END_VAR
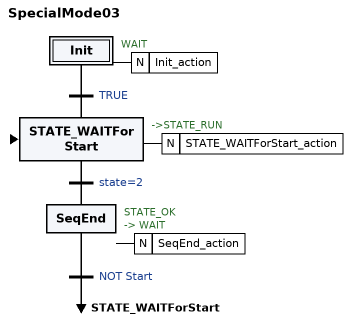
[picture p0: SpecialMode03 (SFC)]
INITIAL_STEP Init: (* WAIT *)
	Init_action(N);
END_STEP
TRANSITION FROM Init TO STATE_WAITForStart := TRUE;
END_TRANSITION
STEP STATE_WAITForStart: (* ->STATE_RUN *)
	STATE_WAITForStart_action(N);
END_STEP
TRANSITION FROM STATE_WAITForStart TO SeqEnd := state=2;
END_TRANSITION
STEP SeqEnd: (* STATE_OK / -> WAIT *)
	SeqEnd_action(N);
END_STEP
TRANSITION FROM SeqEnd TO STATE_WAITForStart := NOT Start;
END_TRANSITION

ACTION Init_action:
Start:=FALSE;
State:=STATE_WAIT;
END_ACTION

ACTION STATE_WAITForStart_action:
IF Start=TRUE
THEN
	State:=STATE_RUN;
	Result:=RESULT_NON;
	SFCTimeStart:=TIME();
(*ELSE*)
END_IF
END_ACTION

ACTION SeqEnd_action:
IF 	State=STATE_RUN THEN
	SFCTime:=TIME_TO_DINT(TIME()-SFCTimeStart);
	State:=STATE_OK;
END_IF

IF 	NOT Start THEN
	State:=STATE_WAIT;
END_IF
END_ACTION
END_PROGRAM

(* POU Stations/ST_00/ST00_SFCs/CheckSFCInInit, ST *)
PROGRAM CheckSFCInInit

VAR_OUTPUT

  AllSeqInInit	:	BOOL;

END_VAR
 AllSeqInInit:=
	ST03_Main.State=STATE_WAIT AND
	ST02_Main.State=STATE_WAIT AND
	(ST08_Process.State=STATE_WAIT OR ST08_Process.State=STATE_OK ) AND
	ST08_Palletizing.State=STATE_WAIT AND
	ST08_Depalletizing.State=STATE_WAIT
;
END_PROGRAM

(* POU Stations/ST_03_Ruestsaetze/ST_03_SFCs/ST03_Main, SFC *)
PROGRAM ST03_Main

VAR_OUTPUT
	SFCCurrentPOU			: STRING:='ST03_Main';
	SFCCurrentStep			: STRING:='';
	FB_CurrentStepHistorie	: FB_CurrentStepHistorie;
	SFCTime					: DINT;
	State   				: StateObject	:= STATE_WAIT;

	Nest10Locked			: BOOL;
	Nest10Done				: BOOL;
	IstPosHelp				: LREAL;
END_VAR
VAR_INPUT
	RunEmpty				: BOOL;
	TestPartsRemove			: BOOL;
	Result 					: DINT;
END_VAR
VAR
	MsgOK					: BOOL;
	MsgCancel				: BOOL;
	SFCRun					: BOOL;
	SFCTimeStart			: TIME;
	Delay					: TON;
	Error					: ErrorStruct;
	(* Userdefinded area *)
	AnzahlTeile   			: DINT;
	PutIdx					: DINT;
	Nest_Empty      		: BOOL;
	kein_Teil_NOK			: BOOL;
	CTR						: DINT;
	CTR2					: DINT;
	Result_help				: DINT;
END_VAR
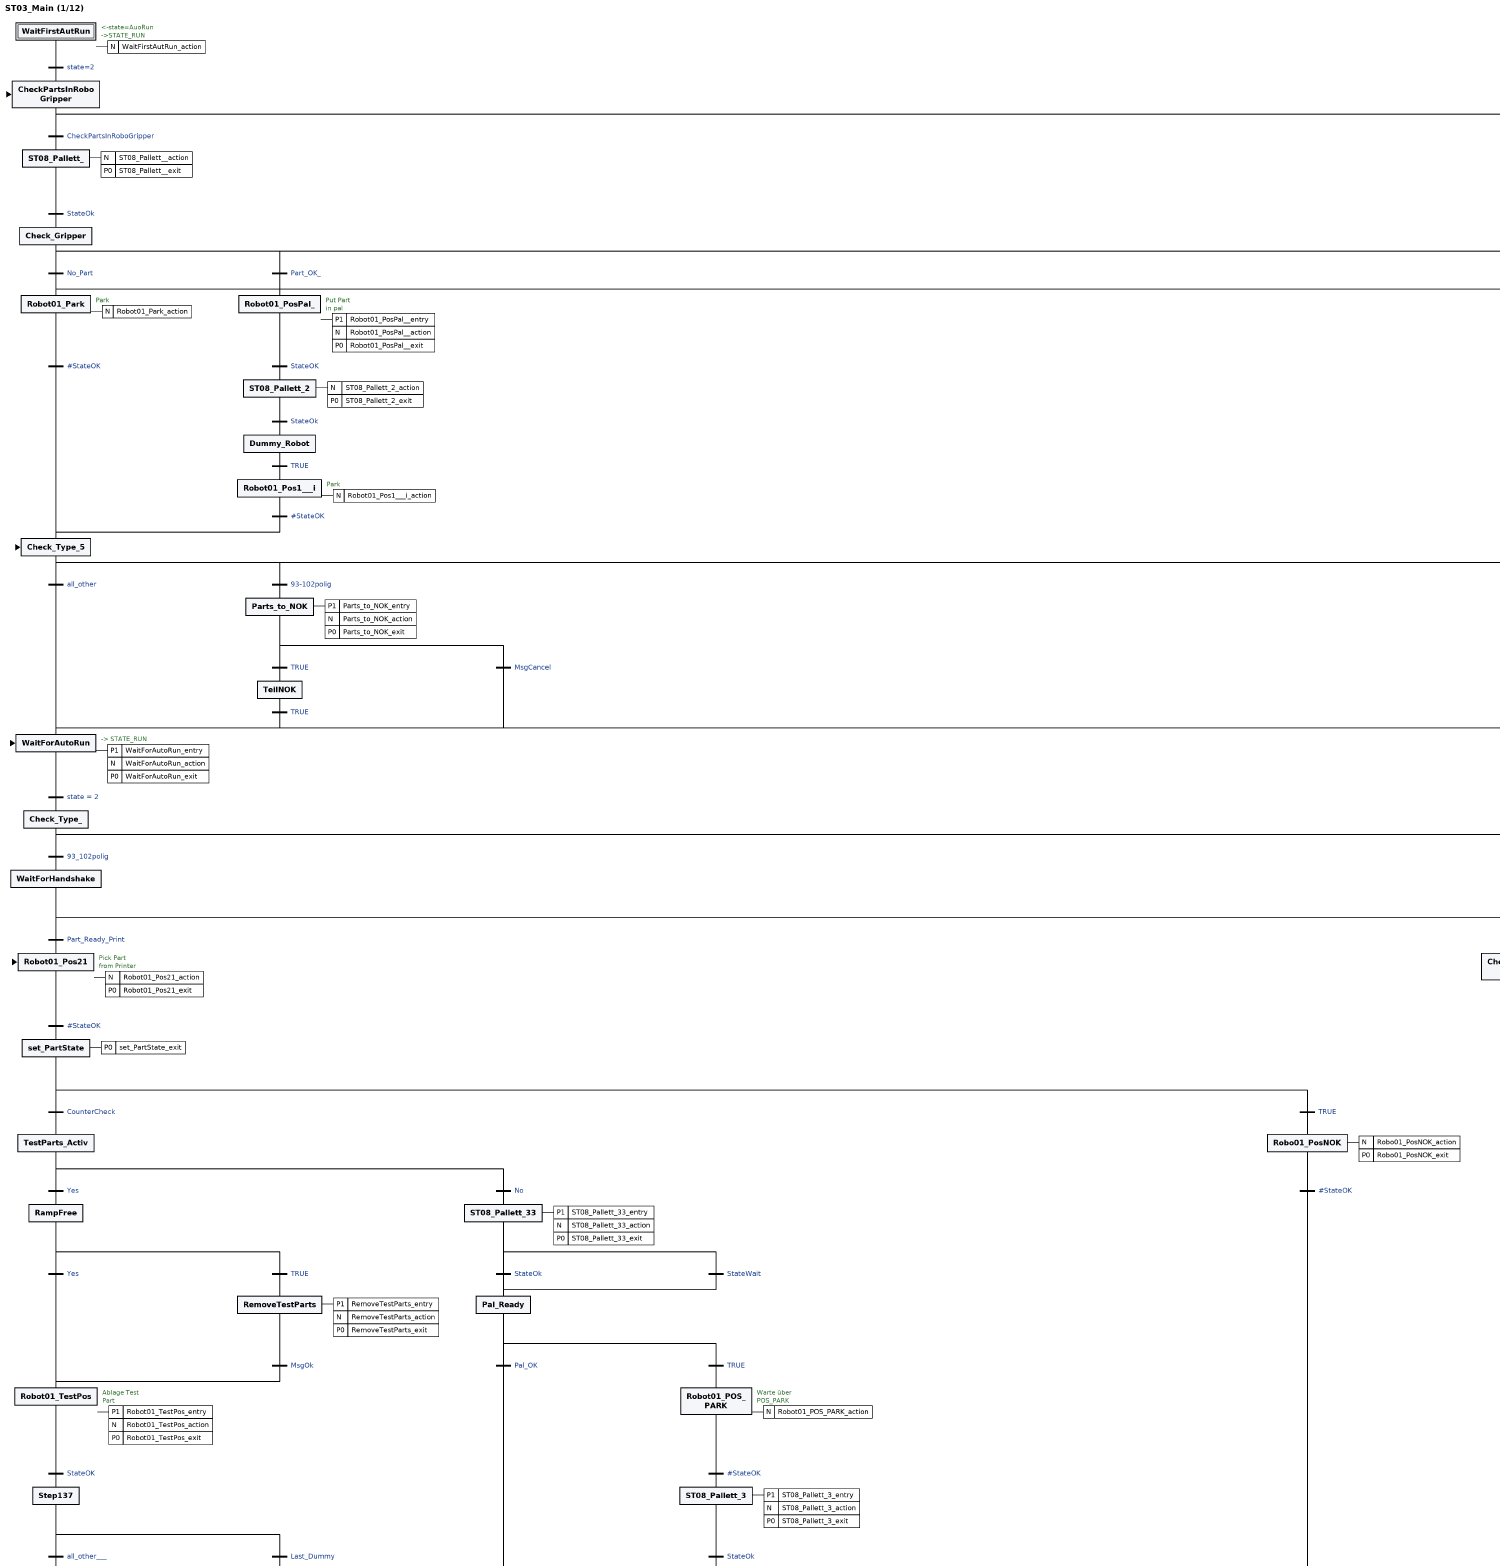
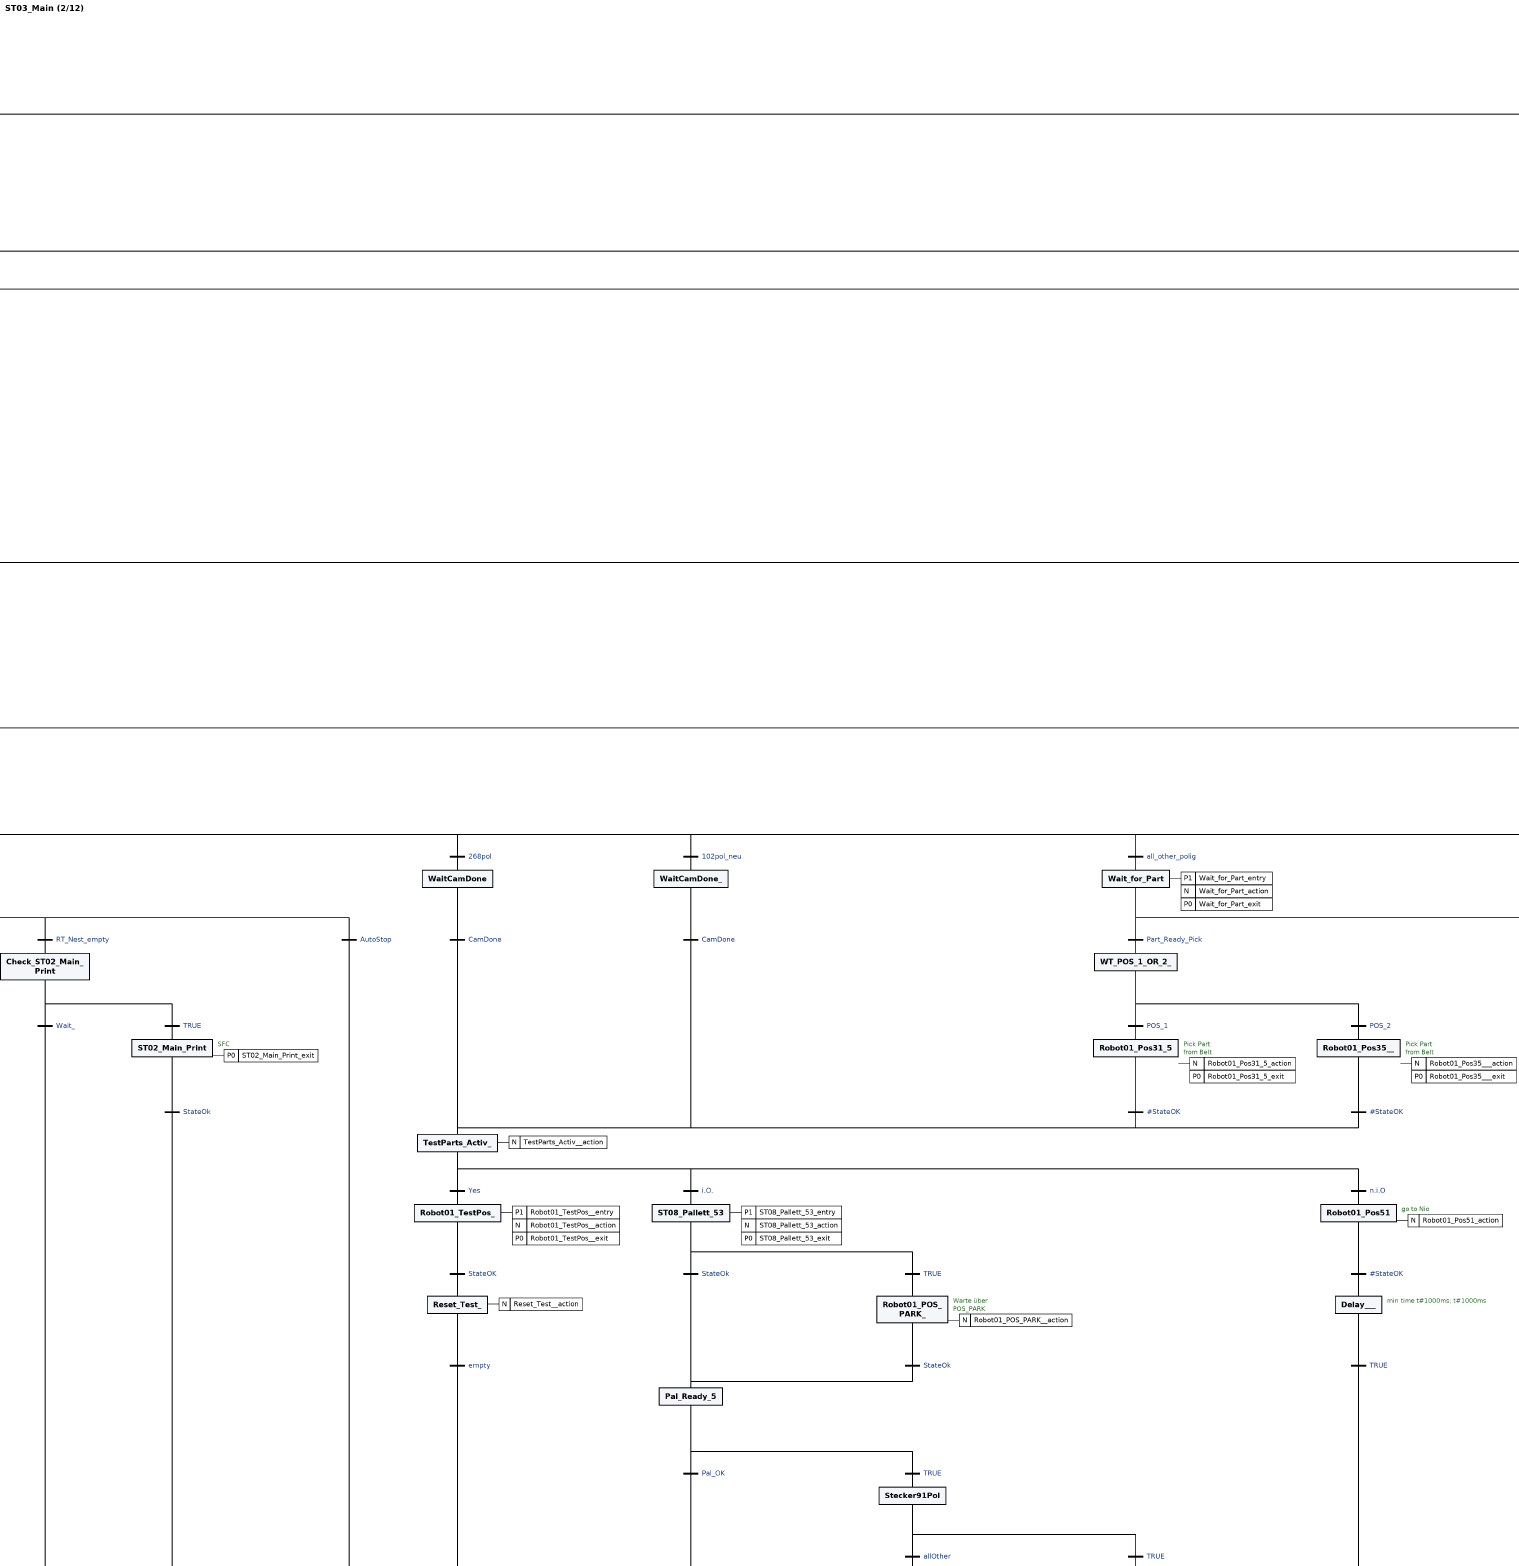
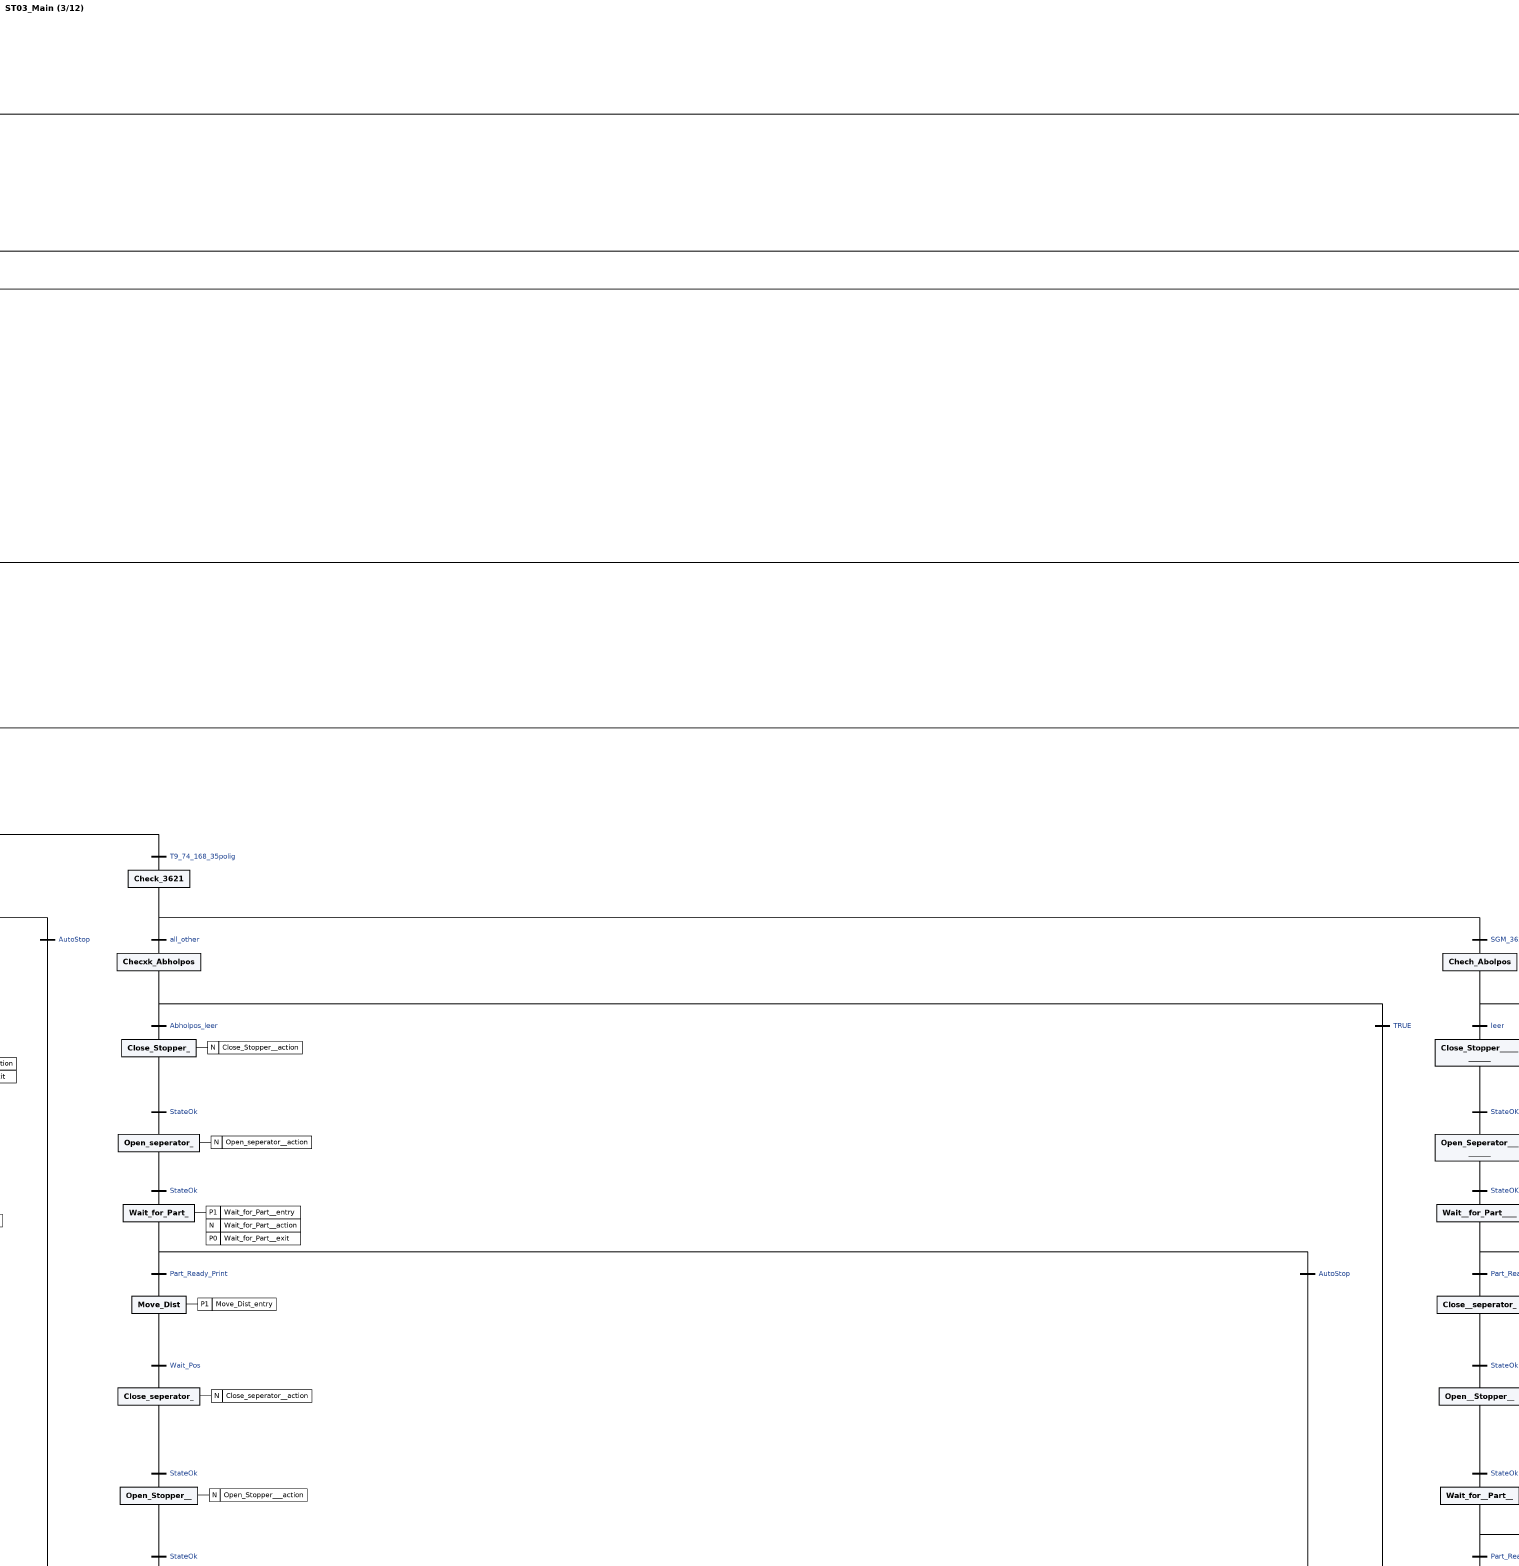
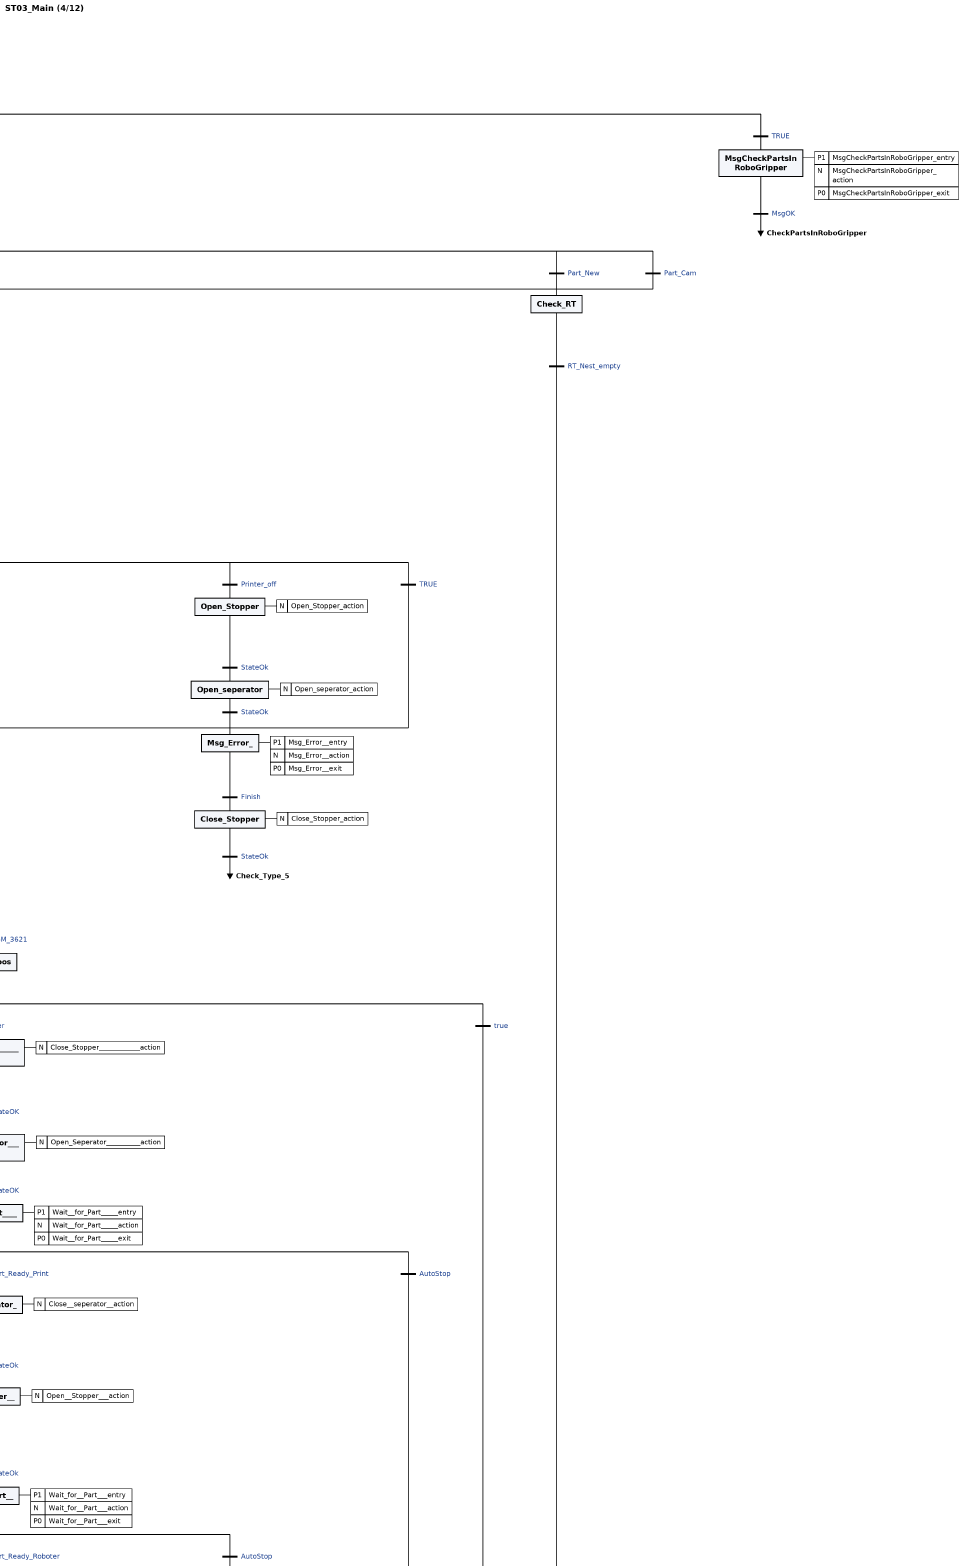
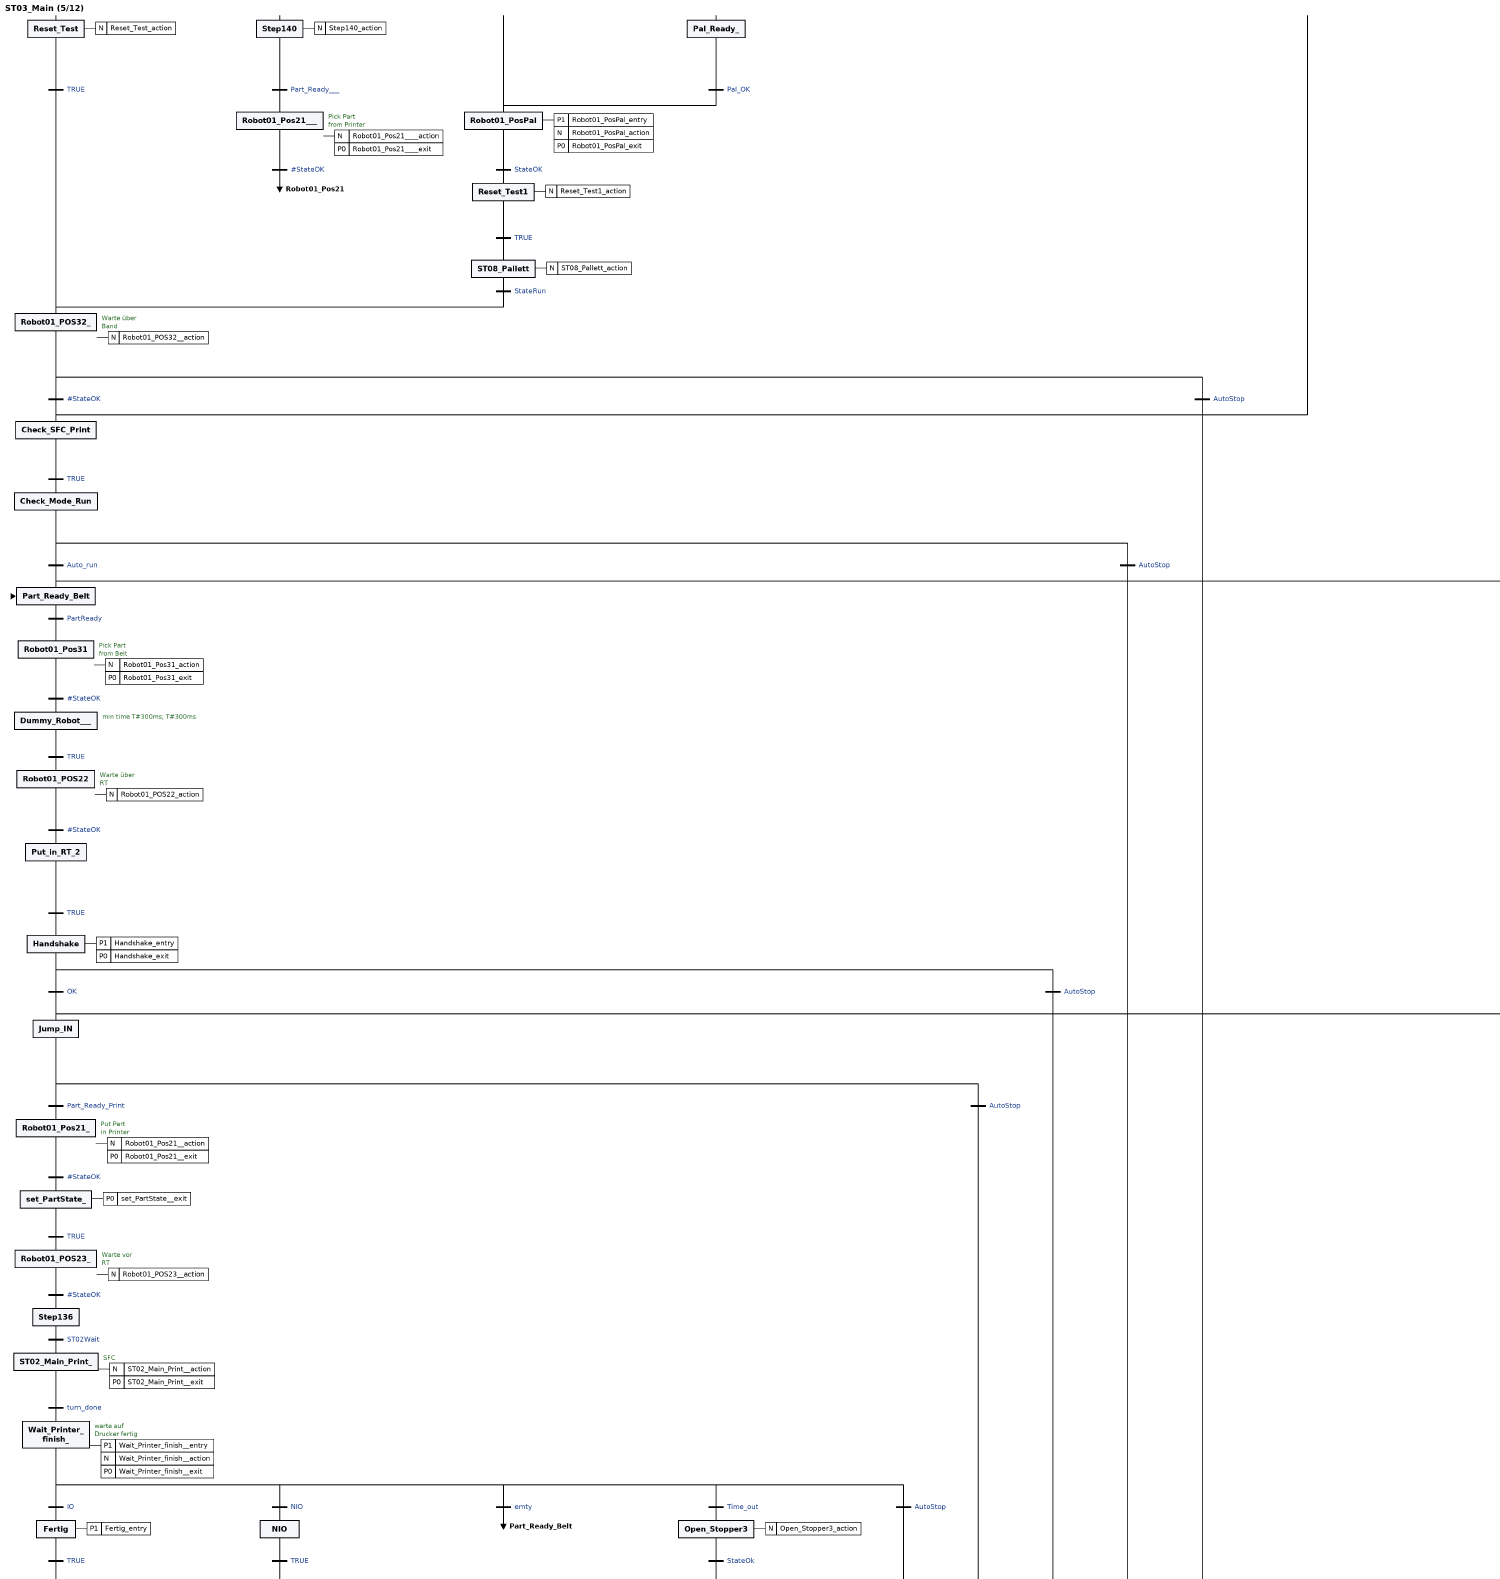
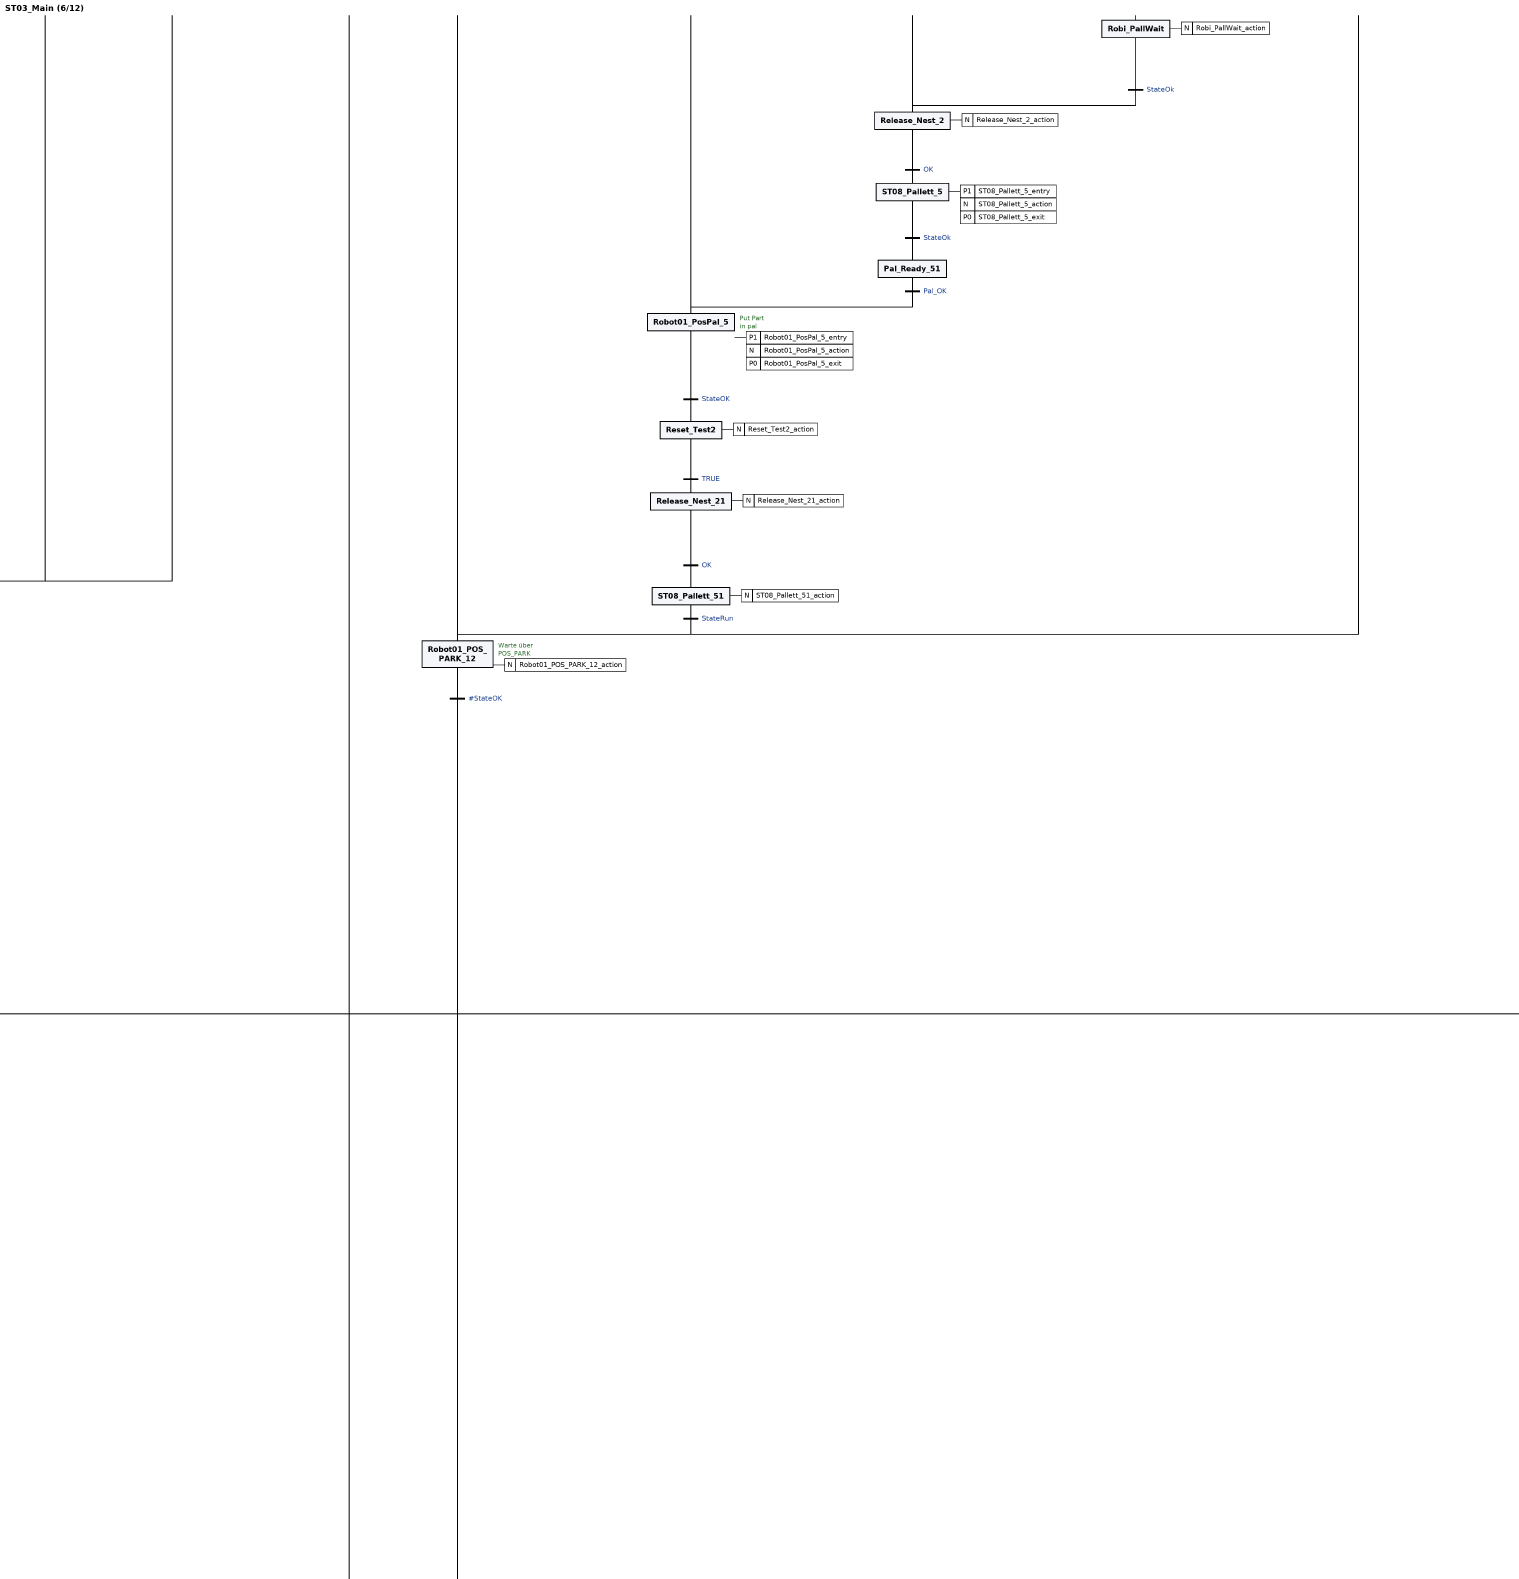
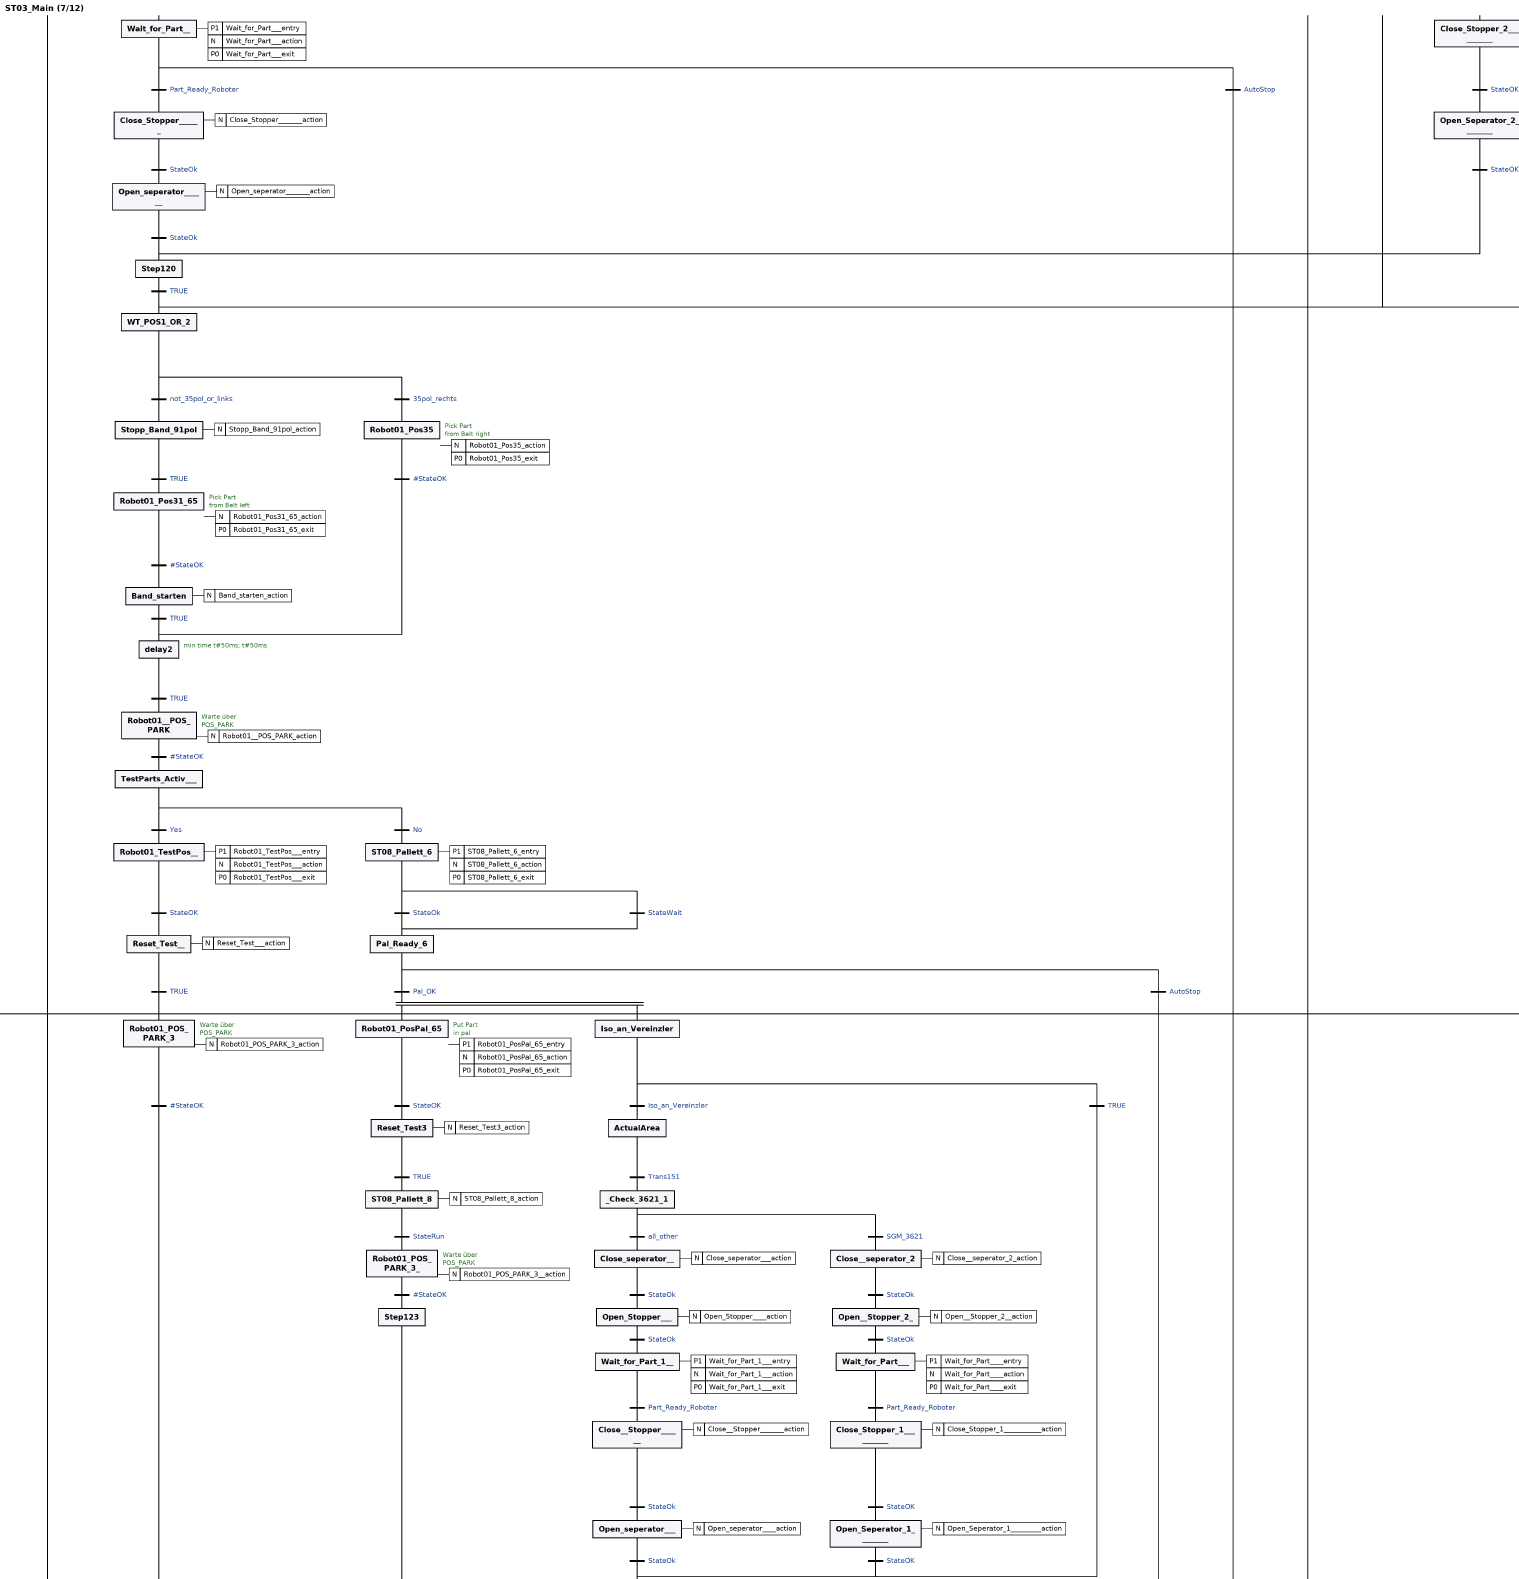
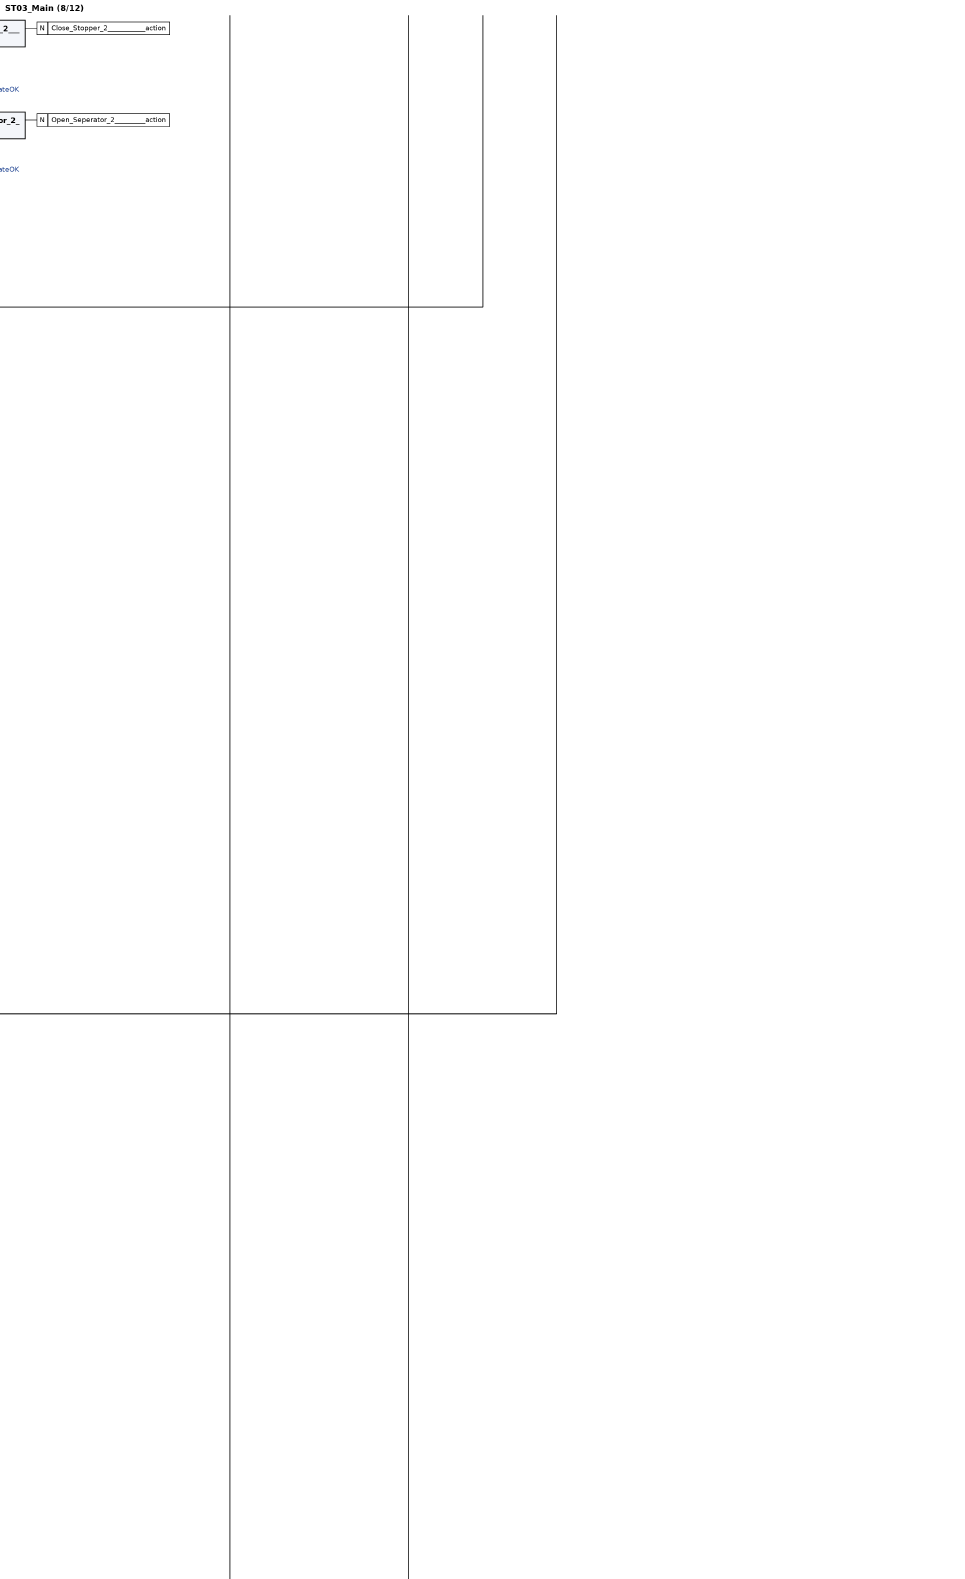
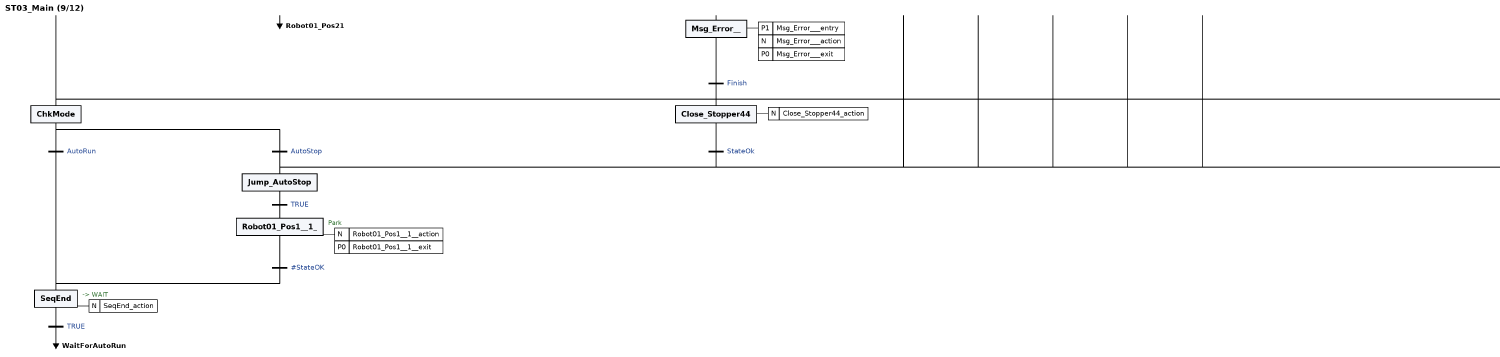
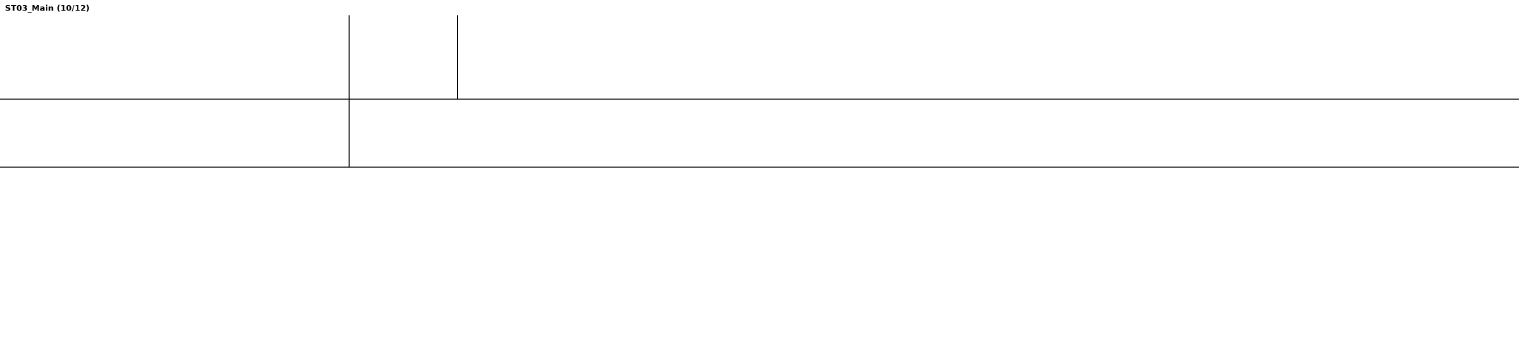
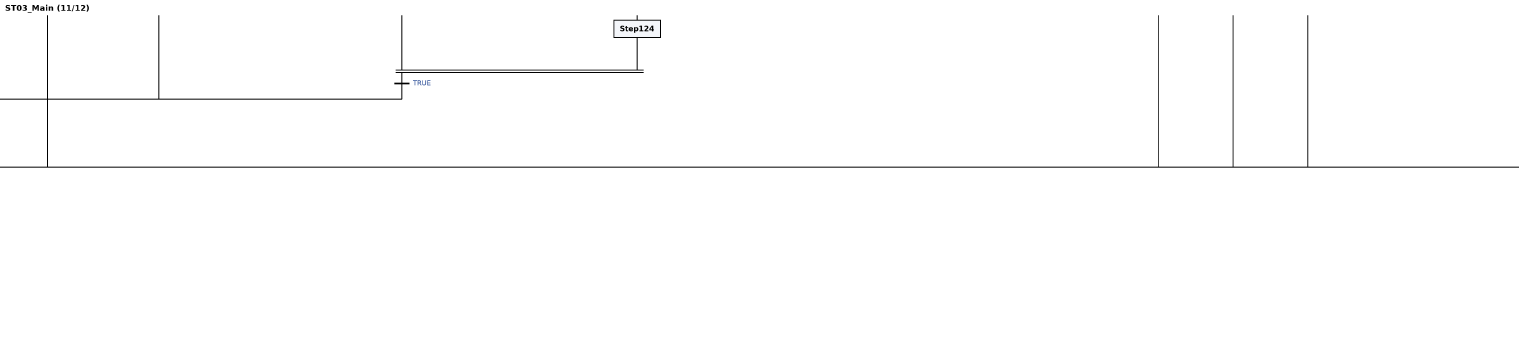
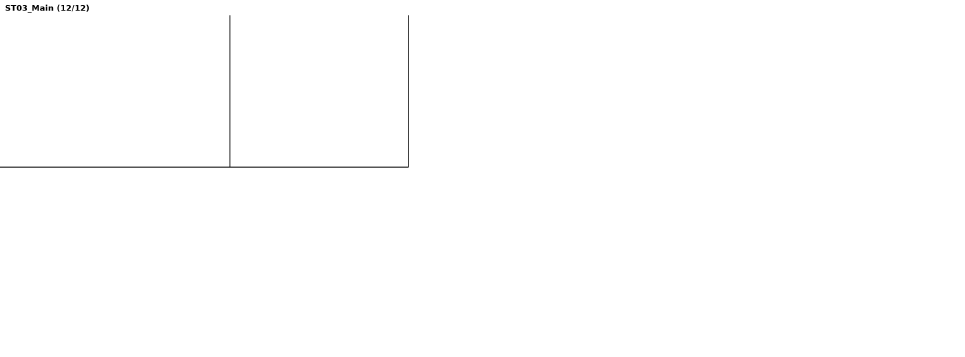
INITIAL_STEP WaitFirstAutRun: (* <-state=AuoRun / ->STATE_RUN *)
	WaitFirstAutRun_action(N);
END_STEP
TRANSITION FROM WaitFirstAutRun TO CheckPartsInRoboGripper := state=2;
END_TRANSITION
STEP CheckPartsInRoboGripper:
END_STEP
TRANSITION FROM CheckPartsInRoboGripper TO ST08_Pallett_ := CheckPartsInRoboGripper;
END_TRANSITION
TRANSITION FROM CheckPartsInRoboGripper TO MsgCheckPartsInRoboGripper := TRUE;
END_TRANSITION
STEP MsgCheckPartsInRoboGripper:
	MsgCheckPartsInRoboGripper_entry(P1);
	MsgCheckPartsInRoboGripper_action(N);
	MsgCheckPartsInRoboGripper_exit(P0);
END_STEP
TRANSITION FROM MsgCheckPartsInRoboGripper TO CheckPartsInRoboGripper := MsgOK;
END_TRANSITION
STEP ST08_Pallett_:
	ST08_Pallett__action(N);
	ST08_Pallett__exit(P0);
END_STEP
TRANSITION FROM ST08_Pallett_ TO Check_Gripper := StateOk;
END_TRANSITION
STEP Check_Gripper:
END_STEP
TRANSITION FROM Check_Gripper TO Robot01_Park := No_Part;
END_TRANSITION
TRANSITION FROM Check_Gripper TO Robot01_PosPal_ := Part_OK_;
END_TRANSITION
TRANSITION FROM Check_Gripper TO Check_RT := Part_New;
END_TRANSITION
TRANSITION FROM Check_Gripper TO Robot01_Park := Part_Cam;
END_TRANSITION
STEP Robot01_PosPal_: (* Put Part / in pal *)
	Robot01_PosPal__entry(P1);
	Robot01_PosPal__action(N);
	Robot01_PosPal__exit(P0);
END_STEP
TRANSITION FROM Robot01_PosPal_ TO ST08_Pallett_2 := StateOK;
END_TRANSITION
STEP ST08_Pallett_2:
	ST08_Pallett_2_action(N);
	ST08_Pallett_2_exit(P0);
END_STEP
TRANSITION FROM ST08_Pallett_2 TO Dummy_Robot := StateOk;
END_TRANSITION
STEP Dummy_Robot:
END_STEP
TRANSITION FROM Dummy_Robot TO Robot01_Pos1___i := TRUE;
END_TRANSITION
STEP Robot01_Pos1___i: (* Park *)
	Robot01_Pos1___i_action(N);
END_STEP
TRANSITION FROM Robot01_Pos1___i TO Check_Type_5 := #StateOK;
END_TRANSITION
STEP Check_RT:
END_STEP
TRANSITION FROM Check_RT TO Jump_IN := RT_Nest_empty;
END_TRANSITION
STEP Robot01_Park: (* Park *)
	Robot01_Park_action(N);
END_STEP
TRANSITION FROM Robot01_Park TO Check_Type_5 := #StateOK;
END_TRANSITION
STEP Check_Type_5:
END_STEP
TRANSITION FROM Check_Type_5 TO WaitForAutoRun := all_other;
END_TRANSITION
TRANSITION FROM Check_Type_5 TO Parts_to_NOK := 93-102polig;
END_TRANSITION
TRANSITION FROM Check_Type_5 TO Open_Stopper := Printer_off;
END_TRANSITION
TRANSITION FROM Check_Type_5 TO WaitForAutoRun := TRUE;
END_TRANSITION
STEP Parts_to_NOK:
	Parts_to_NOK_entry(P1);
	Parts_to_NOK_action(N);
	Parts_to_NOK_exit(P0);
END_STEP
TRANSITION FROM Parts_to_NOK TO TeilNOK := TRUE;
END_TRANSITION
TRANSITION FROM Parts_to_NOK TO WaitForAutoRun := MsgCancel;
END_TRANSITION
STEP TeilNOK:
END_STEP
TRANSITION FROM TeilNOK TO WaitForAutoRun := TRUE;
END_TRANSITION
STEP Open_Stopper:
	Open_Stopper_action(N);
END_STEP
TRANSITION FROM Open_Stopper TO Open_seperator := StateOk;
END_TRANSITION
STEP Open_seperator:
	Open_seperator_action(N);
END_STEP
TRANSITION FROM Open_seperator TO Msg_Error_ := StateOk;
END_TRANSITION
STEP Msg_Error_:
	Msg_Error__entry(P1);
	Msg_Error__action(N);
	Msg_Error__exit(P0);
END_STEP
TRANSITION FROM Msg_Error_ TO Close_Stopper := Finish;
END_TRANSITION
STEP Close_Stopper:
	Close_Stopper_action(N);
END_STEP
TRANSITION FROM Close_Stopper TO Check_Type_5 := StateOk;
END_TRANSITION
STEP WaitForAutoRun: (* -> STATE_RUN *)
	WaitForAutoRun_entry(P1);
	WaitForAutoRun_action(N);
	WaitForAutoRun_exit(P0);
END_STEP
TRANSITION FROM WaitForAutoRun TO Check_Type_ := state = 2;
END_TRANSITION
STEP Check_Type_:
END_STEP
TRANSITION FROM Check_Type_ TO WaitForHandshake := 93_102polig;
END_TRANSITION
TRANSITION FROM Check_Type_ TO WaitCamDone := 268pol;
END_TRANSITION
TRANSITION FROM Check_Type_ TO WaitCamDone_ := 102pol_neu;
END_TRANSITION
TRANSITION FROM Check_Type_ TO Wait_for_Part := all_other_polig;
END_TRANSITION
TRANSITION FROM Check_Type_ TO Check_3621 := T9_74_168_35polig;
END_TRANSITION
STEP WaitCamDone:
END_STEP
TRANSITION FROM WaitCamDone TO TestParts_Activ_ := CamDone;
END_TRANSITION
STEP WaitCamDone_:
END_STEP
TRANSITION FROM WaitCamDone_ TO TestParts_Activ_ := CamDone;
END_TRANSITION
STEP Wait_for_Part: (*  *)
	Wait_for_Part_entry(P1);
	Wait_for_Part_action(N);
	Wait_for_Part_exit(P0);
END_STEP
TRANSITION FROM Wait_for_Part TO WT_POS_1_OR_2_ := Part_Ready_Pick;
END_TRANSITION
TRANSITION FROM Wait_for_Part TO Jump_AutoStop := AutoStop;
END_TRANSITION
STEP WT_POS_1_OR_2_:
END_STEP
TRANSITION FROM WT_POS_1_OR_2_ TO Robot01_Pos31_5 := POS_1;
END_TRANSITION
TRANSITION FROM WT_POS_1_OR_2_ TO Robot01_Pos35__ := POS_2;
END_TRANSITION
STEP Robot01_Pos35__: (* Pick Part / from Belt *)
	Robot01_Pos35___action(N);
	Robot01_Pos35___exit(P0);
END_STEP
TRANSITION FROM Robot01_Pos35__ TO TestParts_Activ_ := #StateOK;
END_TRANSITION
STEP Robot01_Pos31_5: (* Pick Part / from Belt *)
	Robot01_Pos31_5_action(N);
	Robot01_Pos31_5_exit(P0);
END_STEP
TRANSITION FROM Robot01_Pos31_5 TO TestParts_Activ_ := #StateOK;
END_TRANSITION
STEP TestParts_Activ_:
	TestParts_Activ__action(N);
END_STEP
TRANSITION FROM TestParts_Activ_ TO Robot01_TestPos_ := Yes;
END_TRANSITION
TRANSITION FROM TestParts_Activ_ TO ST08_Pallett_53 := i.O.;
END_TRANSITION
TRANSITION FROM TestParts_Activ_ TO Robot01_Pos51 := n.i.O;
END_TRANSITION
STEP ST08_Pallett_53:
	ST08_Pallett_53_entry(P1);
	ST08_Pallett_53_action(N);
	ST08_Pallett_53_exit(P0);
END_STEP
TRANSITION FROM ST08_Pallett_53 TO Pal_Ready_5 := StateOk;
END_TRANSITION
TRANSITION FROM ST08_Pallett_53 TO Robot01_POS_PARK_ := TRUE;
END_TRANSITION
STEP Robot01_POS_PARK_: (* Warte über / POS_PARK *)
	Robot01_POS_PARK__action(N);
END_STEP
TRANSITION FROM Robot01_POS_PARK_ TO Pal_Ready_5 := StateOk;
END_TRANSITION
STEP Pal_Ready_5:
END_STEP
TRANSITION FROM Pal_Ready_5 TO Robot01_PosPal_5 := Pal_OK;
END_TRANSITION
TRANSITION FROM Pal_Ready_5 TO Stecker91Pol := TRUE;
END_TRANSITION
STEP Stecker91Pol:
END_STEP
TRANSITION FROM Stecker91Pol TO Release_Nest_2 := allOther;
END_TRANSITION
TRANSITION FROM Stecker91Pol TO Robi_PallWait := TRUE;
END_TRANSITION
STEP Robi_PallWait:
	Robi_PallWait_action(N);
END_STEP
TRANSITION FROM Robi_PallWait TO Release_Nest_2 := StateOk;
END_TRANSITION
STEP Release_Nest_2:
	Release_Nest_2_action(N);
END_STEP
TRANSITION FROM Release_Nest_2 TO ST08_Pallett_5 := OK;
END_TRANSITION
STEP ST08_Pallett_5:
	ST08_Pallett_5_entry(P1);
	ST08_Pallett_5_action(N);
	ST08_Pallett_5_exit(P0);
END_STEP
TRANSITION FROM ST08_Pallett_5 TO Pal_Ready_51 := StateOk;
END_TRANSITION
STEP Pal_Ready_51:
END_STEP
TRANSITION FROM Pal_Ready_51 TO Robot01_PosPal_5 := Pal_OK;
END_TRANSITION
STEP Robot01_PosPal_5: (* Put Part / in pal *)
	Robot01_PosPal_5_entry(P1);
	Robot01_PosPal_5_action(N);
	Robot01_PosPal_5_exit(P0);
END_STEP
TRANSITION FROM Robot01_PosPal_5 TO Reset_Test2 := StateOK;
END_TRANSITION
STEP Reset_Test2:
	Reset_Test2_action(N);
END_STEP
TRANSITION FROM Reset_Test2 TO Release_Nest_21 := TRUE;
END_TRANSITION
STEP Release_Nest_21:
	Release_Nest_21_action(N);
END_STEP
TRANSITION FROM Release_Nest_21 TO ST08_Pallett_51 := OK;
END_TRANSITION
STEP ST08_Pallett_51:
	ST08_Pallett_51_action(N);
END_STEP
TRANSITION FROM ST08_Pallett_51 TO Robot01_POS_PARK_12 := StateRun;
END_TRANSITION
STEP Robot01_Pos51: (* go to Nio *)
	Robot01_Pos51_action(N);
END_STEP
TRANSITION FROM Robot01_Pos51 TO Delay___ := #StateOK;
END_TRANSITION
STEP Delay___: (* min time t#1000ms; t#1000ms *)
END_STEP
TRANSITION FROM Delay___ TO Robot01_POS_PARK_12 := TRUE;
END_TRANSITION
STEP Robot01_TestPos_:
	Robot01_TestPos__entry(P1);
	Robot01_TestPos__action(N);
	Robot01_TestPos__exit(P0);
END_STEP
TRANSITION FROM Robot01_TestPos_ TO Reset_Test_ := StateOK;
END_TRANSITION
STEP Reset_Test_:
	Reset_Test__action(N);
END_STEP
TRANSITION FROM Reset_Test_ TO Robot01_POS_PARK_12 := empty;
END_TRANSITION
STEP Robot01_POS_PARK_12: (* Warte über / POS_PARK *)
	Robot01_POS_PARK_12_action(N);
END_STEP
TRANSITION FROM Robot01_POS_PARK_12 TO ChkMode := #StateOK;
END_TRANSITION
STEP Check_3621:
END_STEP
TRANSITION FROM Check_3621 TO Checxk_Abholpos := all_other;
END_TRANSITION
TRANSITION FROM Check_3621 TO Chech_Abolpos := SGM_3621;
END_TRANSITION
STEP Chech_Abolpos:
END_STEP
TRANSITION FROM Chech_Abolpos TO Close_Stopper___________ := leer;
END_TRANSITION
TRANSITION FROM Chech_Abolpos TO WT_POS1_OR_2 := true;
END_TRANSITION
STEP Close_Stopper___________:
	Close_Stopper____________action(N);
END_STEP
TRANSITION FROM Close_Stopper___________ TO Open_Seperator_________ := StateOK;
END_TRANSITION
STEP Open_Seperator_________:
	Open_Seperator__________action(N);
END_STEP
TRANSITION FROM Open_Seperator_________ TO Wait__for_Part____ := StateOK;
END_TRANSITION
STEP Wait__for_Part____: (*  *)
	Wait__for_Part_____entry(P1);
	Wait__for_Part_____action(N);
	Wait__for_Part_____exit(P0);
END_STEP
TRANSITION FROM Wait__for_Part____ TO Close__seperator_ := Part_Ready_Print;
END_TRANSITION
TRANSITION FROM Wait__for_Part____ TO Jump_AutoStop := AutoStop;
END_TRANSITION
STEP Close__seperator_:
	Close__seperator__action(N);
END_STEP
TRANSITION FROM Close__seperator_ TO Open__Stopper__ := StateOk;
END_TRANSITION
STEP Open__Stopper__:
	Open__Stopper___action(N);
END_STEP
TRANSITION FROM Open__Stopper__ TO Wait_for__Part__ := StateOk;
END_TRANSITION
STEP Wait_for__Part__:
	Wait_for__Part___entry(P1);
	Wait_for__Part___action(N);
	Wait_for__Part___exit(P0);
END_STEP
TRANSITION FROM Wait_for__Part__ TO Close_Stopper_2__________ := Part_Ready_Roboter;
END_TRANSITION
TRANSITION FROM Wait_for__Part__ TO Jump_AutoStop := AutoStop;
END_TRANSITION
STEP Close_Stopper_2__________:
	Close_Stopper_2___________action(N);
END_STEP
TRANSITION FROM Close_Stopper_2__________ TO Open_Seperator_2________ := StateOK;
END_TRANSITION
STEP Open_Seperator_2________:
	Open_Seperator_2_________action(N);
END_STEP
TRANSITION FROM Open_Seperator_2________ TO Step120 := StateOK;
END_TRANSITION
STEP Checxk_Abholpos:
END_STEP
TRANSITION FROM Checxk_Abholpos TO Close_Stopper_ := Abholpos_leer;
END_TRANSITION
TRANSITION FROM Checxk_Abholpos TO WT_POS1_OR_2 := TRUE;
END_TRANSITION
STEP Close_Stopper_:
	Close_Stopper__action(N);
END_STEP
TRANSITION FROM Close_Stopper_ TO Open_seperator_ := StateOk;
END_TRANSITION
STEP Open_seperator_:
	Open_seperator__action(N);
END_STEP
TRANSITION FROM Open_seperator_ TO Wait_for_Part_ := StateOk;
END_TRANSITION
STEP Wait_for_Part_: (*  *)
	Wait_for_Part__entry(P1);
	Wait_for_Part__action(N);
	Wait_for_Part__exit(P0);
END_STEP
TRANSITION FROM Wait_for_Part_ TO Move_Dist := Part_Ready_Print;
END_TRANSITION
TRANSITION FROM Wait_for_Part_ TO Jump_AutoStop := AutoStop;
END_TRANSITION
STEP Move_Dist:
	Move_Dist_entry(P1);
END_STEP
TRANSITION FROM Move_Dist TO Close_seperator_ := Wait_Pos;
END_TRANSITION
STEP Close_seperator_:
	Close_seperator__action(N);
END_STEP
TRANSITION FROM Close_seperator_ TO Open_Stopper__ := StateOk;
END_TRANSITION
STEP Open_Stopper__:
	Open_Stopper___action(N);
END_STEP
TRANSITION FROM Open_Stopper__ TO Wait_for_Part__ := StateOk;
END_TRANSITION
STEP Wait_for_Part__:
	Wait_for_Part___entry(P1);
	Wait_for_Part___action(N);
	Wait_for_Part___exit(P0);
END_STEP
TRANSITION FROM Wait_for_Part__ TO Close_Stopper______ := Part_Ready_Roboter;
END_TRANSITION
TRANSITION FROM Wait_for_Part__ TO Jump_AutoStop := AutoStop;
END_TRANSITION
STEP Close_Stopper______:
	Close_Stopper_______action(N);
END_STEP
TRANSITION FROM Close_Stopper______ TO Open_seperator______ := StateOk;
END_TRANSITION
STEP Open_seperator______:
	Open_seperator_______action(N);
END_STEP
TRANSITION FROM Open_seperator______ TO Step120 := StateOk;
END_TRANSITION
STEP Step120:
END_STEP
TRANSITION FROM Step120 TO WT_POS1_OR_2 := TRUE;
END_TRANSITION
STEP WT_POS1_OR_2:
END_STEP
TRANSITION FROM WT_POS1_OR_2 TO Stopp_Band_91pol := not_35pol_or_links;
END_TRANSITION
TRANSITION FROM WT_POS1_OR_2 TO Robot01_Pos35 := 35pol_rechts;
END_TRANSITION
STEP Robot01_Pos35: (* Pick Part / from Belt right *)
	Robot01_Pos35_action(N);
	Robot01_Pos35_exit(P0);
END_STEP
TRANSITION FROM Robot01_Pos35 TO delay2 := #StateOK;
END_TRANSITION
STEP Stopp_Band_91pol:
	Stopp_Band_91pol_action(N);
END_STEP
TRANSITION FROM Stopp_Band_91pol TO Robot01_Pos31_65 := TRUE;
END_TRANSITION
STEP Robot01_Pos31_65: (* Pick Part / from Belt left *)
	Robot01_Pos31_65_action(N);
	Robot01_Pos31_65_exit(P0);
END_STEP
TRANSITION FROM Robot01_Pos31_65 TO Band_starten := #StateOK;
END_TRANSITION
STEP Band_starten:
	Band_starten_action(N);
END_STEP
TRANSITION FROM Band_starten TO delay2 := TRUE;
END_TRANSITION
STEP delay2: (* min time t#50ms; t#50ms *)
END_STEP
TRANSITION FROM delay2 TO Robot01__POS_PARK := TRUE;
END_TRANSITION
STEP Robot01__POS_PARK: (* Warte über / POS_PARK *)
	Robot01__POS_PARK_action(N);
END_STEP
TRANSITION FROM Robot01__POS_PARK TO TestParts_Activ___ := #StateOK;
END_TRANSITION
STEP TestParts_Activ___:
END_STEP
TRANSITION FROM TestParts_Activ___ TO Robot01_TestPos__ := Yes;
END_TRANSITION
TRANSITION FROM TestParts_Activ___ TO ST08_Pallett_6 := No;
END_TRANSITION
STEP ST08_Pallett_6:
	ST08_Pallett_6_entry(P1);
	ST08_Pallett_6_action(N);
	ST08_Pallett_6_exit(P0);
END_STEP
TRANSITION FROM ST08_Pallett_6 TO Pal_Ready_6 := StateOk;
END_TRANSITION
TRANSITION FROM ST08_Pallett_6 TO Pal_Ready_6 := StateWait;
END_TRANSITION
STEP Pal_Ready_6:
END_STEP
TRANSITION FROM Pal_Ready_6 TO (Robot01_PosPal_65, Iso_an_Vereinzler) := Pal_OK;
END_TRANSITION
TRANSITION FROM Pal_Ready_6 TO Jump_AutoStop := AutoStop;
END_TRANSITION
STEP Robot01_PosPal_65: (* Put Part / in pal *)
	Robot01_PosPal_65_entry(P1);
	Robot01_PosPal_65_action(N);
	Robot01_PosPal_65_exit(P0);
END_STEP
TRANSITION FROM Robot01_PosPal_65 TO Reset_Test3 := StateOK;
END_TRANSITION
STEP Reset_Test3:
	Reset_Test3_action(N);
END_STEP
TRANSITION FROM Reset_Test3 TO ST08_Pallett_8 := TRUE;
END_TRANSITION
STEP ST08_Pallett_8:
	ST08_Pallett_8_action(N);
END_STEP
TRANSITION FROM ST08_Pallett_8 TO Robot01_POS_PARK_3_ := StateRun;
END_TRANSITION
STEP Robot01_POS_PARK_3_: (* Warte über / POS_PARK *)
	Robot01_POS_PARK_3__action(N);
END_STEP
TRANSITION FROM Robot01_POS_PARK_3_ TO Step123 := #StateOK;
END_TRANSITION
STEP Step123:
END_STEP
STEP Iso_an_Vereinzler:
END_STEP
TRANSITION FROM Iso_an_Vereinzler TO ActualArea := Iso_an_Vereinzler;
END_TRANSITION
TRANSITION FROM Iso_an_Vereinzler TO Step124 := TRUE;
END_TRANSITION
STEP ActualArea:
END_STEP
TRANSITION FROM ActualArea TO _Check_3621_1 := Trans151;
END_TRANSITION
STEP _Check_3621_1:
END_STEP
TRANSITION FROM _Check_3621_1 TO Close_seperator__ := all_other;
END_TRANSITION
TRANSITION FROM _Check_3621_1 TO Close__seperator_2 := SGM_3621;
END_TRANSITION
STEP Close__seperator_2:
	Close__seperator_2_action(N);
END_STEP
TRANSITION FROM Close__seperator_2 TO Open__Stopper_2_ := StateOk;
END_TRANSITION
STEP Open__Stopper_2_:
	Open__Stopper_2__action(N);
END_STEP
TRANSITION FROM Open__Stopper_2_ TO Wait_for_Part___ := StateOk;
END_TRANSITION
STEP Wait_for_Part___:
	Wait_for_Part____entry(P1);
	Wait_for_Part____action(N);
	Wait_for_Part____exit(P0);
END_STEP
TRANSITION FROM Wait_for_Part___ TO Close_Stopper_1__________ := Part_Ready_Roboter;
END_TRANSITION
STEP Close_Stopper_1__________:
	Close_Stopper_1___________action(N);
END_STEP
TRANSITION FROM Close_Stopper_1__________ TO Open_Seperator_1________ := StateOK;
END_TRANSITION
STEP Open_Seperator_1________:
	Open_Seperator_1_________action(N);
END_STEP
TRANSITION FROM Open_Seperator_1________ TO Step124 := StateOK;
END_TRANSITION
STEP Close_seperator__:
	Close_seperator___action(N);
END_STEP
TRANSITION FROM Close_seperator__ TO Open_Stopper___ := StateOk;
END_TRANSITION
STEP Open_Stopper___:
	Open_Stopper____action(N);
END_STEP
TRANSITION FROM Open_Stopper___ TO Wait_for_Part_1__ := StateOk;
END_TRANSITION
STEP Wait_for_Part_1__:
	Wait_for_Part_1___entry(P1);
	Wait_for_Part_1___action(N);
	Wait_for_Part_1___exit(P0);
END_STEP
TRANSITION FROM Wait_for_Part_1__ TO Close__Stopper______ := Part_Ready_Roboter;
END_TRANSITION
STEP Close__Stopper______:
	Close__Stopper_______action(N);
END_STEP
TRANSITION FROM Close__Stopper______ TO Open_seperator___ := StateOk;
END_TRANSITION
STEP Open_seperator___:
	Open_seperator____action(N);
END_STEP
TRANSITION FROM Open_seperator___ TO Step124 := StateOk;
END_TRANSITION
STEP Step124:
END_STEP
TRANSITION FROM (Step123, Step124) TO ChkMode := TRUE;
END_TRANSITION
STEP Robot01_TestPos__:
	Robot01_TestPos___entry(P1);
	Robot01_TestPos___action(N);
	Robot01_TestPos___exit(P0);
END_STEP
TRANSITION FROM Robot01_TestPos__ TO Reset_Test__ := StateOK;
END_TRANSITION
STEP Reset_Test__:
	Reset_Test___action(N);
END_STEP
TRANSITION FROM Reset_Test__ TO Robot01_POS_PARK_3 := TRUE;
END_TRANSITION
STEP Robot01_POS_PARK_3: (* Warte über / POS_PARK *)
	Robot01_POS_PARK_3_action(N);
END_STEP
TRANSITION FROM Robot01_POS_PARK_3 TO ChkMode := #StateOK;
END_TRANSITION
STEP WaitForHandshake: (*  *)
END_STEP
TRANSITION FROM WaitForHandshake TO Robot01_Pos21 := Part_Ready_Print;
END_TRANSITION
TRANSITION FROM WaitForHandshake TO Check_ST02_Main_Print := RT_Nest_empty;
END_TRANSITION
TRANSITION FROM WaitForHandshake TO Jump_AutoStop := AutoStop;
END_TRANSITION
STEP Check_ST02_Main_Print:
END_STEP
TRANSITION FROM Check_ST02_Main_Print TO Part_Ready_Belt := Wait_;
END_TRANSITION
TRANSITION FROM Check_ST02_Main_Print TO ST02_Main_Print := TRUE;
END_TRANSITION
STEP ST02_Main_Print: (* SFC *)
	ST02_Main_Print_exit(P0);
END_STEP
TRANSITION FROM ST02_Main_Print TO Part_Ready_Belt := StateOk;
END_TRANSITION
STEP Robot01_Pos21: (* Pick Part / from Printer *)
	Robot01_Pos21_action(N);
	Robot01_Pos21_exit(P0);
END_STEP
TRANSITION FROM Robot01_Pos21 TO set_PartState := #StateOK;
END_TRANSITION
STEP set_PartState:
	set_PartState_exit(P0);
END_STEP
TRANSITION FROM set_PartState TO TestParts_Activ := CounterCheck;
END_TRANSITION
TRANSITION FROM set_PartState TO Robo01_PosNOK := TRUE;
END_TRANSITION
STEP Robo01_PosNOK:
	Robo01_PosNOK_action(N);
	Robo01_PosNOK_exit(P0);
END_STEP
TRANSITION FROM Robo01_PosNOK TO Check_SFC_Print := #StateOK;
END_TRANSITION
STEP TestParts_Activ:
END_STEP
TRANSITION FROM TestParts_Activ TO RampFree := Yes;
END_TRANSITION
TRANSITION FROM TestParts_Activ TO ST08_Pallett_33 := No;
END_TRANSITION
STEP ST08_Pallett_33:
	ST08_Pallett_33_entry(P1);
	ST08_Pallett_33_action(N);
	ST08_Pallett_33_exit(P0);
END_STEP
TRANSITION FROM ST08_Pallett_33 TO Pal_Ready := StateOk;
END_TRANSITION
TRANSITION FROM ST08_Pallett_33 TO Pal_Ready := StateWait;
END_TRANSITION
STEP Pal_Ready:
END_STEP
TRANSITION FROM Pal_Ready TO Robot01_PosPal := Pal_OK;
END_TRANSITION
TRANSITION FROM Pal_Ready TO Robot01_POS_PARK := TRUE;
END_TRANSITION
STEP Robot01_POS_PARK: (* Warte über / POS_PARK *)
	Robot01_POS_PARK_action(N);
END_STEP
TRANSITION FROM Robot01_POS_PARK TO ST08_Pallett_3 := #StateOK;
END_TRANSITION
STEP ST08_Pallett_3:
	ST08_Pallett_3_entry(P1);
	ST08_Pallett_3_action(N);
	ST08_Pallett_3_exit(P0);
END_STEP
TRANSITION FROM ST08_Pallett_3 TO Pal_Ready_ := StateOk;
END_TRANSITION
STEP Pal_Ready_:
END_STEP
TRANSITION FROM Pal_Ready_ TO Robot01_PosPal := Pal_OK;
END_TRANSITION
STEP Robot01_PosPal:
	Robot01_PosPal_entry(P1);
	Robot01_PosPal_action(N);
	Robot01_PosPal_exit(P0);
END_STEP
TRANSITION FROM Robot01_PosPal TO Reset_Test1 := StateOK;
END_TRANSITION
STEP Reset_Test1:
	Reset_Test1_action(N);
END_STEP
TRANSITION FROM Reset_Test1 TO ST08_Pallett := TRUE;
END_TRANSITION
STEP ST08_Pallett:
	ST08_Pallett_action(N);
END_STEP
TRANSITION FROM ST08_Pallett TO Robot01_POS32_ := StateRun;
END_TRANSITION
STEP RampFree:
END_STEP
TRANSITION FROM RampFree TO Robot01_TestPos := Yes;
END_TRANSITION
TRANSITION FROM RampFree TO RemoveTestParts := TRUE;
END_TRANSITION
STEP RemoveTestParts:
	RemoveTestParts_entry(P1);
	RemoveTestParts_action(N);
	RemoveTestParts_exit(P0);
END_STEP
TRANSITION FROM RemoveTestParts TO Robot01_TestPos := MsgOk;
END_TRANSITION
STEP Robot01_TestPos: (* Ablage Test / Part *)
	Robot01_TestPos_entry(P1);
	Robot01_TestPos_action(N);
	Robot01_TestPos_exit(P0);
END_STEP
TRANSITION FROM Robot01_TestPos TO Step137 := StateOK;
END_TRANSITION
STEP Step137:
END_STEP
TRANSITION FROM Step137 TO Reset_Test := all_other___;
END_TRANSITION
TRANSITION FROM Step137 TO Step140 := Last_Dummy;
END_TRANSITION
STEP Step140:
	Step140_action(N);
END_STEP
TRANSITION FROM Step140 TO Robot01_Pos21___ := Part_Ready___;
END_TRANSITION
STEP Robot01_Pos21___: (* Pick Part / from Printer *)
	Robot01_Pos21____action(N);
	Robot01_Pos21____exit(P0);
END_STEP
TRANSITION FROM Robot01_Pos21___ TO Robot01_Pos21 := #StateOK;
END_TRANSITION
STEP Reset_Test:
	Reset_Test_action(N);
END_STEP
TRANSITION FROM Reset_Test TO Robot01_POS32_ := TRUE;
END_TRANSITION
STEP Robot01_POS32_: (* Warte über / Band *)
	Robot01_POS32__action(N);
END_STEP
TRANSITION FROM Robot01_POS32_ TO Check_SFC_Print := #StateOK;
END_TRANSITION
TRANSITION FROM Robot01_POS32_ TO Jump_AutoStop := AutoStop;
END_TRANSITION
STEP Check_SFC_Print:
END_STEP
TRANSITION FROM Check_SFC_Print TO Check_Mode_Run := TRUE;
END_TRANSITION
STEP Check_Mode_Run:
END_STEP
TRANSITION FROM Check_Mode_Run TO Part_Ready_Belt := Auto_run;
END_TRANSITION
TRANSITION FROM Check_Mode_Run TO Jump_AutoStop := AutoStop;
END_TRANSITION
STEP Part_Ready_Belt:
END_STEP
TRANSITION FROM Part_Ready_Belt TO Robot01_Pos31 := PartReady;
END_TRANSITION
STEP Robot01_Pos31: (* Pick Part / from Belt *)
	Robot01_Pos31_action(N);
	Robot01_Pos31_exit(P0);
END_STEP
TRANSITION FROM Robot01_Pos31 TO Dummy_Robot___ := #StateOK;
END_TRANSITION
STEP Dummy_Robot___: (* min time T#300ms; T#300ms *)
END_STEP
TRANSITION FROM Dummy_Robot___ TO Robot01_POS22 := TRUE;
END_TRANSITION
STEP Robot01_POS22: (* Warte über / RT *)
	Robot01_POS22_action(N);
END_STEP
TRANSITION FROM Robot01_POS22 TO Put_in_RT_2 := #StateOK;
END_TRANSITION
STEP Put_in_RT_2:
END_STEP
TRANSITION FROM Put_in_RT_2 TO Handshake := TRUE;
END_TRANSITION
STEP Handshake:
	Handshake_entry(P1);
	Handshake_exit(P0);
END_STEP
TRANSITION FROM Handshake TO Jump_IN := OK;
END_TRANSITION
TRANSITION FROM Handshake TO Jump_AutoStop := AutoStop;
END_TRANSITION
STEP Jump_IN:
END_STEP
TRANSITION FROM Jump_IN TO Robot01_Pos21_ := Part_Ready_Print;
END_TRANSITION
TRANSITION FROM Jump_IN TO Jump_AutoStop := AutoStop;
END_TRANSITION
STEP Robot01_Pos21_: (* Put Part / in Printer *)
	Robot01_Pos21__action(N);
	Robot01_Pos21__exit(P0);
END_STEP
TRANSITION FROM Robot01_Pos21_ TO set_PartState_ := #StateOK;
END_TRANSITION
STEP set_PartState_:
	set_PartState__exit(P0);
END_STEP
TRANSITION FROM set_PartState_ TO Robot01_POS23_ := TRUE;
END_TRANSITION
STEP Robot01_POS23_: (* Warte vor / RT *)
	Robot01_POS23__action(N);
END_STEP
TRANSITION FROM Robot01_POS23_ TO Step136 := #StateOK;
END_TRANSITION
STEP Step136:
END_STEP
TRANSITION FROM Step136 TO ST02_Main_Print_ := ST02Wait;
END_TRANSITION
STEP ST02_Main_Print_: (* SFC *)
	ST02_Main_Print__action(N);
	ST02_Main_Print__exit(P0);
END_STEP
TRANSITION FROM ST02_Main_Print_ TO Wait_Printer_finish_ := turn_done;
END_TRANSITION
STEP Wait_Printer_finish_: (* warte auf / Drucker fertig *)
	Wait_Printer_finish__entry(P1);
	Wait_Printer_finish__action(N);
	Wait_Printer_finish__exit(P0);
END_STEP
TRANSITION FROM Wait_Printer_finish_ TO Fertig := IO;
END_TRANSITION
TRANSITION FROM Wait_Printer_finish_ TO NIO := NIO;
END_TRANSITION
TRANSITION FROM Wait_Printer_finish_ TO Part_Ready_Belt := emty;
END_TRANSITION
TRANSITION FROM Wait_Printer_finish_ TO Open_Stopper3 := Time_out;
END_TRANSITION
TRANSITION FROM Wait_Printer_finish_ TO Jump_AutoStop := AutoStop;
END_TRANSITION
STEP NIO:
END_STEP
TRANSITION FROM NIO TO Robot01_Pos21 := TRUE;
END_TRANSITION
STEP Open_Stopper3:
	Open_Stopper3_action(N);
END_STEP
TRANSITION FROM Open_Stopper3 TO Msg_Error__ := StateOk;
END_TRANSITION
STEP Msg_Error__:
	Msg_Error___entry(P1);
	Msg_Error___action(N);
	Msg_Error___exit(P0);
END_STEP
TRANSITION FROM Msg_Error__ TO Close_Stopper44 := Finish;
END_TRANSITION
STEP Close_Stopper44:
	Close_Stopper44_action(N);
END_STEP
TRANSITION FROM Close_Stopper44 TO Jump_AutoStop := StateOk;
END_TRANSITION
STEP Fertig:
	Fertig_entry(P1);
END_STEP
TRANSITION FROM Fertig TO ChkMode := TRUE;
END_TRANSITION
STEP ChkMode:
END_STEP
TRANSITION FROM ChkMode TO SeqEnd := AutoRun;
END_TRANSITION
TRANSITION FROM ChkMode TO Jump_AutoStop := AutoStop;
END_TRANSITION
STEP Jump_AutoStop:
END_STEP
TRANSITION FROM Jump_AutoStop TO Robot01_Pos1__1_ := TRUE;
END_TRANSITION
STEP Robot01_Pos1__1_: (* Park *)
	Robot01_Pos1__1__action(N);
	Robot01_Pos1__1__exit(P0);
END_STEP
TRANSITION FROM Robot01_Pos1__1_ TO SeqEnd := #StateOK;
END_TRANSITION
STEP SeqEnd: (* -> WAIT *)
	SeqEnd_action(N);
END_STEP
TRANSITION FROM SeqEnd TO WaitForAutoRun := TRUE;
END_TRANSITION

ACTION WaitFirstAutRun_action:
IF 	ModeSelect.Mode=MODE_AUTO_RUN OR
	ModeSelect.Mode=MODE_STEP_RUN OR
	(SpecialMode06.State=State_Run AND
	(gTypeCode=312 OR			(*93pol*)
	gTypeCode=499)) 			(*102pol*)
THEN
	State:=STATE_RUN;
ELSE
	State:=STATE_WAIT;
	MsgOK:=FALSE;
	MsgCancel:=FALSE;
	SFCRun:=FALSE;
END_IF

Nest10Locked:=FALSE;
Nest10Done:=FALSE;
Side_1:=FALSE;
Side_2:=FALSE;
PutIdx:=0;
Nest_Empty:=FALSE;
ST03_Autostop.Start:=FALSE;
CTR:=0;
CTR2:=0;
END_ACTION

ACTION MsgCheckPartsInRoboGripper_entry:
MessageHandler.ClearMessageLines(sVisu:=Visu.Message);
MsgOk := FALSE;
END_ACTION

ACTION MsgCheckPartsInRoboGripper_action:
MessageHandler.Msg.ID:='PM121';
MessageHandler.Msg.Name:='Anzahl Teile im Greifer darf nicht 0 sein';
MessageHandler.Msg.Text:= 'Anzahl Teile im Greifer darf nicht 0 sein ';
MessageHandler.Msg.Color:=Color.red;
MessageHandler.Msg.Station:=1;

MessageHandler(
	Prio:=2, 								(*1=highest, .. , 4=lowest*)
	Btn1Addr:=ADR(MsgOk),		(*Address of Button1 , if Zero then Button is unvisible*)
	Btn2Addr:=0,						(*Address of Button2 , if Zero then Button is unvisible*)
	sVisu:=Visu.Message);
END_ACTION

ACTION MsgCheckPartsInRoboGripper_exit:
MsgOk := FALSE;
END_ACTION

ACTION ST08_Pallett__action:
IF 	ST08_Process.State=STATE_WAIT THEN
	ST08_Process.Start:=TRUE;
END_IF
END_ACTION

ACTION ST08_Pallett__exit:
ST08_Process.Start:=FALSE;
END_ACTION

ACTION Robot01_PosPal__entry:
IF 	PosIdx<TD.PartsInRoboGripper THEN
	PosIdx:=TD.PartsInRoboGripper;
END_IF
END_ACTION

ACTION Robot01_PosPal__action:
Robot01.PosNo:=POS_FEED_PAL_WAIT + (PosIdx/TD.PartsInRoboGripper);
Robot01.PosOffset:=gRobotOffset;
Robot01.Override:=MP.ST00.Override;
Robot01.SetToolOn:=TRUE;
Robot01.SetToolOff:=FALSE;
Robot01.ExecuteMove:=TRUE;
END_ACTION

ACTION Robot01_PosPal__exit:
gRob01GripState:=PART_NO;
PosIdx:=PosIdx+TD.PartsInRoboGripper;
gPartsInserted:=gPartsInserted+TD.PartsInRoboGripper;
gPartsTest:=gPartsTest+TD.PartsInRoboGripper;
END_ACTION

ACTION ST08_Pallett_2_action:
IF 	ST08_Process.State=STATE_WAIT THEN
	ST08_Process.Start:=TRUE;
END_IF
END_ACTION

ACTION ST08_Pallett_2_exit:
ST08_Process.Start:=FALSE;
END_ACTION

ACTION Robot01_Pos1___i_action:
Robot01.PosNo:=POS_PARK;
Robot01.PosOffset:=gRobotOffset;
Robot01.Override:=MP.ST00.Override;
(*Robot01.SetToolOn:=TRUE;
Robot01.SetToolOff:=FALSE;*)
Robot01.ExecuteMove:=TRUE;
END_ACTION

ACTION Robot01_Park_action:
Robot01.PosNo:=POS_PARK;
Robot01.PosOffset:=gRobotOffset;
Robot01.Override:=MP.ST00.Override;
Robot01.SetToolOn:=TRUE;
Robot01.SetToolOff:=FALSE;
Robot01.ExecuteMove:=TRUE;
END_ACTION

ACTION Parts_to_NOK_entry:
MessageHandler.ClearMessageLines(sVisu:=Visu.Message);
END_ACTION

ACTION Parts_to_NOK_action:
MessageHandler.Msg.ID:='PM114';
MessageHandler.Msg.Name:='Start Stecker 93polig';
MessageHandler.Msg.Text:='Solllen die ersten Teile auf NOK pos gelegt werden -> mit OK$R';
MessageHandler.Msg.Text:=CONCAT(MessageHandler.Msg.Text,'-> Abbrechen, sofort in Palettierer');
MessageHandler.Msg.Color:=Color.yellow;
MessageHandler.Msg.Station:=1;


MessageHandler(
	Prio:=2, 									(*1=highest, .. , 4=lowest*)
	Btn1Addr:=ADR(MsgOk),			(*Address of Button1 , if Zero then Button is unvisible*)
	Btn2Addr:=ADR(MsgCancel),	(*Address of Button2 , if Zero then Button is unvisible*)
	sVisu:=Visu.Message);


MessageHandler.MessageLine[1].Visible:=TRUE;
MessageHandler.MessageLine[1].Editable:=TRUE;
MessageHandler.MessageLine[1].Text:='Anzahl Teile auf NOK';
MessageHandler.MessageLine[1].MsgTypeEnum:=MsgDataTypeDint;
END_ACTION

ACTION Parts_to_NOK_exit:
MsgOk:=FALSE;
MsgCancel:=FALSE;
AnzahlTeile:=MessageHandler.MessageLine[1].MsgInt;

(*erstes Teil soll immer in nok Box*)
IF AnzahlTeile < 3 THEN
	AnzahlTeile := 3;
END_IF
END_ACTION

ACTION Open_Stopper_action:
ST00_74_Y2_4.MoveWork:=TRUE;
END_ACTION

ACTION Open_seperator_action:
ST00_74_Y2_5.MoveInit:=TRUE;
END_ACTION

ACTION Msg_Error__entry:
MessageHandler.ClearMessageLines(sVisu:=Visu.Message);
END_ACTION

ACTION Msg_Error__action:
MessageHandler.Msg.ID:='PM115';
MessageHandler.Msg.Name:='Drucker';
MessageHandler.Msg.Text:='Kein Betriebsbereit vom Drucker!Drucker Einschalten weiter mit OK ';
MessageHandler.Msg.Color:=Color.Red;
MessageHandler.Msg.Station:=1;


MessageHandler(
	Prio:=2, 									(*1=highest, .. , 4=lowest*)
	Btn1Addr:=ADR(MsgOk),			(*Address of Button1 , if Zero then Button is unvisible*)
	Btn2Addr:=0,	(*Address of Button2 , if Zero then Button is unvisible*)
	sVisu:=Visu.Message);
END_ACTION

ACTION Msg_Error__exit:
MessageHandler.ClearMessageLines(sVisu:=Visu.Message);
MsgOk:=FALSE;
END_ACTION

ACTION Close_Stopper_action:
ST00_74_Y2_4.MoveInit:=TRUE;
END_ACTION

ACTION WaitForAutoRun_entry:
ST03_Autostop.Start:=FALSE;
END_ACTION

ACTION WaitForAutoRun_action:
IF 	(ModeSelect.Mode=MODE_AUTO_RUN OR
	ModeSelect.Mode=MODE_STEP_RUN OR
	(SpecialMode06.State=State_Run AND
	(gTypeCode=312 OR			(*93pol*)
	gTypeCode=499) ) ) AND			(*102pol*)
	NOT gRunEmpty
THEN
	State:=STATE_RUN;
	SFCTimeStart:=TIME();
ELSE
	State:=STATE_WAIT;
	MsgOK:=FALSE;
	MsgCancel:=FALSE;
	SFCRun:=FALSE;
	ST08_Process.Start:=FALSE;
END_IF

IF 	CTR >= MP.ST03.NoOfTestParts THEN
	CTR:=0;
	gTakeTestParts:=FALSE;
	gTakeTestPartsAuto:=FALSE;
END_IF

IF 	CTR2 >= MP.ST02.NoOfDummys THEN
	CTR2:=0;
	MP.ST02.DummyPruefung_93pol := FALSE;
END_IF
END_ACTION

ACTION WaitForAutoRun_exit:
ST03_Autostop.Start:=TRUE;
END_ACTION

ACTION Wait_for_Part_entry:
ProcessMessage01:='';
Delay.IN:=FALSE;
Delay();
END_ACTION

ACTION Wait_for_Part_action:
ProcessMessage01:='1IM10';(*warte auf Teil in Abholpositon*)
Delay(IN:=ST03_Init_AbholPos.RoboPos31 OR ST03_Init_AbholPos.RoboPos35);
Delay.PT:=T#50ms;
END_ACTION

ACTION Wait_for_Part_exit:
ProcessMessage01:='';
END_ACTION

ACTION Robot01_Pos35___action:
Robot01.PosNo:=POS_WT_POS2;
Robot01.PosOffset:=gRobotOffset;
Robot01.Override:=MP.ST00.Override;
Robot01.SetToolOn:=FALSE;
Robot01.SetToolOff:=TRUE;
Robot01.ExecuteMove:=TRUE;
END_ACTION

ACTION Robot01_Pos35___exit:
IF	Result = RESULT_OK THEN
	gRob01GripState:=PART_OK;
ELSE
	gRob01GripState:=PART_NOK;
END_IF
Result:= RESULT_NON;
END_ACTION

ACTION Robot01_Pos31_5_action:
Robot01.PosNo:=POS_WT_POS1;
Robot01.PosOffset:=gRobotOffset;
Robot01.Override:=MP.ST00.Override;
Robot01.SetToolOn:=FALSE;
Robot01.SetToolOff:=TRUE;
Robot01.ExecuteMove:=TRUE;
END_ACTION

ACTION Robot01_Pos31_5_exit:
IF	Result = RESULT_OK THEN
	gRob01GripState:=PART_OK;
ELSE
	gRob01GripState:=PART_NOK;
END_IF
Result:= RESULT_NON;
END_ACTION

ACTION TestParts_Activ__action:
ST03_51_M1.MotorOn:=TRUE;
END_ACTION

ACTION ST08_Pallett_53_entry:
ProcessMessage01:='';
END_ACTION

ACTION ST08_Pallett_53_action:
ProcessMessage01:='1IM7';(*warte Pallette*)
END_ACTION

ACTION ST08_Pallett_53_exit:
ST08_Process.Start:=FALSE;
ProcessMessage01:='';
END_ACTION

ACTION Robot01_POS_PARK__action:
Robot01.PosNo:=POS_PARK;
Robot01.PosOffset:=gRobotOffset;
Robot01.Override:=MP.ST00.Override;
Robot01.SetToolOn:=FALSE;
Robot01.SetToolOff:=TRUE;
Robot01.ExecuteMove:=TRUE;
END_ACTION

ACTION Robi_PallWait_action:
Robot01.PosNo:=POS_FEED_PAL_WAIT;
	Robot01.PosOffset:=gRobotOffset;
	Robot01.Override:=MP.ST00.Override;
	Robot01.SetToolOn:=FALSE;
	Robot01.SetToolOff:=TRUE;
	Robot01.ExecuteMove:=TRUE;
END_ACTION

ACTION Release_Nest_2_action:
ST00_71_K2.SetSignalHigh:=TRUE; (* Schnittstelle Bedrucken Tinte Abholposition frei *)
END_ACTION

ACTION ST08_Pallett_5_entry:
ProcessMessage01:='';
END_ACTION

ACTION ST08_Pallett_5_action:
ProcessMessage01:='1IM7';(*warte Pallette*)
END_ACTION

ACTION ST08_Pallett_5_exit:
ST08_Process.Start:=FALSE;
ProcessMessage01:='';
END_ACTION

ACTION Robot01_PosPal_5_entry:
IF 	PosIdx<TD.PartsInRoboGripper THEN
	PosIdx:=TD.PartsInRoboGripper;
END_IF

(*für das ausschleusen der Testteile mit einem Blister*)
IF	(gTakeTestParts OR gTakeTestPartsAuto) AND
	PosIdx <= MP.ST03.NoOfTestParts THEN
	CTR:=PosIdx;
END_IF
END_ACTION

ACTION Robot01_PosPal_5_action:
Robot01.PosNo:=POS_FEED_PAL_WAIT + (PosIdx/TD.PartsInRoboGripper);
Robot01.PosOffset:=gRobotOffset;
Robot01.Override:=MP.ST00.Override;
Robot01.SetToolOn:=TRUE;
Robot01.SetToolOff:=FALSE;
Robot01.ExecuteMove:=TRUE;
END_ACTION

ACTION Robot01_PosPal_5_exit:
gRob01GripState:=PART_NO;
PosIdx:=PosIdx+ TD.PartsInRoboGripper;
gPartsInserted:=gPartsInserted+ TD.PartsInRoboGripper;
gPartsTest:=gPartsTest+ TD.PartsInRoboGripper;
END_ACTION

ACTION Reset_Test2_action:
(*für das ausschleusen der Testteile mit einem Blister*)
IF	(gTakeTestParts OR gTakeTestPartsAuto) AND
	CTR>= MP.ST03.NoOfTestParts THEN
	ST08_Palletizing.TestpartMoveOut:=TRUE;
	CTR:=0;
	gTakeTestParts:=FALSE;
	gTakeTestPartsAuto:=FALSE;
	TestPartsRemove := TRUE;
END_IF
END_ACTION

ACTION Release_Nest_21_action:
ST00_71_K2.SetSignalHigh:=TRUE; (* Schnittstelle Bedrucken Tinte Abholposition frei *)
END_ACTION

ACTION ST08_Pallett_51_action:
IF ST08_Process.State=STATE_WAIT THEN
	ST08_Process.Start:=TRUE;
END_IF
END_ACTION

ACTION Robot01_Pos51_action:
Robot01.PosNo:=POS_NOK;
Robot01.PosOffset:=gRobotOffset;
Robot01.Override:=MP.ST00.Override;
Robot01.SetToolOn:=TRUE;
Robot01.SetToolOff:=FALSE;
Robot01.ExecuteMove:=TRUE;
END_ACTION

ACTION Robot01_TestPos__entry:
CTR:=CTR+1;
END_ACTION

ACTION Robot01_TestPos__action:
Robot01.PosNo:=POS_TEST_PARTS ;
Robot01.PosOffset:=gRobotOffset;
Robot01.Override:=MP.ST00.Override;
Robot01.SetToolOn:=TRUE;
Robot01.SetToolOff:=FALSE;
Robot01.ExecuteMove:=TRUE;
END_ACTION

ACTION Robot01_TestPos__exit:
gRob01GripState:=PART_NO;
END_ACTION

ACTION Reset_Test__action:
IF CTR>=MP.ST03.NoOfTestParts THEN
	CTR:=0;
	gTakeTestParts:=FALSE;
	gTakeTestPartsAuto:=FALSE;
	TestPartsRemove:=TRUE;
END_IF
END_ACTION

ACTION Robot01_POS_PARK_12_action:
Robot01.PosNo:=POS_PARK;
Robot01.PosOffset:=gRobotOffset;
Robot01.Override:=MP.ST00.Override;
Robot01.SetToolOn:=FALSE;
Robot01.SetToolOff:=FALSE;
Robot01.ExecuteMove:=TRUE;
END_ACTION

ACTION Close_Stopper____________action:
ST03_422_Y64_6.MoveInit:=TRUE;
END_ACTION

ACTION Open_Seperator__________action:
ST03_422_Y64_5.MoveInit:=TRUE;	(* Förderband  Stopper Vereinzler AST/GST *)
END_ACTION

ACTION Wait__for_Part_____entry:
ProcessMessage01:='';
Delay.IN:=FALSE;
Delay();
END_ACTION

ACTION Wait__for_Part_____action:
ProcessMessage01:='1IM6';(*warte auf Teil in Vereinzelung*)
Delay.IN:= ST03_421_B63_7.BitInToCheck; 			 (* Schnittstelle Iso auf Übergabeposition *)
Delay.PT:=T#500ms;
Delay();
END_ACTION

ACTION Wait__for_Part_____exit:
ProcessMessage01:='';
END_ACTION

ACTION Close__seperator__action:
ST03_422_Y64_5.MoveWork:=TRUE;
END_ACTION

ACTION Open__Stopper___action:
ST03_422_Y64_6.MoveWork:=TRUE;
END_ACTION

ACTION Wait_for__Part___entry:
ProcessMessage01:='';
Delay.IN:=FALSE;
Delay();
END_ACTION

ACTION Wait_for__Part___action:
ProcessMessage01:='1IM10';(*warte auf Teil in Abholpositon*)
Delay.IN:=ST03_422_B64_4.BitInToCheck; 		 (* Teil auf Abholposition Roboter *)
Delay.PT:=T#500ms;
Delay();
END_ACTION

ACTION Wait_for__Part___exit:
ProcessMessage01:='';
END_ACTION

ACTION Close_Stopper_2___________action:
ST03_422_Y64_6.MoveInit:=TRUE;
END_ACTION

ACTION Open_Seperator_2_________action:
ST03_422_Y64_5.MoveInit:=TRUE;	(* Förderband  Stopper Vereinzler AST/GST *)
END_ACTION

ACTION Close_Stopper__action:
ST08_412_Y55_2.MoveWork:=TRUE;
END_ACTION

ACTION Open_seperator__action:
ST08_412_Y55_0.MoveInit:=TRUE;
END_ACTION

ACTION Wait_for_Part__entry:
ProcessMessage01:='';
Delay.IN:=FALSE;
Delay();
END_ACTION

ACTION Wait_for_Part__action:
ProcessMessage01:='1IM6';(*warte auf Teil in Vereinzelung*)
Delay.IN:=ST08_412_B58_7.BitInToCheck; 		 (* Schnittstelle Iso auf Übergabeposition *)
Delay.PT:=T#50ms;
Delay();
END_ACTION

ACTION Wait_for_Part__exit:
ProcessMessage01:='';
END_ACTION

ACTION Move_Dist_entry:
IstPosHelp:=ST03_51_M1.sPos.ist;
END_ACTION

ACTION Close_seperator__action:
ST08_412_Y55_0.MoveWork:=TRUE;
END_ACTION

ACTION Open_Stopper___action:
ST08_412_Y55_2.MoveInit:=TRUE;
END_ACTION

ACTION Wait_for_Part___entry:
ProcessMessage01:='';
Delay.IN:=FALSE;
Delay();
END_ACTION

ACTION Wait_for_Part___action:
ProcessMessage01:='1IM10';(*warte auf Teil in Abholpositon*)
Delay.IN:=ST08_412_B59_0.BitInToCheck; 		 (* Teil auf Abholposition Roboter *)
Delay.PT:=T#500ms;
Delay();
END_ACTION

ACTION Wait_for_Part___exit:
ProcessMessage01:='';
END_ACTION

ACTION Close_Stopper_______action:
ST08_412_Y55_2.MoveWork:=TRUE;
END_ACTION

ACTION Open_seperator_______action:
ST08_412_Y55_0.MoveInit:=TRUE;
END_ACTION

ACTION Robot01_Pos35_action:
Robot01.PosNo:=POS_WT_POS2;
Robot01.PosOffset:=gRobotOffset;
Robot01.Override:=MP.ST00.Override;
Robot01.SetToolOn:=FALSE;
Robot01.SetToolOff:=TRUE;
Robot01.ExecuteMove:=TRUE;
END_ACTION

ACTION Robot01_Pos35_exit:
gRob01GripState:=PART_OK;
END_ACTION

ACTION Stopp_Band_91pol_action:
(* Bei 91 poligen Stecker das Band anhalten*)

IF 	gTypeCode=379 THEN
	ST03_51_M1.MotorOn:=FALSE;
	ST03_51_M1.MotorOff :=TRUE;
END_IF
END_ACTION

ACTION Robot01_Pos31_65_action:
Robot01.PosNo:=POS_WT_POS1;
Robot01.PosOffset:=gRobotOffset;
Robot01.Override:=MP.ST00.Override;
Robot01.SetToolOn:=FALSE;
Robot01.SetToolOff:=TRUE;
Robot01.ExecuteMove:=TRUE;
END_ACTION

ACTION Robot01_Pos31_65_exit:
gRob01GripState:=PART_OK;
END_ACTION

ACTION Band_starten_action:
(* Band wieder starten*)

IF 	gTypeCode=379 THEN
	ST03_51_M1.MotorOn:=TRUE;
	ST03_51_M1.MotorOff :=FALSE;
END_IF
END_ACTION

ACTION Robot01__POS_PARK_action:
Robot01.PosNo:=POS_PARK;
Robot01.PosOffset:=gRobotOffset;
Robot01.Override:=MP.ST00.Override;
Robot01.SetToolOn:=FALSE;
Robot01.SetToolOff:=FALSE;
Robot01.ExecuteMove:=TRUE;
END_ACTION

ACTION ST08_Pallett_6_entry:
ProcessMessage01:='';
END_ACTION

ACTION ST08_Pallett_6_action:
ProcessMessage01:='1IM7';(*warte Pallette*)
END_ACTION

ACTION ST08_Pallett_6_exit:
ST08_Process.Start:=FALSE;
ProcessMessage01:='';
END_ACTION

ACTION Robot01_PosPal_65_entry:
IF 	PosIdx<TD.PartsInRoboGripper THEN
	PosIdx:=TD.PartsInRoboGripper;
END_IF

(*für das ausschleusen der Testteile mit einem Blister*)
IF	(gTakeTestParts OR gTakeTestPartsAuto) AND
	PosIdx <= MP.ST03.NoOfTestParts THEN
	CTR:=PosIdx;
END_IF
END_ACTION

ACTION Robot01_PosPal_65_action:
Robot01.PosNo:=POS_FEED_PAL_WAIT + PosIdx;
Robot01.PosOffset:=gRobotOffset;
Robot01.Override:=MP.ST00.Override;
Robot01.SetToolOn:=TRUE;
Robot01.SetToolOff:=FALSE;
Robot01.ExecuteMove:=TRUE;
END_ACTION

ACTION Robot01_PosPal_65_exit:
gRob01GripState:=PART_NO;
PosIdx:=PosIdx+TD.PartsInRoboGripper;
gPartsInserted:=gPartsInserted+TD.PartsInRoboGripper;
gPartsTest:=gPartsTest+ TD.PartsInRoboGripper;
END_ACTION

ACTION Reset_Test3_action:
(*für das ausschleusen der Testteile mit einem Blister*)
IF	(gTakeTestParts OR gTakeTestPartsAuto) AND
	CTR>= MP.ST03.NoOfTestParts THEN
	ST08_Palletizing.TestpartMoveOut:=TRUE;
	CTR:=0;
	gTakeTestParts:=FALSE;
	gTakeTestPartsAuto:=FALSE;
	TestPartsRemove := TRUE;
END_IF
END_ACTION

ACTION ST08_Pallett_8_action:
IF 	ST08_Process.State=STATE_WAIT THEN
	ST08_Process.Start:=TRUE;
END_IF
END_ACTION

ACTION Robot01_POS_PARK_3__action:
Robot01.PosNo:=POS_PARK;
Robot01.PosOffset:=gRobotOffset;
Robot01.Override:=MP.ST00.Override;
Robot01.SetToolOn:=FALSE;
Robot01.SetToolOff:=FALSE;
Robot01.ExecuteMove:=TRUE;
END_ACTION

ACTION Close__seperator_2_action:
ST03_422_Y64_5.MoveWork:=TRUE;
END_ACTION

ACTION Open__Stopper_2__action:
ST03_422_Y64_6.MoveWork:=TRUE;
END_ACTION

ACTION Wait_for_Part____entry:
ProcessMessage01:='';
Delay.IN:=FALSE;
Delay();
END_ACTION

ACTION Wait_for_Part____action:
ProcessMessage01:='1IM10';(*warte auf Teil in Abholpositon*)
Delay.IN:=ST03_422_B64_4.BitInToCheck; 		 (* Teil auf Abholposition Roboter *)
Delay.PT:=T#500ms;
Delay();
END_ACTION

ACTION Wait_for_Part____exit:
ProcessMessage01:='';
END_ACTION

ACTION Close_Stopper_1___________action:
ST03_422_Y64_6.MoveInit:=TRUE;
END_ACTION

ACTION Open_Seperator_1_________action:
ST03_422_Y64_5.MoveInit:=TRUE;	(* Förderband  Stopper Vereinzler AST/GST *)
END_ACTION

ACTION Close_seperator___action:
ST08_412_Y55_0.MoveWork:=TRUE;
END_ACTION

ACTION Open_Stopper____action:
ST08_412_Y55_2.MoveInit:=TRUE;
END_ACTION

ACTION Wait_for_Part_1___entry:
ProcessMessage01:='';
Delay.IN:=FALSE;
Delay();
END_ACTION

ACTION Wait_for_Part_1___action:
ProcessMessage01:='1IM10';(*warte auf Teil in Abholpositon*)
Delay.IN:=ST08_412_B59_0.BitInToCheck; 		 (* Teil auf Abholposition Roboter *)
Delay.PT:=T#500ms;
Delay();
END_ACTION

ACTION Wait_for_Part_1___exit:
ProcessMessage01:='';
END_ACTION

ACTION Close__Stopper_______action:
ST08_412_Y55_2.MoveWork:=TRUE;
END_ACTION

ACTION Open_seperator____action:
ST08_412_Y55_0.MoveInit:=TRUE;
END_ACTION

ACTION Robot01_TestPos___entry:
CTR:=CTR+1;
END_ACTION

ACTION Robot01_TestPos___action:
Robot01.PosNo:=POS_TEST_PARTS ;
Robot01.PosOffset:=gRobotOffset;
Robot01.Override:=MP.ST00.Override;
Robot01.SetToolOn:=TRUE;
Robot01.SetToolOff:=FALSE;
Robot01.ExecuteMove:=TRUE;
END_ACTION

ACTION Robot01_TestPos___exit:
gRob01GripState:=PART_NO;
END_ACTION

ACTION Reset_Test___action:
IF CTR>=MP.ST03.NoOfTestParts
THEN
	CTR:=0;
	gTakeTestParts:=FALSE;
	gTakeTestPartsAuto:=FALSE;
END_IF
END_ACTION

ACTION Robot01_POS_PARK_3_action:
Robot01.PosNo:=POS_PARK;
Robot01.PosOffset:=gRobotOffset;
Robot01.Override:=MP.ST00.Override;
Robot01.SetToolOn:=FALSE;
Robot01.SetToolOff:=FALSE;
Robot01.ExecuteMove:=TRUE;
END_ACTION

ACTION ST02_Main_Print_exit:
ST02_Main.Start:=FALSE;
SFCRun:=FALSE;
END_ACTION

ACTION Robot01_Pos21_action:
Robot01.PosNo:=POS_RT;
Robot01.PosOffset:=gRobotOffset;
Robot01.Override:=MP.ST00.Override;
Robot01.SetToolOn:=FALSE;
Robot01.SetToolOff:=TRUE;
Robot01.ExecuteMove:=TRUE;
END_ACTION

ACTION Robot01_Pos21_exit:
IF	MP.ST02.TableData[1].ProcessData.	Result =11 THEN
	gRob01GripState:= PART_OK;
ELSE
	gRob01GripState:=PART_NOK;
END_IF
END_ACTION

ACTION set_PartState_exit:
Result_help:=MP.ST02.TableData[1].ProcessData.Result;
MP.ST02.TableData[1].ProcessData.Part:= FALSE; 		 (* Schnittstelle Tampondrucker Nest 1 leer *)
MP.ST02.TableData[1].ProcessData.Result:=0;	(*   0 = Teil noch nicht bearbeitet *)
											(*   1 =  Oberseite OK*)
											(*  11 = Oberseite und Unterseite OK*)
											(*  99 = Teil ist NOK	*)
END_ACTION

ACTION Robo01_PosNOK_action:
Robot01.PosNo:=POS_NOK;
Robot01.PosOffset:=gRobotOffset;
Robot01.Override:=MP.ST00.Override;
Robot01.SetToolOn:=TRUE;
Robot01.SetToolOff:=FALSE;
Robot01.ExecuteMove:=TRUE;
END_ACTION

ACTION Robo01_PosNOK_exit:
gRob01GripState:=PART_NO;
IF	Result_help =11 THEN
	PutIdx:=PutIdx+1;
	i32_first_parts :=i32_first_parts+1;
END_IF
END_ACTION

ACTION ST08_Pallett_33_entry:
ProcessMessage01:='';
END_ACTION

ACTION ST08_Pallett_33_action:
ProcessMessage01:='1IM7';(*warte Pallette*)
END_ACTION

ACTION ST08_Pallett_33_exit:
ST08_Process.Start:=FALSE;
ProcessMessage01:='';
END_ACTION

ACTION Robot01_POS_PARK_action:
Robot01.PosNo:=POS_PARK;
Robot01.PosOffset:=gRobotOffset;
Robot01.Override:=MP.ST00.Override;
Robot01.SetToolOn:=FALSE;
Robot01.SetToolOff:=FALSE;
Robot01.ExecuteMove:=TRUE;
END_ACTION

ACTION ST08_Pallett_3_entry:
ProcessMessage01:='';
END_ACTION

ACTION ST08_Pallett_3_action:
ProcessMessage01:='1IM7';(*warte Pallette*)
END_ACTION

ACTION ST08_Pallett_3_exit:
ST08_Process.Start:=FALSE;
ProcessMessage01:='';
END_ACTION

ACTION Robot01_PosPal_entry:
IF 	PosIdx<TD.PartsInRoboGripper THEN
	PosIdx:=TD.PartsInRoboGripper;
END_IF

(*für das ausschleusen der Testteile mit einem Blister*)
IF	(gTakeTestParts OR gTakeTestPartsAuto) AND
	PosIdx <= MP.ST03.NoOfTestParts THEN
	CTR:=PosIdx;
END_IF
END_ACTION

ACTION Robot01_PosPal_action:
Robot01.PosNo:=POS_FEED_PAL_WAIT + (PosIdx/TD.PartsInRoboGripper);
Robot01.PosOffset:=gRobotOffset;
Robot01.Override:=MP.ST00.Override;
Robot01.SetToolOn:=TRUE;
Robot01.SetToolOff:=FALSE;
Robot01.ExecuteMove:=TRUE;
END_ACTION

ACTION Robot01_PosPal_exit:
gRob01GripState:=PART_NO;
PosIdx:=PosIdx+TD.PartsInRoboGripper;
gPartsInserted:=gPartsInserted+TD.PartsInRoboGripper;
gPartsTest:=gPartsTest+TD.PartsInRoboGripper;
END_ACTION

ACTION Reset_Test1_action:
(*für das ausschleusen der Testteile mit einem Blister*)
IF	(gTakeTestParts OR gTakeTestPartsAuto) AND
	CTR>= MP.ST03.NoOfTestParts THEN
	ST08_Palletizing.TestpartMoveOut:=TRUE;
	CTR:=0;
	gTakeTestParts:=FALSE;
	gTakeTestPartsAuto:=FALSE;
	TestPartsRemove := TRUE;
END_IF
END_ACTION

ACTION ST08_Pallett_action:
IF 	ST08_Process.State=STATE_WAIT THEN
	ST08_Process.Start:=TRUE;
END_IF
END_ACTION

ACTION RemoveTestParts_entry:
MessageHandler.ClearMessageLines(sVisu:=Visu.Message);
END_ACTION

ACTION RemoveTestParts_action:
IF  ST03_8_75_B13_5.SignalIn THEN		(*voll/belegt keine Prüfmittel mehr  *)
	MessageHandler.Msg.ID:='PM116';
ELSIF ST03_8_75_B13_6.SignalIn THEN	(* belegt mit 6 Prüfmittel  *)
	MessageHandler.Msg.ID:='PM117';
END_IF

MessageHandler.Msg.Name:='Prüfteile entnehmen';
MessageHandler.Msg.Text:='Kontrolle ob die Rutsche leer ist.';
MessageHandler.Msg.Color:=Color.red;
MessageHandler.Msg.Station:=1;


MessageHandler(
	Prio:=2, 							(*1=highest, .. , 4=lowest*)
	Btn1Addr:=ADR(MsgOk),			(*Address of Button1 , if Zero then Button is unvisible*)
	Btn2Addr:=0,						(*Address of Button2 , if Zero then Button is unvisible*)
	sVisu:=Visu.Message);
END_ACTION

ACTION RemoveTestParts_exit:
MsgOk:=FALSE;
MsgCancel:=FALSE;
END_ACTION

ACTION Robot01_TestPos_entry:
CTR:=CTR+1;
CTR2:=CTR2+1;
END_ACTION

ACTION Robot01_TestPos_action:
Robot01.PosNo:=POS_TEST_PARTS;
Robot01.PosOffset:=gRobotOffset;
Robot01.Override:=MP.ST00.Override;
Robot01.SetToolOn:=TRUE;
Robot01.SetToolOff:=FALSE;
Robot01.ExecuteMove:=TRUE;
END_ACTION

ACTION Robot01_TestPos_exit:
gRob01GripState:=PART_NO;
i32_first_parts :=i32_first_parts+1;
END_ACTION

ACTION Step140_action:
IF ST02_Main.State=STATE_WAIT THEN
	ST02_Main.Start:=TRUE;
END_IF
END_ACTION

ACTION Robot01_Pos21____action:
Robot01.PosNo:=POS_RT;
Robot01.PosOffset:=gRobotOffset;
Robot01.Override:=MP.ST00.Override;
Robot01.SetToolOn:=FALSE;
Robot01.SetToolOff:=TRUE;
Robot01.ExecuteMove:=TRUE;
END_ACTION

ACTION Robot01_Pos21____exit:
IF	MP.ST02.TableData[1].ProcessData.	Result =11 THEN
	gRob01GripState:= PART_OK;
ELSE
	gRob01GripState:=PART_NOK;
END_IF
END_ACTION

ACTION Reset_Test_action:
IF NOT MP.ST02.DummyPruefung_93pol AND
 CTR=MP.ST03.NoOfTestParts
THEN
	CTR:=0;
	gTakeTestParts:=FALSE;
	gTakeTestPartsAuto:=FALSE;
	TestPartsRemove:=TRUE;
ELSIF
	 CTR2 = MP.ST02.NoOfDummys THEN
	CTR2:=0;
	MP.ST02.DummyPruefung_93pol:= FALSE;
END_IF
END_ACTION

ACTION Robot01_POS32__action:
Robot01.PosNo:=POS_WT_POS1_WAIT;
Robot01.PosOffset:=gRobotOffset;
Robot01.Override:=MP.ST00.Override;
Robot01.SetToolOn:=FALSE;
Robot01.SetToolOff:=FALSE;
Robot01.ExecuteMove:=TRUE;
END_ACTION

ACTION Robot01_Pos31_action:
Robot01.PosNo:=POS_WT_POS1;
Robot01.PosOffset:=gRobotOffset;
Robot01.Override:=MP.ST00.Override;
Robot01.SetToolOn:=FALSE;
Robot01.SetToolOff:=TRUE;
Robot01.ExecuteMove:=TRUE;
END_ACTION

ACTION Robot01_Pos31_exit:
gRob01GripState:=PART_NEW;
END_ACTION

ACTION Robot01_POS22_action:
Robot01.PosNo:=POS_RT_WAIT;
Robot01.PosOffset:=gRobotOffset;
Robot01.Override:=MP.ST00.Override;
Robot01.SetToolOn:=FALSE;
Robot01.SetToolOff:=FALSE;
Robot01.ExecuteMove:=TRUE;
END_ACTION

ACTION Handshake_entry:
Nest_Empty:=TRUE;
END_ACTION

ACTION Handshake_exit:
Nest_Empty:=FALSE;
END_ACTION

ACTION Robot01_Pos21__action:
Robot01.PosNo:=POS_RT;
Robot01.PosOffset:=gRobotOffset;
Robot01.Override:=MP.ST00.Override;
Robot01.SetToolOn:=TRUE;
Robot01.SetToolOff:=FALSE;
Robot01.ExecuteMove:=TRUE;
END_ACTION

ACTION Robot01_Pos21__exit:
gRob01GripState:=PART_NO;
gRTState[1]:=PART_NEW;
END_ACTION

ACTION set_PartState__exit:
MP.ST02.TableData[1].ProcessData.Part:= TRUE; 		 (* Schnittstelle Tampondrucker Nest 1 leer *)
MP.ST02.TableData[1].ProcessData.Result:=0;	(*   0 = Teil noch nicht bearbeitet *)
											(*   1 =  Oberseite OK*)
											(*  11 = Oberseite und Unterseite OK*)
											(*  99 = Teil ist NOK	*)
END_ACTION

ACTION Robot01_POS23__action:
Robot01.PosNo:=23;
Robot01.PosOffset:=gRobotOffset;
Robot01.Override:=MP.ST00.Override;
Robot01.SetToolOn:=FALSE;
Robot01.SetToolOff:=FALSE;
Robot01.ExecuteMove:=TRUE;
END_ACTION

ACTION ST02_Main_Print__action:
IF 	ST02_Main.State=STATE_WAIT THEN
	ST02_Main.Start:=TRUE;
END_IF
END_ACTION

ACTION ST02_Main_Print__exit:
ST02_Main.Start:=FALSE;
END_ACTION

ACTION Wait_Printer_finish__entry:
ProcessMessage01:='';
Delay.IN:=FALSE;
Delay();
END_ACTION

ACTION Wait_Printer_finish__action:
ProcessMessage01:='1IM23';(*warte auf Druck fertig*)
Delay.IN:=TRUE;

IF MP.ST00.Override >0 AND gTipImp THEN
	DElay.PT:=t#4000s / MP.ST00.Override;
ELSE
	DElay.PT:=t#1h;
END_IF

Delay();
END_ACTION

ACTION Wait_Printer_finish__exit:
ProcessMessage01:='';
END_ACTION

ACTION Open_Stopper3_action:
ST00_74_Y2_4.MoveWork:=TRUE;
END_ACTION

ACTION Msg_Error___entry:
MessageHandler.ClearMessageLines(sVisu:=Visu.Message);
END_ACTION

ACTION Msg_Error___action:
MessageHandler.Msg.ID:='PM115';
MessageHandler.Msg.Name:='Drucker';
MessageHandler.Msg.Text:='Kein Betriebsbereit vom Drucker ';
MessageHandler.Msg.Color:=Color.Red;
MessageHandler.Msg.Station:=1;


MessageHandler(
	Prio:=2, 									(*1=highest, .. , 4=lowest*)
	Btn1Addr:=ADR(MsgOk),			(*Address of Button1 , if Zero then Button is unvisible*)
	Btn2Addr:=0,	(*Address of Button2 , if Zero then Button is unvisible*)
	sVisu:=Visu.Message);
END_ACTION

ACTION Msg_Error___exit:
MessageHandler.ClearMessageLines(sVisu:=Visu.Message);
MsgOk:=FALSE;
END_ACTION

ACTION Close_Stopper44_action:
ST00_74_Y2_4.MoveInit:=TRUE;
END_ACTION

ACTION Fertig_entry:
gRTState[1]:=gRTState[2];
gRTState[2]:=PART_OK;
END_ACTION

ACTION Robot01_Pos1__1__action:
Robot01.PosNo:=POS_PARK;
Robot01.PosOffset:=gRobotOffset;
Robot01.Override:=MP.ST00.Override;
(*Robot01.SetToolOn:=TRUE;
Robot01.SetToolOff:=FALSE;*)
Robot01.ExecuteMove:=TRUE;
END_ACTION

ACTION Robot01_Pos1__1__exit:
ST08_Process.Start:=FALSE;
END_ACTION

ACTION SeqEnd_action:
SFCTime:=TIME_TO_DINT(TIME()-SFCTimeStart);
State:=STATE_WAIT;
END_ACTION

TRANSITION CheckPartsInRoboGripper:
TD.PartsInRoboGripper > 0 (*Diffision durch 0 verhindern*)
END_TRANSITION

TRANSITION StateOk:
ST08_Process.State=STATE_OK
END_TRANSITION

TRANSITION No_Part:
gRob01GripState=PART_NO
END_TRANSITION

TRANSITION Part_OK_:
gRob01GripState = PART_OK AND
((NOT MP.ST08.TrayAushebenMotor AND ST08_406_B54_4.ValveSensor) OR	(* Ausheber Trays Entnahmepos. Isok. STN8 AST *)
(MP.ST08.TrayAushebenMotor AND ABS(ST08_190_M1.sPos.ist - TD.PosTrayAusheben[2].Pos) < 0.5)) (*1=unten, 2=oben, *)
END_TRANSITION

TRANSITION StateOK:
Robot01.State=STATE_OK
END_TRANSITION

TRANSITION StateOk:
ST08_Process.State=STATE_OK
END_TRANSITION

TRANSITION #StateOK:
Robot01.State=STATE_OK

AND gTipImp
END_TRANSITION

TRANSITION Part_New:
gRob01GripState=PART_NEW AND
gTypeCode=312
END_TRANSITION

TRANSITION Part_Cam:
gRob01GripState=PART_CAM (*Teil im Greifer ohne Kameraprüfung*)
END_TRANSITION

TRANSITION RT_Nest_empty:
     (ST02_DT_65B11.BitInToCheck      (* Tampondrucker Nest 1 leer *)
 	 AND ST02_DT_62_B91.ValveSensor )	     (* Tampondrucker Nest 1 in Abholposition *)

OR
	   (ST02_DT_65B21.BitInToCheck  		 (* Tampondrucker Nest 2 leer *)
  AND ST02_DT_62_B81.ValveSensor )     (* Tampondrucker Nest 2 in Abholposition *)
END_TRANSITION

TRANSITION #StateOK:
Robot01.State=STATE_OK

AND gTipImp
END_TRANSITION

TRANSITION all_other:
(gTypeCode<>4991 AND	(*102 pol*)
 gTypeCode<>312) 		(*93 pol*)
END_TRANSITION

TRANSITION 93-102polig:
(gTypeCode=4991 OR 	(*102 pol*)
 gTypeCode=312) 	(*93 pol*)

AND
(ST02_DT_62_B81.ValveSensor OR	(* Tampondrucker Nest 1 in Abholposition *)
 ST02_DT_62_B91.ValveSensor )		(* Tampondrucker Nest 2 in Abholposition *)
END_TRANSITION

TRANSITION Printer_off:
NOT ST02_DT_62_B81.ValveSensor	 AND	     (* Tampondrucker Nest 1 in Abholposition *)
NOT ST02_DT_62_B91.ValveSensor 		     (* Tampondrucker Nest 2 in Abholposition *)
END_TRANSITION

TRANSITION StateOk:
ST00_74_Y2_4.State=STATE_OK
END_TRANSITION

TRANSITION StateOk:
ST00_74_Y2_5.State=STATE_OK
END_TRANSITION

TRANSITION Finish:
	ST00_72_X1_8.BitInToCheck (* Schnittstelle Tampondrucker Druck abgeschlossen *)
END_TRANSITION

TRANSITION StateOk:
ST00_74_Y2_4.State=STATE_OK
END_TRANSITION

TRANSITION 93_102polig:
(*mit Tampondrucker*)
gTypeCode=4991 OR 	(*102 pol*)
gTypeCode=312		(*93 pol*)
END_TRANSITION

TRANSITION 268pol:
gTypeCode=5841 (* AND 	(*268 pol*)
ST03_8_100_A1.Activated*)
END_TRANSITION

TRANSITION CamDone:
(gRob01GripState=PART_OK OR
gRob01GripState=PART_NOK) AND
ST03_268pol_Zufuehrung.State=STATE_WAIT
END_TRANSITION

TRANSITION 102pol_neu:
gTypeCode=4993 (*  AND 	(*102 pol neu*)
ST03_8_100_A1.Activated*)
END_TRANSITION

TRANSITION CamDone:
(gRob01GripState=PART_OK OR
gRob01GripState=PART_NOK) AND
ST03_102pol_neu_Zufuehrung.State=STATE_WAIT
END_TRANSITION

TRANSITION all_other_polig:
(*Tampondrucker*)
(gTypeCode<>4991 AND(*102 pol*)
gTypeCode<>312) AND	(*93 pol*)

(*alte Rüstsätze*)
gTypeCode<>360  AND	(*74pol*)
(*gTypeCode<>379  AND*)	(*91pol*)
gTypeCode<>4992 AND	(*35pol*)
gTypeCode<>489		(*168pol*)
END_TRANSITION

TRANSITION Part_Ready_Pick:
Delay.Q
END_TRANSITION

TRANSITION AutoStop:
		ModeSelect.Mode=MODE_AUTO_STOP
OR	ModeSelect.Mode=MODE_STEP_STOP
END_TRANSITION

TRANSITION POS_1:
ST03_Init_AbholPos.RoboPos31
END_TRANSITION

TRANSITION POS_2:
ST03_Init_AbholPos.RoboPos35
END_TRANSITION

TRANSITION #StateOK:
Robot01.State=STATE_OK

AND gTipImp
END_TRANSITION

TRANSITION #StateOK:
Robot01.State=STATE_OK

AND gTipImp
END_TRANSITION

TRANSITION Yes:
(
gTakeTestParts OR
gTakeTestPartsAuto)
AND
NOT TD.TestpartBilister AND
gRob01GripState = PART_OK AND
NOT ST03_8_75_B13_5.BitInToCheck
END_TRANSITION

TRANSITION i.O.:
gRob01GripState = PART_OK
END_TRANSITION

TRANSITION StateOk:
ST08_Process.State=STATE_OK
OR
gTypeCode=379
END_TRANSITION

TRANSITION StateOk:
Robot01.State=STATE_OK
END_TRANSITION

TRANSITION Pal_OK:
ST08_Process.Pal_Ready AND
NOT ST08_Palletizing.TestpartMoveOut AND
((NOT MP.ST08.TrayAushebenMotor AND ST08_406_B54_4.ValveSensor) OR	(* Ausheber Trays Entnahmepos. Isok. STN8 AST *)
(MP.ST08.TrayAushebenMotor AND ABS(ST08_190_M1.sPos.ist - TD.PosTrayAusheben[2].Pos) < 0.5)) (*1=unten, 2=oben, *)
END_TRANSITION

TRANSITION allOther:
gTypeCode<>379 AND	(*91 pol*)
gTypeCode<>4993		(*102pol neu*)
END_TRANSITION

TRANSITION StateOk:
Robot01.State=STATE_OK
END_TRANSITION

TRANSITION OK:
ST00_71_K2.State=State_OK
END_TRANSITION

TRANSITION StateOk:
ST08_Process.State=STATE_OK OR
ST08_Process.State=STATE_Wait
END_TRANSITION

TRANSITION Pal_OK:
ST08_Process.Pal_Ready AND
NOT ST08_Palletizing.TestpartMoveOut AND
((NOT MP.ST08.TrayAushebenMotor AND ST08_406_B54_4.ValveSensor) OR	(* Ausheber Trays Entnahmepos. Isok. STN8 AST *)
(MP.ST08.TrayAushebenMotor AND ABS(ST08_190_M1.sPos.ist - TD.PosTrayAusheben[2].Pos) < 0.5)) (*1=unten, 2=oben, *)
END_TRANSITION

TRANSITION StateOK:
Robot01.State=STATE_OK
END_TRANSITION

TRANSITION OK:
ST00_71_K2.State=State_OK
END_TRANSITION

TRANSITION StateRun:
ST08_Process.State=STATE_Run OR
gRunEmpty
END_TRANSITION

TRANSITION n.i.O:
gRob01GripState = PART_NOK
END_TRANSITION

TRANSITION #StateOK:
Robot01.State=STATE_OK

AND gTipImp
END_TRANSITION

TRANSITION StateOK:
Robot01.State=STATE_OK
END_TRANSITION

TRANSITION empty:
NOT ST03_8_75_B13_5.BitInToCheck
END_TRANSITION

TRANSITION #StateOK:
Robot01.State=STATE_OK

AND gTipImp
END_TRANSITION

TRANSITION T9_74_168_35polig:
(*alte Rüstsätze*)
gTypeCode=360 OR	(*74pol*)
(*gTypeCode=379 OR*)	(*91pol*)
gTypeCode=4992 OR	(*35pol*)
gTypeCode=489		(*168pol*)
END_TRANSITION

TRANSITION all_other:
NOT MP.ST03.SGM_3621
END_TRANSITION

TRANSITION SGM_3621:
MP.ST03.SGM_3621
END_TRANSITION

TRANSITION leer:
NOT ST03_422_B64_4.BitInToCheck 		 (* Teil auf Abholpos *)
END_TRANSITION

TRANSITION StateOK:
ST03_422_Y64_6.State=STATE_OK
END_TRANSITION

TRANSITION StateOK:
ST03_422_Y64_5.State=STATE_OK
END_TRANSITION

TRANSITION Part_Ready_Print:
Delay.Q
END_TRANSITION

TRANSITION AutoStop:
		ModeSelect.Mode=MODE_AUTO_STOP
OR	ModeSelect.Mode=MODE_STEP_STOP
END_TRANSITION

TRANSITION StateOk:
ST03_422_Y64_5.State=STATE_OK
END_TRANSITION

TRANSITION StateOk:
ST03_422_Y64_6.State=STATE_OK
END_TRANSITION

TRANSITION Part_Ready_Roboter:
Delay.Q
END_TRANSITION

TRANSITION AutoStop:
		ModeSelect.Mode=MODE_AUTO_STOP
OR	ModeSelect.Mode=MODE_STEP_STOP
END_TRANSITION

TRANSITION StateOK:
ST03_422_Y64_6.State=STATE_OK
END_TRANSITION

TRANSITION StateOK:
ST03_422_Y64_5.State=STATE_OK
END_TRANSITION

TRANSITION Abholpos_leer:
NOT ST08_412_B59_0.BitInToCheck 		 (* Teil auf Abholpos *)
END_TRANSITION

TRANSITION StateOk:
ST08_412_Y55_2.State=STATE_OK
END_TRANSITION

TRANSITION StateOk:
ST08_412_Y55_0.State=STATE_OK
END_TRANSITION

TRANSITION Part_Ready_Print:
Delay.Q
END_TRANSITION

TRANSITION AutoStop:
		ModeSelect.Mode=MODE_AUTO_STOP
OR	ModeSelect.Mode=MODE_STEP_STOP
END_TRANSITION

TRANSITION Wait_Pos:
(ST03_51_M1.sPos.ist >
IstPosHelp +TD.DistIso AND MP.ST03.BandMoveP)

OR
(ST03_51_M1.sPos.ist <
IstPosHelp + TD.DistIso AND NOT MP.ST03.BandMoveP)
END_TRANSITION

TRANSITION StateOk:
ST08_412_Y55_0.State=STATE_OK
END_TRANSITION

TRANSITION StateOk:
ST08_412_Y55_2.State=STATE_OK
END_TRANSITION

TRANSITION Part_Ready_Roboter:
Delay.Q
END_TRANSITION

TRANSITION AutoStop:
		ModeSelect.Mode=MODE_AUTO_STOP
OR	ModeSelect.Mode=MODE_STEP_STOP
END_TRANSITION

TRANSITION StateOk:
ST08_412_Y55_2.State=STATE_OK
END_TRANSITION

TRANSITION StateOk:
ST08_412_Y55_0.State=STATE_OK
END_TRANSITION

TRANSITION not_35pol_or_links:
ST03_Init_AbholPos.RoboPos31
END_TRANSITION

TRANSITION 35pol_rechts:
ST03_Init_AbholPos.RoboPos35
END_TRANSITION

TRANSITION #StateOK:
Robot01.State=STATE_OK

AND gTipImp
END_TRANSITION

TRANSITION #StateOK:
Robot01.State=STATE_OK

AND gTipImp
END_TRANSITION

TRANSITION #StateOK:
Robot01.State=STATE_OK

AND gTipImp
END_TRANSITION

TRANSITION Yes:
(gTakeTestParts OR
gTakeTestPartsAuto)
AND
NOT TD.TestpartBilister
AND
NOT ST03_8_75_B13_5.BitInToCheck
END_TRANSITION

TRANSITION No:
gRob01GripState = PART_OK
END_TRANSITION

TRANSITION StateOk:
ST08_Process.State=STATE_OK
END_TRANSITION

TRANSITION StateWait:
ST08_Process.State=STATE_Wait
END_TRANSITION

TRANSITION Pal_OK:
ST08_Process.Pal_Ready
END_TRANSITION

TRANSITION AutoStop:
		ModeSelect.Mode=MODE_AUTO_STOP
OR	ModeSelect.Mode=MODE_STEP_STOP
END_TRANSITION

TRANSITION StateOK:
Robot01.State=STATE_OK
END_TRANSITION

TRANSITION StateRun:
ST08_Process.State=STATE_Run
END_TRANSITION

TRANSITION #StateOK:
Robot01.State=STATE_OK

AND gTipImp
END_TRANSITION

TRANSITION Iso_an_Vereinzler:
ST08_412_B58_7.BitInToCheck 		 (* Schnittstelle Iso auf Übergabeposition *)
OR
 ST03_421_B63_7.BitInToCheck (* für SGM 3621 *)
END_TRANSITION

TRANSITION Trans151:
Robot01.ActualArea <> 4
END_TRANSITION

TRANSITION all_other:
NOT MP.ST03.SGM_3621
END_TRANSITION

TRANSITION SGM_3621:
MP.ST03.SGM_3621
END_TRANSITION

TRANSITION StateOk:
ST03_422_Y64_5.State=STATE_OK
END_TRANSITION

TRANSITION StateOk:
ST03_422_Y64_6.State=STATE_OK
END_TRANSITION

TRANSITION Part_Ready_Roboter:
Delay.Q
END_TRANSITION

TRANSITION StateOK:
ST03_422_Y64_6.State=STATE_OK
END_TRANSITION

TRANSITION StateOK:
ST03_422_Y64_5.State=STATE_OK
END_TRANSITION

TRANSITION StateOk:
ST08_412_Y55_0.State=STATE_OK
END_TRANSITION

TRANSITION StateOk:
ST08_412_Y55_2.State=STATE_OK
END_TRANSITION

TRANSITION Part_Ready_Roboter:
Delay.Q
END_TRANSITION

TRANSITION StateOk:
ST08_412_Y55_2.State=STATE_OK
END_TRANSITION

TRANSITION StateOk:
ST08_412_Y55_0.State=STATE_OK
END_TRANSITION

TRANSITION StateOK:
Robot01.State=STATE_OK
END_TRANSITION

TRANSITION #StateOK:
Robot01.State=STATE_OK

AND gTipImp
END_TRANSITION

TRANSITION Part_Ready_Print:
(NOT ST02_DT_65B11.BitInToCheck AND	(* Tampondrucker Nest 1 leer *)
ST02_DT_61_B51.ValveSensor AND			(* Schwenkarm 1 90 Grad*)
ST02_DT_62_B91.ValveSensor)				(* Tampondrucker Nest 1 in Abholposition 180°*)
OR
(NOT ST02_DT_65B21.BitInToCheck AND	(* Tampondrucker Nest 2 leer *)
ST02_DT_61_B21.ValveSensor AND			(* Schwenkarm 2 90 Grad*)
ST02_DT_62_B81.ValveSensor)			 	(* Tampondrucker Nest 2 in Abholposition 0° *)
END_TRANSITION

TRANSITION RT_Nest_empty:
(ST02_DT_65B11.BitInToCheck AND		(* Tampondrucker Nest 1 leer *)
 ST02_DT_62_B91.ValveSensor)		(* Tampondrucker Nest 1 in Abholposition 180°*)
OR
(ST02_DT_65B21.BitInToCheck AND		(* Tampondrucker Nest 2 leer *)
 ST02_DT_62_B81.ValveSensor ) 		(* Tampondrucker Nest 2 in Abholposition 0°*)
END_TRANSITION

TRANSITION Wait_:
ST02_Main.State=State_WAIT
END_TRANSITION

TRANSITION StateOk:
(*SFCRun AND*)
ST02_Main.State=State_WAIT
END_TRANSITION

TRANSITION AutoStop:
(ModeSelect.Mode=MODE_AUTO_STOP OR
ModeSelect.Mode=MODE_STEP_STOP) AND
ST02_Main.State = STATE_WAIT
END_TRANSITION

TRANSITION #StateOK:
Robot01.State=STATE_OK

AND gTipImp
END_TRANSITION

TRANSITION CounterCheck:
MP.ST02.DummyPruefung_93pol OR
 (gRob01GripState = PART_OK
AND
(PutIdx>=AnzahlTeile OR	(*93pol*)
kein_Teil_NOK))
END_TRANSITION

TRANSITION #StateOK:
Robot01.State = STATE_OK

AND gTipImp
END_TRANSITION

TRANSITION Yes:
(gTakeTestParts OR
gTakeTestPartsAuto OR
MP.ST02.DummyPruefung_93pol)
AND
NOT TD.TestpartBilister
END_TRANSITION

TRANSITION No:
NOT MP.ST02.DummyPruefung_93pol
OR
NOT ST03_8_75_B13_5.BitInToCheck
END_TRANSITION

TRANSITION StateOk:
ST08_Process.State=STATE_OK
END_TRANSITION

TRANSITION StateWait:
ST08_Process.State=STATE_Wait
END_TRANSITION

TRANSITION Pal_OK:
ST08_Process.Pal_Ready=TRUE
END_TRANSITION

TRANSITION #StateOK:
Robot01.State=STATE_OK

AND gTipImp
END_TRANSITION

TRANSITION StateOk:
ST08_Process.State=STATE_OK OR ST08_Process.State=STATE_Wait
END_TRANSITION

TRANSITION Pal_OK:
ST08_Process.Pal_Ready=TRUE
END_TRANSITION

TRANSITION StateOK:
Robot01.State=STATE_OK
END_TRANSITION

TRANSITION StateRun:
ST08_Process.State=STATE_Run
END_TRANSITION

TRANSITION Yes:
NOT ST03_8_75_B13_5.SignalIn AND	(*voll/belegt keine Prüfmittel mehr  *)
NOT ST03_8_75_B13_6.SignalIn AND	(* belegt mit 6 Prüfmittel  *)
NOT TestPartsRemove
END_TRANSITION

TRANSITION StateOK:
Robot01.State=STATE_OK
END_TRANSITION

TRANSITION all_other___:
(gTakeTestParts OR
(gTakeTestPartsAuto AND NOT MP.ST02.DummyPruefung_93pol )OR
(MP.ST02.DummyPruefung_93pol AND CTR2 <>5))
AND
NOT TD.TestpartBilister
END_TRANSITION

TRANSITION Last_Dummy:
MP.ST02.DummyPruefung_93pol AND
CTR2 = 5
END_TRANSITION

TRANSITION Part_Ready___:
(NOT ST02_DT_65B11.BitInToCheck AND	(* Tampondrucker Nest 1 leer *)
ST02_DT_61_B51.ValveSensor AND			(* Schwenkarm 1 90 Grad*)
ST02_DT_62_B91.ValveSensor)				(* Tampondrucker Nest 1 in Abholposition 180°*)
OR
(NOT ST02_DT_65B21.BitInToCheck AND	(* Tampondrucker Nest 2 leer *)
ST02_DT_61_B21.ValveSensor AND			(* Schwenkarm 2 90 Grad*)
ST02_DT_62_B81.ValveSensor)			 	(* Tampondrucker Nest 2 in Abholposition 0° *)
END_TRANSITION

TRANSITION #StateOK:
Robot01.State=STATE_OK

AND gTipImp
END_TRANSITION

TRANSITION #StateOK:
Robot01.State=STATE_OK
AND gTipImp
END_TRANSITION

TRANSITION AutoStop:
(ModeSelect.Mode=MODE_AUTO_STOP OR
ModeSelect.Mode=MODE_STEP_STOP) AND
ST02_Main.State = STATE_WAIT
END_TRANSITION

TRANSITION Auto_run:
ModeSelect.Mode<>MODE_AUTO_STOP AND
ModeSelect.Mode<>MODE_STEP_STOP
END_TRANSITION

TRANSITION AutoStop:
ModeSelect.Mode=MODE_AUTO_STOP OR
ModeSelect.Mode=MODE_STEP_STOP
END_TRANSITION

TRANSITION PartReady:
ST03_102pol_Zufuehrung.PartReady
END_TRANSITION

TRANSITION #StateOK:
Robot01.State=STATE_OK

AND gTipImp
END_TRANSITION

TRANSITION #StateOK:
Robot01.State=STATE_OK

AND gTipImp
END_TRANSITION

TRANSITION OK:
NOT ST03_102pol_Zufuehrung.PartReady
END_TRANSITION

TRANSITION AutoStop:
(ModeSelect.Mode=MODE_AUTO_STOP OR
ModeSelect.Mode=MODE_STEP_STOP) AND
ST02_Main.State = STATE_WAIT
END_TRANSITION

TRANSITION Part_Ready_Print:
  ( ST02_DT_65B11.BitInToCheck AND     (* Tampondrucker Nest 1 leer *)
ST02_DT_61_B51.ValveSensor AND		(* Schwenkarm 1 90 Grad*)
ST02_DT_62_B91.ValveSensor)  		(* Tampondrucker Nest 1 in Abholposition *)
OR
  ( ST02_DT_65B21.BitInToCheck AND  	(* Tampondrucker Nest 2 leer *)
ST02_DT_61_B21.ValveSensor AND		(* Schwenkarm 2 90 Grad*)
ST02_DT_62_B81.ValveSensor ) 		(* Tampondrucker Nest 2 in Abholposition *)
END_TRANSITION

TRANSITION AutoStop:
(ModeSelect.Mode=MODE_AUTO_STOP OR
ModeSelect.Mode=MODE_STEP_STOP) AND
ST02_Main.State = STATE_WAIT
END_TRANSITION

TRANSITION #StateOK:
Robot01.State=STATE_OK

AND gTipImp
END_TRANSITION

TRANSITION #StateOK:
Robot01.State=STATE_OK

AND gTipImp
END_TRANSITION

TRANSITION ST02Wait:
ST02_Main.State=STATE_WAIT
END_TRANSITION

TRANSITION turn_done:
ST02_Main.turn_done
END_TRANSITION

TRANSITION IO:
ST02_Main.turn_done
AND
MP.ST02.TableData[1].ProcessData.	Result =11
											(*   0 = Teil noch nicht bearbeitet *)
											(*   1 =  Oberseite OK*)
											(*  11 = Oberseite und Unterseite OK*)
											(*  99 = Teil ist NOK	*)
END_TRANSITION

TRANSITION NIO:
ST02_Main.turn_done
AND

MP.ST02.TableData[1].ProcessData.	Result <>11
AND

((ST02_DT_65B11.BitInToCheck=FALSE AND     (* Tampondrucker Nest 1 leer *)
ST02_DT_62_B91.ValveSensor)  		(* Tampondrucker Nest 1 in Abholposition *)(*180 Grad*)
OR
(ST02_DT_65B21.BitInToCheck=FALSE AND  	(* Tampondrucker Nest 2 leer *)
ST02_DT_62_B81.ValveSensor )) 		(* Tampondrucker Nest 2 in Abholposition *)(*0 Grad*)
END_TRANSITION

TRANSITION emty:
(ST02_DT_62_B91.ValveSensor AND	(* Tampondrucker Nest 1 in Abholposition *) (*180 Grad*)
 ST02_DT_65B11.BitInToCheck)     		(* Tampondrucker Nest 1 leer *)

OR
(ST02_DT_62_B81.ValveSensor AND 	(* Tampondrucker Nest 2 in Abholposition *)(*0 Grad*)
 ST02_DT_65B21.BitInToCheck) 		 (* Tampondrucker Nest 2 leer *)
END_TRANSITION

TRANSITION Time_out:
Delay.Q
END_TRANSITION

TRANSITION StateOk:
ST00_74_Y2_4.State=STATE_OK
END_TRANSITION

TRANSITION Finish:
 MsgOk
END_TRANSITION

TRANSITION StateOk:
ST00_74_Y2_4.State=STATE_OK
END_TRANSITION

TRANSITION AutoStop:
(ModeSelect.Mode=MODE_AUTO_STOP OR
ModeSelect.Mode=MODE_STEP_STOP) AND
ST02_Main.State = STATE_WAIT
END_TRANSITION

TRANSITION AutoRun:
ModeSelect.Mode=MODE_AUTO_RUN OR
ModeSelect.Mode=MODE_STEP_RUN
	OR (SpecialMode06.State=State_Run AND
		(gTypeCode=312 OR			(*93pol*)
		gTypeCode=499 OR				(*102pol*)
		gTypeCode=322))				(*160pol*)
END_TRANSITION

TRANSITION AutoStop:
(ModeSelect.Mode=MODE_AUTO_STOP OR
ModeSelect.Mode=MODE_STEP_STOP) AND
ST02_Main.State = STATE_WAIT
END_TRANSITION

TRANSITION #StateOK:
    Robot01.State=STATE_OK
AND gTipImp
END_TRANSITION
END_PROGRAM

(* POU zLibrary/ept/Funktionen/FB_CurrentStepHistorie, ST *)
FUNCTION_BLOCK FB_CurrentStepHistorie
VAR_INPUT
	st_CurrentStep	:STRING(20);
END_VAR

VAR
	arr_last_step_history 		:ARRAY[0..maxNumberOfPuffer] OF STRING;
	fb_Time					:TON;
	st_Time					:STRING;
	st_CurrentStepCopy		:STRING;
END_VAR
VAR_TEMP
	i					:INT;
END_VAR
VAR CONSTANT
	maxNumberOfPuffer			: INT:=30;
END_VAR
(*======================================================
   PRG: ST_CurrentStepHistorie
 ------------------------------------------------------
   Auth: 		Werner Friedl    						 
   Date: 		1.6.2015    						     
   Rev.: 		1.0	
   Desc:		Ablauf wird in einer Historie aufgezeichnet
   Historie:   1.0

	Beispiel eines Aufrufs:
	ST02_Nest05.FB_CurrentStepHistorie(st_CurrentStep:=ST02_Nest05.SFCCurrentStep);
 ========================================================*)

fb_Time();

IF st_CurrentStep<>st_CurrentStepCopy THEN
	fb_Time(IN:=FALSE);
	FOR i:=maxNumberOfPuffer TO 1  BY -1 DO
			arr_last_step_history[i] :=arr_last_step_history[i-1];
	END_FOR
	st_CurrentStepCopy:=st_CurrentStep;
	fb_Time(IN:=TRUE,PT:=t#100m);
END_IF
st_Time:=TIME_TO_STRING(fb_Time.ET);
st_Time:=DELETE(st_Time,2,1);
st_Time:=CONCAT(st_Time,': ');
arr_last_step_history[0]:=CONCAT(st_Time,st_CurrentStep);
END_FUNCTION_BLOCK

(* POU Stations/ST_00/ST00_SFCs/_SpecialModeSFCs/SpecialMode06, SFC *)
PROGRAM SpecialMode06 (*Used for: Dummytestprogramm*)
(* Date: 06.03.2019    Author: Rid Tobias   *)

VAR_OUTPUT
	SFCCurrentPOU		: STRING:='SpecialMode06';
	SFCCurrentStep		: STRING:='';
	SFCTime			: DINT;
 	State   				: DINT;
  	Result  				: DINT;
END_VAR
VAR_INPUT
	Start					: BOOL;

END_VAR
VAR

	MsgOK				: BOOL;
	MsgCancel			: BOOL;
	SFCRun				: BOOL;
	SFCTimeStart		: TIME;
  	LoopCounter   		: DINT;	(* aktuelle Dummynummer *)
	Delay				: TON;
	(*PartOk				: BOOL;	(* Ergebnisvariable für aktuelles *)*)
  	Dummy_ResOK		: BOOL;	(* Ergebnisvariable für den kompletten Dummytest *)
 	i           				: DINT;
  	NokMsgString		: STRING(255);
	startBand			:BOOL;
	NokMsgString1		 : STRING;

	StartErlaubt93pol			:BOOL;
	(* Userdefinded area *)

END_VAR
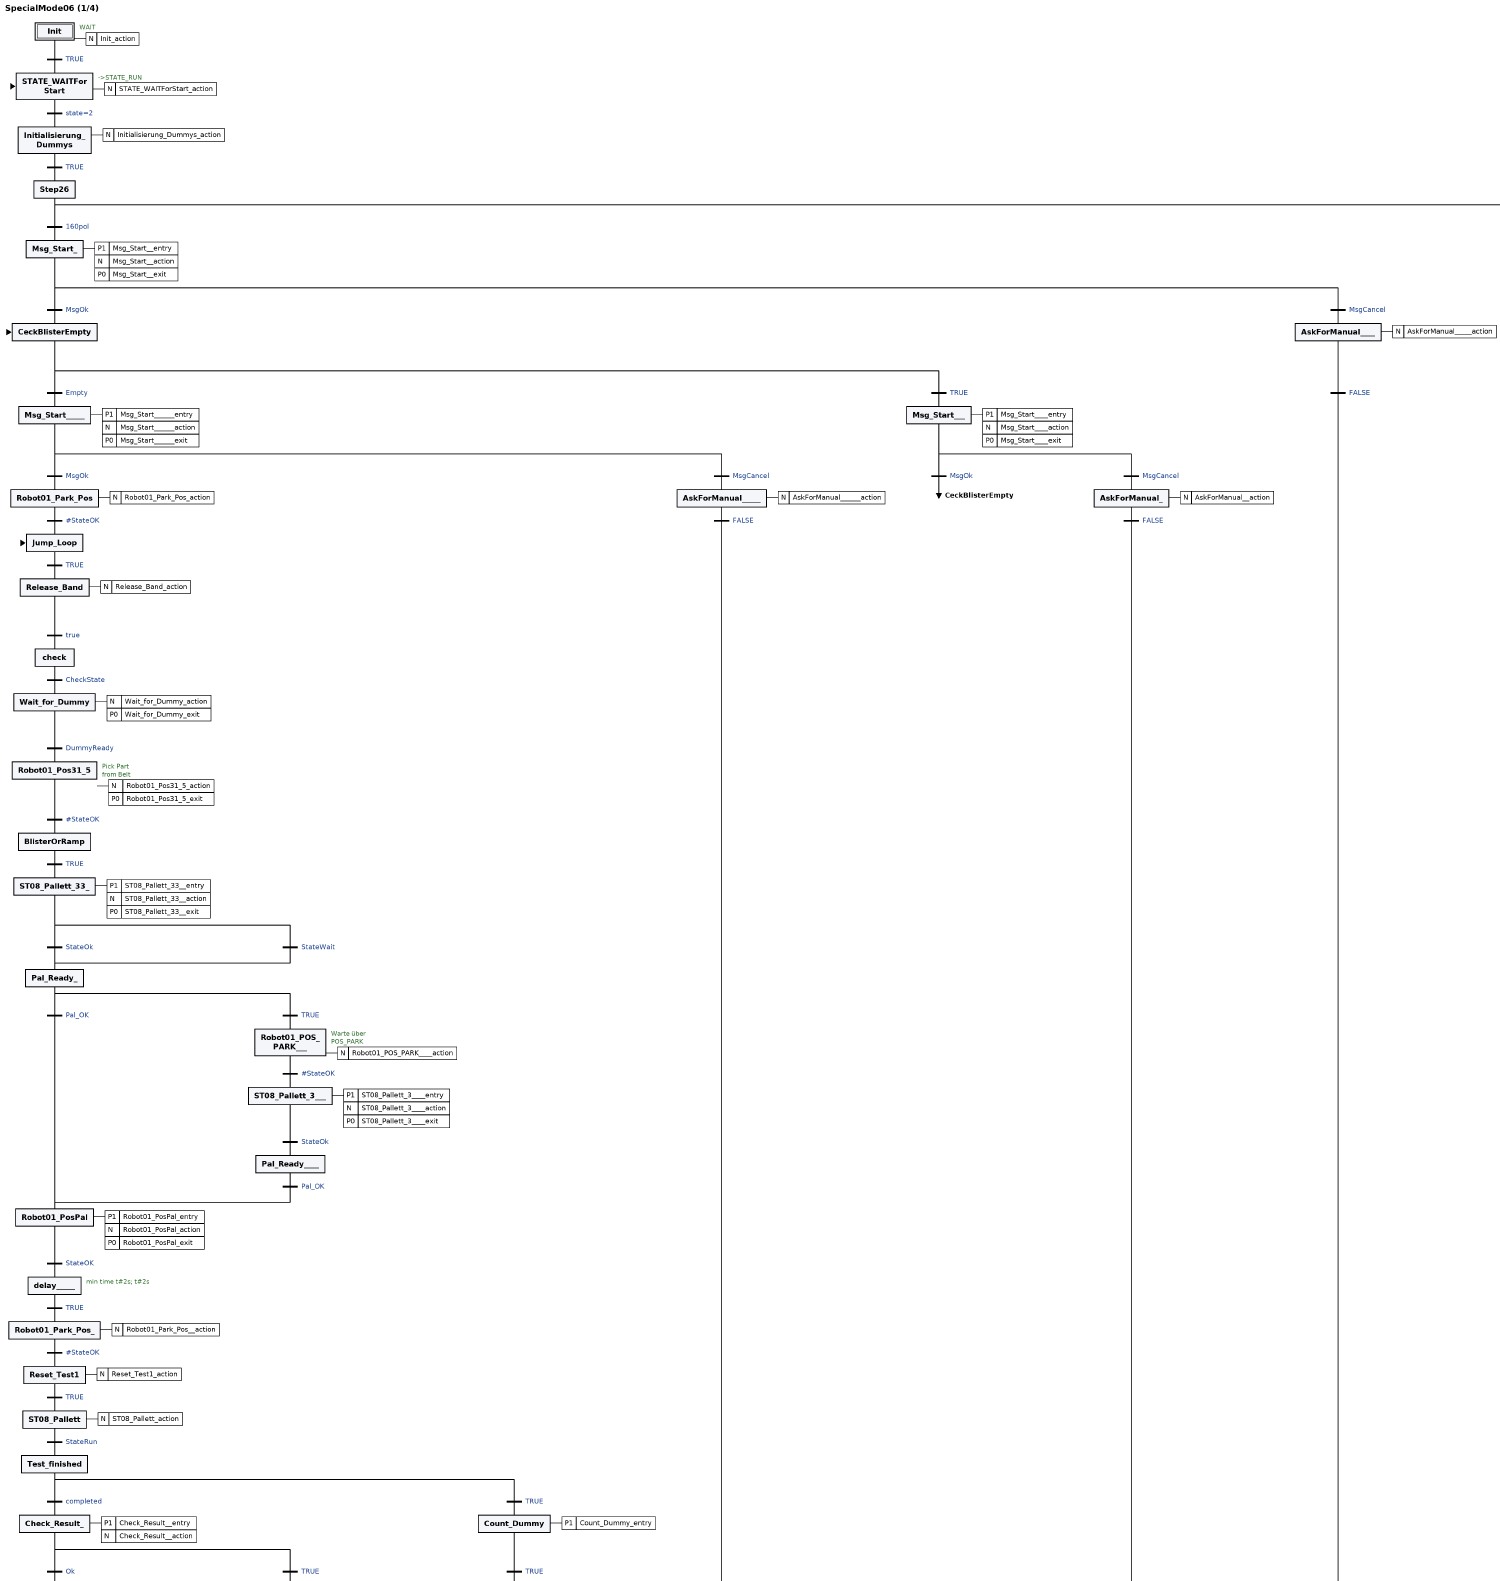
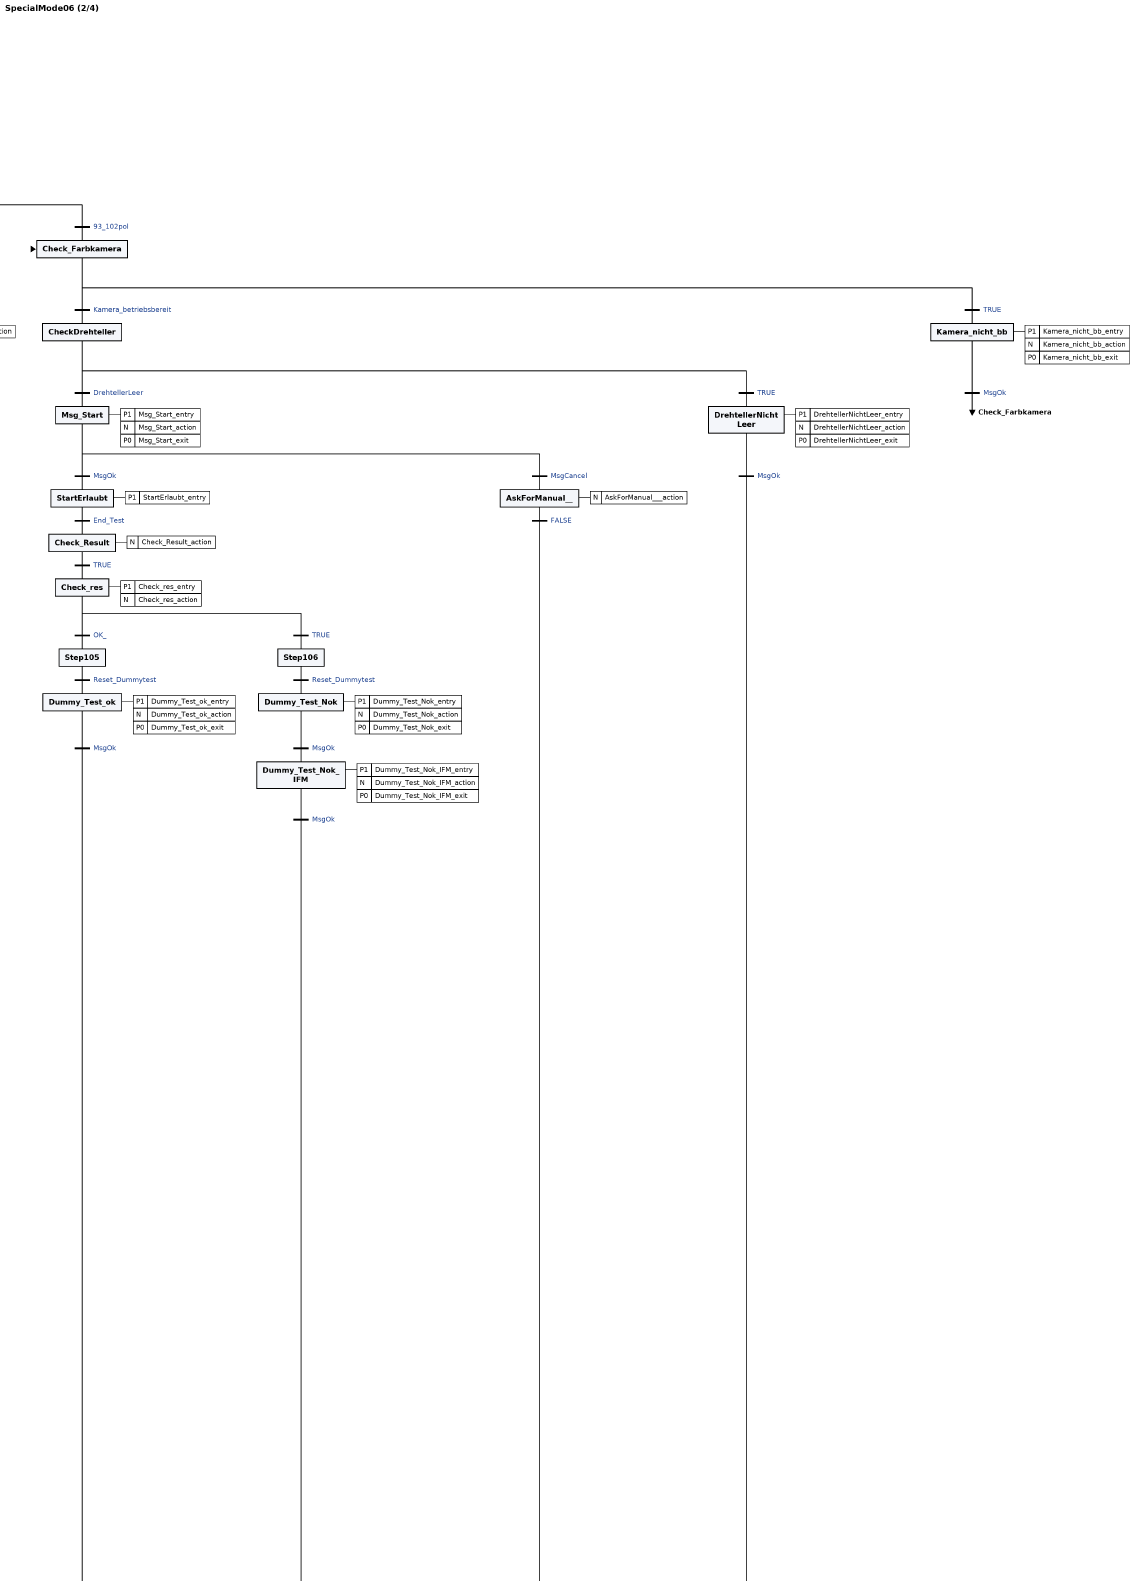
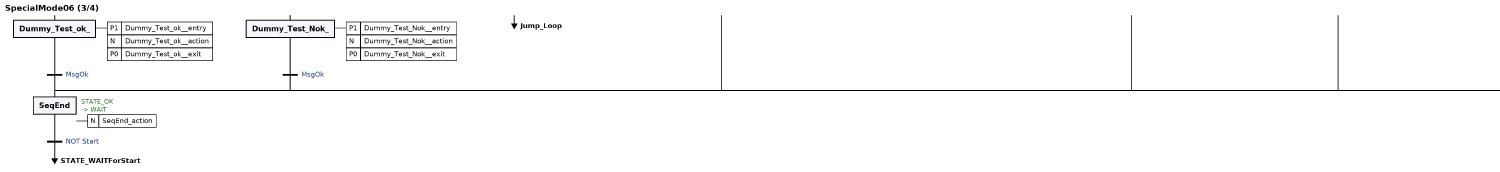
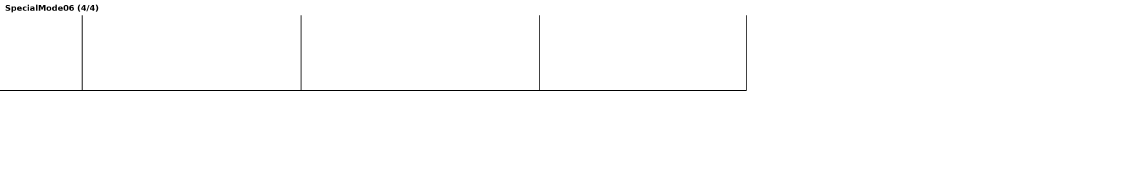
INITIAL_STEP Init: (* WAIT *)
	Init_action(N);
END_STEP
TRANSITION FROM Init TO STATE_WAITForStart := TRUE;
END_TRANSITION
STEP STATE_WAITForStart: (* ->STATE_RUN *)
	STATE_WAITForStart_action(N);
END_STEP
TRANSITION FROM STATE_WAITForStart TO Initialisierung_Dummys := state=2;
END_TRANSITION
STEP Initialisierung_Dummys:
	Initialisierung_Dummys_action(N);
END_STEP
TRANSITION FROM Initialisierung_Dummys TO Step26 := TRUE;
END_TRANSITION
STEP Step26:
END_STEP
TRANSITION FROM Step26 TO Msg_Start_ := 160pol;
END_TRANSITION
TRANSITION FROM Step26 TO Check_Farbkamera := 93_102pol;
END_TRANSITION
STEP Msg_Start_:
	Msg_Start__entry(P1);
	Msg_Start__action(N);
	Msg_Start__exit(P0);
END_STEP
TRANSITION FROM Msg_Start_ TO CeckBlisterEmpty := MsgOk;
END_TRANSITION
TRANSITION FROM Msg_Start_ TO AskForManual____ := MsgCancel;
END_TRANSITION
STEP CeckBlisterEmpty:
END_STEP
TRANSITION FROM CeckBlisterEmpty TO Msg_Start_____ := Empty;
END_TRANSITION
TRANSITION FROM CeckBlisterEmpty TO Msg_Start___ := TRUE;
END_TRANSITION
STEP Msg_Start___:
	Msg_Start____entry(P1);
	Msg_Start____action(N);
	Msg_Start____exit(P0);
END_STEP
TRANSITION FROM Msg_Start___ TO CeckBlisterEmpty := MsgOk;
END_TRANSITION
TRANSITION FROM Msg_Start___ TO AskForManual_ := MsgCancel;
END_TRANSITION
STEP AskForManual_:
	AskForManual__action(N);
END_STEP
TRANSITION FROM AskForManual_ TO SeqEnd := FALSE;
END_TRANSITION
STEP AskForManual____:
	AskForManual_____action(N);
END_STEP
TRANSITION FROM AskForManual____ TO SeqEnd := FALSE;
END_TRANSITION
STEP Msg_Start_____:
	Msg_Start______entry(P1);
	Msg_Start______action(N);
	Msg_Start______exit(P0);
END_STEP
TRANSITION FROM Msg_Start_____ TO Robot01_Park_Pos := MsgOk;
END_TRANSITION
TRANSITION FROM Msg_Start_____ TO AskForManual_____ := MsgCancel;
END_TRANSITION
STEP AskForManual_____:
	AskForManual______action(N);
END_STEP
TRANSITION FROM AskForManual_____ TO SeqEnd := FALSE;
END_TRANSITION
STEP Robot01_Park_Pos:
	Robot01_Park_Pos_action(N);
END_STEP
TRANSITION FROM Robot01_Park_Pos TO Jump_Loop := #StateOK;
END_TRANSITION
STEP Check_Farbkamera:
END_STEP
TRANSITION FROM Check_Farbkamera TO CheckDrehteller := Kamera_betriebsbereit;
END_TRANSITION
TRANSITION FROM Check_Farbkamera TO Kamera_nicht_bb := TRUE;
END_TRANSITION
STEP CheckDrehteller:
END_STEP
TRANSITION FROM CheckDrehteller TO Msg_Start := DrehtellerLeer;
END_TRANSITION
TRANSITION FROM CheckDrehteller TO DrehtellerNichtLeer := TRUE;
END_TRANSITION
STEP DrehtellerNichtLeer:
	DrehtellerNichtLeer_entry(P1);
	DrehtellerNichtLeer_action(N);
	DrehtellerNichtLeer_exit(P0);
END_STEP
TRANSITION FROM DrehtellerNichtLeer TO SeqEnd := MsgOk;
END_TRANSITION
STEP Kamera_nicht_bb:
	Kamera_nicht_bb_entry(P1);
	Kamera_nicht_bb_action(N);
	Kamera_nicht_bb_exit(P0);
END_STEP
TRANSITION FROM Kamera_nicht_bb TO Check_Farbkamera := MsgOk;
END_TRANSITION
STEP Msg_Start:
	Msg_Start_entry(P1);
	Msg_Start_action(N);
	Msg_Start_exit(P0);
END_STEP
TRANSITION FROM Msg_Start TO StartErlaubt := MsgOk;
END_TRANSITION
TRANSITION FROM Msg_Start TO AskForManual__ := MsgCancel;
END_TRANSITION
STEP AskForManual__:
	AskForManual___action(N);
END_STEP
TRANSITION FROM AskForManual__ TO SeqEnd := FALSE;
END_TRANSITION
STEP StartErlaubt:
	StartErlaubt_entry(P1);
END_STEP
TRANSITION FROM StartErlaubt TO Check_Result := End_Test;
END_TRANSITION
STEP Check_Result:
	Check_Result_action(N);
END_STEP
TRANSITION FROM Check_Result TO Check_res := TRUE;
END_TRANSITION
STEP Check_res:
	Check_res_entry(P1);
	Check_res_action(N);
END_STEP
TRANSITION FROM Check_res TO Step105 := OK_;
END_TRANSITION
TRANSITION FROM Check_res TO Step106 := TRUE;
END_TRANSITION
STEP Step105:
END_STEP
TRANSITION FROM Step105 TO Dummy_Test_ok := Reset_Dummytest;
END_TRANSITION
STEP Dummy_Test_ok:
	Dummy_Test_ok_entry(P1);
	Dummy_Test_ok_action(N);
	Dummy_Test_ok_exit(P0);
END_STEP
TRANSITION FROM Dummy_Test_ok TO SeqEnd := MsgOk;
END_TRANSITION
STEP Step106:
END_STEP
TRANSITION FROM Step106 TO Dummy_Test_Nok := Reset_Dummytest;
END_TRANSITION
STEP Dummy_Test_Nok:
	Dummy_Test_Nok_entry(P1);
	Dummy_Test_Nok_action(N);
	Dummy_Test_Nok_exit(P0);
END_STEP
TRANSITION FROM Dummy_Test_Nok TO Dummy_Test_Nok_IFM := MsgOk;
END_TRANSITION
STEP Dummy_Test_Nok_IFM:
	Dummy_Test_Nok_IFM_entry(P1);
	Dummy_Test_Nok_IFM_action(N);
	Dummy_Test_Nok_IFM_exit(P0);
END_STEP
TRANSITION FROM Dummy_Test_Nok_IFM TO SeqEnd := MsgOk;
END_TRANSITION
STEP Jump_Loop:
END_STEP
TRANSITION FROM Jump_Loop TO Release_Band := TRUE;
END_TRANSITION
STEP Release_Band:
	Release_Band_action(N);
END_STEP
TRANSITION FROM Release_Band TO check := true;
END_TRANSITION
STEP check:
END_STEP
TRANSITION FROM check TO Wait_for_Dummy := CheckState;
END_TRANSITION
STEP Wait_for_Dummy:
	Wait_for_Dummy_action(N);
	Wait_for_Dummy_exit(P0);
END_STEP
TRANSITION FROM Wait_for_Dummy TO Robot01_Pos31_5 := DummyReady;
END_TRANSITION
STEP Robot01_Pos31_5: (* Pick Part / from Belt *)
	Robot01_Pos31_5_action(N);
	Robot01_Pos31_5_exit(P0);
END_STEP
TRANSITION FROM Robot01_Pos31_5 TO BlisterOrRamp := #StateOK;
END_TRANSITION
STEP BlisterOrRamp:
END_STEP
TRANSITION FROM BlisterOrRamp TO ST08_Pallett_33_ := TRUE;
END_TRANSITION
STEP ST08_Pallett_33_:
	ST08_Pallett_33__entry(P1);
	ST08_Pallett_33__action(N);
	ST08_Pallett_33__exit(P0);
END_STEP
TRANSITION FROM ST08_Pallett_33_ TO Pal_Ready_ := StateOk;
END_TRANSITION
TRANSITION FROM ST08_Pallett_33_ TO Pal_Ready_ := StateWait;
END_TRANSITION
STEP Pal_Ready_:
END_STEP
TRANSITION FROM Pal_Ready_ TO Robot01_PosPal := Pal_OK;
END_TRANSITION
TRANSITION FROM Pal_Ready_ TO Robot01_POS_PARK___ := TRUE;
END_TRANSITION
STEP Robot01_POS_PARK___: (* Warte über / POS_PARK *)
	Robot01_POS_PARK____action(N);
END_STEP
TRANSITION FROM Robot01_POS_PARK___ TO ST08_Pallett_3___ := #StateOK;
END_TRANSITION
STEP ST08_Pallett_3___:
	ST08_Pallett_3____entry(P1);
	ST08_Pallett_3____action(N);
	ST08_Pallett_3____exit(P0);
END_STEP
TRANSITION FROM ST08_Pallett_3___ TO Pal_Ready____ := StateOk;
END_TRANSITION
STEP Pal_Ready____:
END_STEP
TRANSITION FROM Pal_Ready____ TO Robot01_PosPal := Pal_OK;
END_TRANSITION
STEP Robot01_PosPal:
	Robot01_PosPal_entry(P1);
	Robot01_PosPal_action(N);
	Robot01_PosPal_exit(P0);
END_STEP
TRANSITION FROM Robot01_PosPal TO delay_____ := StateOK;
END_TRANSITION
STEP delay_____: (* min time t#2s; t#2s *)
END_STEP
TRANSITION FROM delay_____ TO Robot01_Park_Pos_ := TRUE;
END_TRANSITION
STEP Robot01_Park_Pos_:
	Robot01_Park_Pos__action(N);
END_STEP
TRANSITION FROM Robot01_Park_Pos_ TO Reset_Test1 := #StateOK;
END_TRANSITION
STEP Reset_Test1:
	Reset_Test1_action(N);
END_STEP
TRANSITION FROM Reset_Test1 TO ST08_Pallett := TRUE;
END_TRANSITION
STEP ST08_Pallett:
	ST08_Pallett_action(N);
END_STEP
TRANSITION FROM ST08_Pallett TO Test_finished := StateRun;
END_TRANSITION
STEP Test_finished:
END_STEP
TRANSITION FROM Test_finished TO Check_Result_ := completed;
END_TRANSITION
TRANSITION FROM Test_finished TO Count_Dummy := TRUE;
END_TRANSITION
STEP Count_Dummy:
	Count_Dummy_entry(P1);
END_STEP
TRANSITION FROM Count_Dummy TO Jump_Loop := TRUE;
END_TRANSITION
STEP Check_Result_:
	Check_Result__entry(P1);
	Check_Result__action(N);
END_STEP
TRANSITION FROM Check_Result_ TO Dummy_Test_ok_ := Ok;
END_TRANSITION
TRANSITION FROM Check_Result_ TO Dummy_Test_Nok_ := TRUE;
END_TRANSITION
STEP Dummy_Test_Nok_:
	Dummy_Test_Nok__entry(P1);
	Dummy_Test_Nok__action(N);
	Dummy_Test_Nok__exit(P0);
END_STEP
TRANSITION FROM Dummy_Test_Nok_ TO SeqEnd := MsgOk;
END_TRANSITION
STEP Dummy_Test_ok_:
	Dummy_Test_ok__entry(P1);
	Dummy_Test_ok__action(N);
	Dummy_Test_ok__exit(P0);
END_STEP
TRANSITION FROM Dummy_Test_ok_ TO SeqEnd := MsgOk;
END_TRANSITION
STEP SeqEnd: (* STATE_OK / -> WAIT *)
	SeqEnd_action(N);
END_STEP
TRANSITION FROM SeqEnd TO STATE_WAITForStart := NOT Start;
END_TRANSITION

ACTION Init_action:
Start:=FALSE;
State:=STATE_WAIT;
LoopCounter:=1;
startBand := FALSE;
StartErlaubt93pol:=FALSE;
END_ACTION

ACTION STATE_WAITForStart_action:
IF Start=TRUE
THEN
	State:=STATE_RUN;
	Result:=RESULT_NON;
	SFCTimeStart:=TIME();
(*ELSE*)
END_IF
END_ACTION

ACTION Initialisierung_Dummys_action:
(*Reihenfolge der Dummys für 160 pol.*)
(*		TRUE = Gutteil
   		FALSE = Schlechtteil		*)
Dummy_test_Vorgabe[1] := FALSE;
Dummy_test_Vorgabe[2] := FALSE;
Dummy_test_Vorgabe[3] := FALSE;
Dummy_test_Vorgabe[4] := FALSE;
Dummy_test_Vorgabe[5] := FALSE;
Dummy_test_Vorgabe[6] := FALSE;
END_ACTION

ACTION Msg_Start__entry:
MessageHandler.ClearMessageLines(sVisu:=Visu.Message);
END_ACTION

ACTION Msg_Start__action:
MessageHandler.Msg.ID:='PM59';
MessageHandler.Msg.Name:='Prüfung Dummy/Nio-Teile';
MessageHandler.Msg.Text:='Blister und Band leer räumen und$R$N Teile im Blister auf 0 stellen$R$NJa: Start mit OK$R$NNein: Abbrechen';
MessageHandler.Msg.Color:=Color.yellow;
MessageHandler.Msg.Station:=0;


MessageHandler(
	Prio:=2, 									(*1=highest, .. , 4=lowest*)
	Btn1Addr:=ADR(MsgOk),			(*Address of Button1 , if Zero then Button is unvisible*)
	Btn2Addr:=ADR(MsgCancel),	(*Address of Button2 , if Zero then Button is unvisible*)
	sVisu:=Visu.Message);
END_ACTION

ACTION Msg_Start__exit:
MsgOk:=FALSE;
MsgCancel:=FALSE;
END_ACTION

ACTION Msg_Start____entry:
MessageHandler.ClearMessageLines(sVisu:=Visu.Message);
END_ACTION

ACTION Msg_Start____action:
MessageHandler.Msg.ID:='PM60';
MessageHandler.Msg.Name:='Prüfung Dummy/Nio-Teile';
MessageHandler.Msg.Text:='Blister ist nicht leer, Blister leerräumen 0$R$N und Teile auf Anzahl Teile auf 0 stellen$R$NJa: Start mit OK$R$NNein: Abbrechen';
MessageHandler.Msg.Color:=Color.yellow;
MessageHandler.Msg.Station:=0;


MessageHandler(
	Prio:=2, 									(*1=highest, .. , 4=lowest*)
	Btn1Addr:=ADR(MsgOk),			(*Address of Button1 , if Zero then Button is unvisible*)
	Btn2Addr:=ADR(MsgCancel),	(*Address of Button2 , if Zero then Button is unvisible*)
	sVisu:=Visu.Message);
END_ACTION

ACTION Msg_Start____exit:
MsgOk:=FALSE;
MsgCancel:=FALSE;
END_ACTION

ACTION AskForManual__action:
ModeSelect.AskForManual:=TRUE;
END_ACTION

ACTION AskForManual_____action:
ModeSelect.AskForManual:=TRUE;
END_ACTION

ACTION Msg_Start______entry:
MessageHandler.ClearMessageLines(sVisu:=Visu.Message);
END_ACTION

ACTION Msg_Start______action:
MessageHandler.Msg.ID:='PM57';
MessageHandler.Msg.Name:='Prüfung Dummy/Nio-Teile';
MessageHandler.Msg.Text:='Bitte die 6 Prüfteile nacheinander einlegen$R$NJedes Teil muss mit Ok bestätigt werden$R$NJa: Start mit OK$R$NNein: Abbrechen';
MessageHandler.Msg.Color:=Color.yellow;
MessageHandler.Msg.Station:=0;


MessageHandler(
	Prio:=2, 									(*1=highest, .. , 4=lowest*)
	Btn1Addr:=ADR(MsgOk),			(*Address of Button1 , if Zero then Button is unvisible*)
	Btn2Addr:=ADR(MsgCancel),	(*Address of Button2 , if Zero then Button is unvisible*)
	sVisu:=Visu.Message);
END_ACTION

ACTION Msg_Start______exit:
MsgOk:=FALSE;
MsgCancel:=FALSE;
END_ACTION

ACTION AskForManual______action:
ModeSelect.AskForManual:=TRUE;
END_ACTION

ACTION Robot01_Park_Pos_action:
Robot01.PosNo:=POS_PARK;
Robot01.PosOffset:=gRobotOffset;
Robot01.Override:=MP.ST00.Override;
Robot01.SetToolOn:=TRUE;
Robot01.SetToolOff:=FALSE;
Robot01.ExecuteMove:=TRUE;
END_ACTION

ACTION DrehtellerNichtLeer_entry:
MessageHandler.ClearMessageLines(sVisu:=Visu.Message);
END_ACTION

ACTION DrehtellerNichtLeer_action:
MessageHandler.Msg.ID:='PM63';
MessageHandler.Msg.Name:='Check Drehteller';
MessageHandler.Msg.Text:='Drehteller ist nicht Leer';
MessageHandler.Msg.Color:=Color.red;
MessageHandler.Msg.Station:=1;


MessageHandler(
	Prio:=2, 							(*1=highest, .. , 4=lowest*)
	Btn1Addr:=ADR(MsgOk),			(*Address of Button1 , if Zero then Button is unvisible*)
	Btn2Addr:=,						(*Address of Button2 , if Zero then Button is unvisible*)
	sVisu:=Visu.Message);
END_ACTION

ACTION DrehtellerNichtLeer_exit:
MsgOk:=FALSE;
MsgCancel:=FALSE;
ST02_DT_95_A1.b_quitt:=TRUE;
END_ACTION

ACTION Kamera_nicht_bb_entry:
MessageHandler.ClearMessageLines(sVisu:=Visu.Message);
END_ACTION

ACTION Kamera_nicht_bb_action:
MessageHandler.Msg.ID:='PM62';
MessageHandler.Msg.Name:='Check Camera';
MessageHandler.Msg.Text:='Sesopart Kamera ist nicht betriebsbereit';
MessageHandler.Msg.Color:=Color.red;
MessageHandler.Msg.Station:=1;


MessageHandler(
	Prio:=2, 							(*1=highest, .. , 4=lowest*)
	Btn1Addr:=ADR(MsgOk),			(*Address of Button1 , if Zero then Button is unvisible*)
	Btn2Addr:=,						(*Address of Button2 , if Zero then Button is unvisible*)
	sVisu:=Visu.Message);
END_ACTION

ACTION Kamera_nicht_bb_exit:
MsgOk:=FALSE;
MsgCancel:=FALSE;
ST02_DT_95_A1.b_quitt:=TRUE;
END_ACTION

ACTION Msg_Start_entry:
MessageHandler.ClearMessageLines(sVisu:=Visu.Message);
END_ACTION

ACTION Msg_Start_action:
MessageHandler.Msg.ID:='PM58';
MessageHandler.Msg.Name:='Prüfung Dummy/Nio-Teile';
MessageHandler.Msg.Text:='Bitte Drehteller leer machen dann $R$Ndie 6 Prüfteile nacheinander einlegen$R$NJa: Start mit OK$R$NNein: Abbrechen';
MessageHandler.Msg.Color:=Color.yellow;
MessageHandler.Msg.Station:=0;


MessageHandler(
	Prio:=2, 									(*1=highest, .. , 4=lowest*)
	Btn1Addr:=ADR(MsgOk),			(*Address of Button1 , if Zero then Button is unvisible*)
	Btn2Addr:=ADR(MsgCancel),	(*Address of Button2 , if Zero then Button is unvisible*)
	sVisu:=Visu.Message);
END_ACTION

ACTION Msg_Start_exit:
MsgOk:=FALSE;
MsgCancel:=FALSE;
END_ACTION

ACTION AskForManual___action:
ModeSelect.AskForManual:=TRUE;
END_ACTION

ACTION StartErlaubt_entry:
StartErlaubt93pol:=TRUE;
END_ACTION

ACTION Check_Result_action:
(*Erklärung der Auswertung:
In der Produktion wird  nur OK und NOK ausgwertet:
   0 = Teil noch nicht bearbeitet bzw. Nest leer
   1 =  Druck ist OK
   9 = Druck ist NOK
Bei der Dummyprüfung muss passend zum Dummy rot, blau oder beide NOK sein:
   6= Teil roter und blauer Druck NOK ist nur bei der Dummyprüfung aktiv
   7= Teil roter Druck NOKist nur bei der Dummyprüfung aktiv
   8= Teil blauer Druck NOK ist nur bei der Dummyprüfung aktiv
Lage:	
Ziffer 1 = 90°		Ziffer 2 =180°
*)

(*Dummy1*)
IF ST02_Main.ResultBuffer[6] = 78 THEN
	 Mp.ST02.Dummy_test_Result[1] := TRUE;
ELSE
	 Mp.ST02.Dummy_test_Result[1] := FALSE;
END_IF
(*Dummy2*)
IF ST02_Main.ResultBuffer[5] = 11 THEN
	 Mp.ST02.Dummy_test_Result[2] :=  TRUE;
ELSE
	 Mp.ST02.Dummy_test_Result[2] := FALSE;
END_IF
(*Dummy3*)
IF ST02_Main.ResultBuffer[4] = 16 THEN
	 Mp.ST02.Dummy_test_Result[3] :=  TRUE;
ELSE
	 Mp.ST02.Dummy_test_Result[3] := FALSE;
END_IF
(*Dummy4*)
IF ST02_Main.ResultBuffer[3] = 66 THEN
	 Mp.ST02.Dummy_test_Result[4] :=  TRUE;
ELSE
	 Mp.ST02.Dummy_test_Result[4] := FALSE;
END_IF
(*Dummy5*)
IF ST02_Main.ResultBuffer[2] = 66 THEN
	 Mp.ST02.Dummy_test_Result[5] :=  TRUE;
ELSE
	 Mp.ST02.Dummy_test_Result[5] := FALSE;
END_IF
(*Dummy6*)
IF ST02_Main.ResultBuffer[1] = 11 THEN
	 Mp.ST02.Dummy_test_Result[6] := TRUE;
ELSE
	 Mp.ST02.Dummy_test_Result[6] := FALSE;
END_IF


(*IFM Flügelerkennung*)
IF ST03_102pol_Zufuehrung.ResultBufferIFM[6] = TRUE THEN
	  Mp.ST02.Dummy_test_Result[7]  := TRUE;
ELSE
	 Mp.ST02.Dummy_test_Result[7] := FALSE;
END_IF

IF ST03_102pol_Zufuehrung.ResultBufferIFM[5] = TRUE THEN
	 Mp.ST02.Dummy_test_Result[8] :=  TRUE;
ELSE
	 Mp.ST02.Dummy_test_Result[8] := FALSE;
END_IF


IF ST03_102pol_Zufuehrung.ResultBufferIFM[4] = FALSE THEN
	 Mp.ST02.Dummy_test_Result[9] :=  TRUE;
ELSE
	 Mp.ST02.Dummy_test_Result[9] := FALSE;
END_IF


IF ST03_102pol_Zufuehrung.ResultBufferIFM[3] = FALSE THEN
	 Mp.ST02.Dummy_test_Result[10] :=  TRUE;
ELSE
	 Mp.ST02.Dummy_test_Result[10] := FALSE;
END_IF


IF ST03_102pol_Zufuehrung.ResultBufferIFM[2] = TRUE THEN
	 Mp.ST02.Dummy_test_Result[11] :=  TRUE;
ELSE
	 Mp.ST02.Dummy_test_Result[11] := FALSE;
END_IF


IF ST03_102pol_Zufuehrung.ResultBufferIFM[1] = FALSE THEN
	 Mp.ST02.Dummy_test_Result[12] := TRUE;
ELSE
	 Mp.ST02.Dummy_test_Result[12] := FALSE;
END_IF
END_ACTION

ACTION Check_res_entry:
Dummy_ResOK:=TRUE;
END_ACTION

ACTION Check_res_action:
FOR i:=1 TO 12
	DO
	  IF Mp.ST02.Dummy_test_Result[i] = FALSE
	  THEN
	     Dummy_ResOK:=FALSE;
	  END_IF
END_FOR
END_ACTION

ACTION Dummy_Test_ok_entry:
MessageHandler.ClearMessageLines(sVisu:=Visu.Message);
MsgOk:=FALSE;
END_ACTION

ACTION Dummy_Test_ok_action:
MessageHandler.Msg.ID:='PM54';
MessageHandler.Msg.Name:='DummyTest';
MessageHandler.Msg.Text:=' Dummy Pruefung OK, Ergebnis aller Teile OK ';
MessageHandler.Msg.Color:=Color.green;
MessageHandler.Msg.Station:=1;


MessageHandler(
	Prio:=2, 								(*1=highest, .. , 4=lowest*)
	Btn1Addr:=ADR(MsgOk),						(*Address of Button1 , if Zero then Button is unvisible*)
	Btn2Addr:=0,						(*Address of Button2 , if Zero then Button is unvisible*)
	sVisu:=Visu.Message);
END_ACTION

ACTION Dummy_Test_ok_exit:
MessageHandler.ClearMessageLines(sVisu:=Visu.Message);
MsgOk:=FALSE;
END_ACTION

ACTION Dummy_Test_Nok_entry:
MessageHandler.ClearMessageLines(sVisu:=Visu.Message);
MsgOk:=FALSE;
END_ACTION

ACTION Dummy_Test_Nok_action:
NokMsgString:='';
NokMsgString1:='';

MessageHandler.Msg.ID:='PM55';
MessageHandler.Msg.Name:='Sensopart Dummyprüfung NOK';
MessageHandler.Msg.Text:=CONCAT(NokMsgString,'$N$R');
MessageHandler.Msg.Text:=CONCAT(MessageHandler.Msg.Text,NokMsgString1);
MessageHandler.Msg.Color:=Color.red;
MessageHandler.Msg.Station:=2;

FOR i:= 1 TO 6 BY 1 DO
	MessageHandler.MessageLine[i].MsgTypeEnum:=MsgDataTypeString;
	MessageHandler.MessageLine[i].Text:=CONCAT('Dummy_',DINT_TO_STRING(i));
	IF Mp.ST02.Dummy_test_Result[i] THEN
		MessageHandler.MessageLine[i].MsgString:='OK';
	ELSE
		MessageHandler.MessageLine[i].MsgString:='NOK';
	END_IF
END_FOR

MessageHandler(
	Prio:=2, 								(*1=highest, .. , 4=lowest*)
	Btn1Addr:=ADR(MsgOk),						(*Address of Button1 , if Zero then Button is unvisible*)
	Btn2Addr:=0,						(*Address of Button2 , if Zero then Button is unvisible*)
	sVisu:=Visu.Message);
END_ACTION

ACTION Dummy_Test_Nok_exit:
MessageHandler.ClearMessageLines(sVisu:=Visu.Message);
MsgOk:=FALSE;
END_ACTION

ACTION Dummy_Test_Nok_IFM_entry:
MessageHandler.ClearMessageLines(sVisu:=Visu.Message);
MsgOk:=FALSE;
END_ACTION

ACTION Dummy_Test_Nok_IFM_action:
NokMsgString:='';
NokMsgString1:='';

MessageHandler.Msg.ID:='PM56';
MessageHandler.Msg.Name:='IFM Dummyprüfung NOK';
MessageHandler.Msg.Text:='IFM Dummyprüfung NOK';
MessageHandler.Msg.Color:=Color.red;
MessageHandler.Msg.Station:=2;


FOR i:= 7 TO 12 BY 1 DO
	MessageHandler.MessageLine[i-6].MsgTypeEnum:=MsgDataTypeString;
	MessageHandler.MessageLine[i-6].Text:=CONCAT('Dummy_',DINT_TO_STRING(i));
	IF Mp.ST02.Dummy_test_Result[i] THEN
		MessageHandler.MessageLine[i-6].MsgString:='OK';
	ELSE
		MessageHandler.MessageLine[i-6].MsgString:='NOK';
	END_IF
END_FOR


MessageHandler(
	Prio:=2, 								(*1=highest, .. , 4=lowest*)
	Btn1Addr:=ADR(MsgOk),						(*Address of Button1 , if Zero then Button is unvisible*)
	Btn2Addr:=0,						(*Address of Button2 , if Zero then Button is unvisible*)
	sVisu:=Visu.Message);
END_ACTION

ACTION Dummy_Test_Nok_IFM_exit:
MessageHandler.ClearMessageLines(sVisu:=Visu.Message);
MsgOk:=FALSE;
END_ACTION

ACTION Release_Band_action:
ST03_160pol_Zufuehrung.Start:=TRUE;
startBand := TRUE;
END_ACTION

ACTION Wait_for_Dummy_action:
Delay.IN:=ST03_422_B64_4.BitInToCheck;  		 (* Schnittstelle Bedrucken Tinte ISK i.O. oder n.i.O. auf Übergabeposition *)
END_ACTION

ACTION Wait_for_Dummy_exit:
(*Auswertung Kamera Ergebnis für die 6 Dummys*)
IF NOT MP.ST03.SGM_3621 THEN
	IF LoopCounter = 1 THEN
		IF 	ST03_160pol_Zufuehrung.CamResult = 11 AND
			ST03_160pol_Zufuehrung.CamResult2 = 11	 AND
			ST03_160pol_Zufuehrung.CamResult3 = 11 THEN
			Dummy_test_Result[1] := TRUE;
		ELSE
			Dummy_test_Result[1] := FALSE;
		END_IF
	ELSIF LoopCounter = 2 THEN
		IF 	ST03_160pol_Zufuehrung.CamResult = 11 AND
			ST03_160pol_Zufuehrung.CamResult2 = 11  AND
			ST03_160pol_Zufuehrung.CamResult3 = 11 THEN
			Dummy_test_Result[2] := TRUE;
		ELSE
			Dummy_test_Result[2] := FALSE;
		END_IF
	ELSIF LoopCounter = 3 THEN
		IF 	ST03_160pol_Zufuehrung.CamResult = 99 AND
			ST03_160pol_Zufuehrung.CamResult2 = 99	 AND
			ST03_160pol_Zufuehrung.CamResult3 = 99 THEN
			Dummy_test_Result[3] := TRUE;
		ELSE
			Dummy_test_Result[3] := FALSE;
		END_IF
	
	ELSIF LoopCounter = 4 THEN
		IF 	ST03_160pol_Zufuehrung.CamResult = 11 AND
			ST03_160pol_Zufuehrung.CamResult2 = 11	 AND
			ST03_160pol_Zufuehrung.CamResult3 = 99 THEN
			Dummy_test_Result[4] := TRUE;
		ELSE
			Dummy_test_Result[4] := FALSE;
		END_IF
	
	
	ELSIF LoopCounter = 5 THEN
		IF 	ST03_160pol_Zufuehrung.CamResult = 99 AND
			ST03_160pol_Zufuehrung.CamResult2 = 99	 AND
			ST03_160pol_Zufuehrung.CamResult3 = 99 THEN
			Dummy_test_Result[5] := TRUE;
		ELSE
			Dummy_test_Result[5] := FALSE;
		END_IF
	
	ELSIF LoopCounter = 6 THEN
		IF 	ST03_160pol_Zufuehrung.CamResult = 99 AND
			ST03_160pol_Zufuehrung.CamResult2 = 99	 AND
			ST03_160pol_Zufuehrung.CamResult3 = 99 THEN
			Dummy_test_Result[6] := TRUE;
		ELSE
			Dummy_test_Result[6] := FALSE;
		END_IF
	END_IF
ELSE
	IF LoopCounter = 1 THEN
		IF 	ST03_160pol_Zufuehrung.CamResult = 11 AND
			ST03_160pol_Zufuehrung.CamResult2 = 11	 AND
			ST03_160pol_Zufuehrung.CamResult3 = 11 THEN
			Dummy_test_Result[1] := TRUE;
		ELSE
			Dummy_test_Result[1] := FALSE;
		END_IF
	ELSIF LoopCounter = 2 THEN
		IF 	ST03_160pol_Zufuehrung.CamResult = 11 AND
			ST03_160pol_Zufuehrung.CamResult2 = 11	 AND
			ST03_160pol_Zufuehrung.CamResult3 = 11 THEN
			Dummy_test_Result[2] := TRUE;
		ELSE
			Dummy_test_Result[2] := FALSE;
		END_IF
	ELSIF LoopCounter = 3 THEN
		IF 	ST03_160pol_Zufuehrung.CamResult = 99 AND
			ST03_160pol_Zufuehrung.CamResult2 = 99	 AND
			ST03_160pol_Zufuehrung.CamResult3 = 99 THEN
			Dummy_test_Result[3] := TRUE;
		ELSE
			Dummy_test_Result[3] := FALSE;
		END_IF
	
	ELSIF LoopCounter = 4 THEN
		IF 	ST03_160pol_Zufuehrung.CamResult = 11 AND
			ST03_160pol_Zufuehrung.CamResult2 = 11	 AND
			ST03_160pol_Zufuehrung.CamResult3 = 99 THEN
			Dummy_test_Result[4] := TRUE;
		ELSE
			Dummy_test_Result[4] := FALSE;
		END_IF
	
	
	ELSIF LoopCounter = 5 THEN
		IF 	ST03_160pol_Zufuehrung.CamResult =  99 AND
			ST03_160pol_Zufuehrung.CamResult2 = 99	 AND
			ST03_160pol_Zufuehrung.CamResult3 = 99 THEN
			Dummy_test_Result[5] := TRUE;
		ELSE
			Dummy_test_Result[5] := FALSE;
		END_IF
	
	ELSIF LoopCounter = 6 THEN
		IF	ST03_160pol_Zufuehrung.CamResult = 99 AND
			ST03_160pol_Zufuehrung.CamResult2 = 99 AND
			ST03_160pol_Zufuehrung.CamResult3 = 99 THEN
			Dummy_test_Result[6] := TRUE;
		ELSE
			Dummy_test_Result[6] := FALSE;
		END_IF
	END_IF
END_IF
END_ACTION

ACTION Robot01_Pos31_5_action:
Robot01.PosNo:=POS_WT_POS1;
Robot01.PosOffset:=gRobotOffset;
Robot01.Override:=MP.ST00.Override;
Robot01.SetToolOn:=FALSE;
Robot01.SetToolOff:=TRUE;
Robot01.ExecuteMove:=TRUE;
END_ACTION

ACTION Robot01_Pos31_5_exit:
IF ST03_160pol_Zufuehrung.PartOk THEN
	gRob01GripState:=PART_OK;
ELSE
	gRob01GripState:=PART_NOK;
END_IF
END_ACTION

ACTION ST08_Pallett_33__entry:
ProcessMessage01:='';
END_ACTION

ACTION ST08_Pallett_33__action:
ProcessMessage01:='1IM7';(*warte Pallette*)
END_ACTION

ACTION ST08_Pallett_33__exit:
ST08_Process.Start:=FALSE;
ProcessMessage01:='';
END_ACTION

ACTION Robot01_POS_PARK____action:
Robot01.PosNo:=POS_PARK;
Robot01.PosOffset:=gRobotOffset;
Robot01.Override:=MP.ST00.Override;
Robot01.SetToolOn:=FALSE;
Robot01.SetToolOff:=FALSE;
Robot01.ExecuteMove:=TRUE;
END_ACTION

ACTION ST08_Pallett_3____entry:
ProcessMessage01:='';
END_ACTION

ACTION ST08_Pallett_3____action:
ProcessMessage01:='1IM7';(*warte Pallette*)
END_ACTION

ACTION ST08_Pallett_3____exit:
ST08_Process.Start:=FALSE;
ProcessMessage01:='';
END_ACTION

ACTION Robot01_PosPal_entry:
IF 	PosIdx<TD.PartsInRoboGripper THEN
	PosIdx:=TD.PartsInRoboGripper;
END_IF
END_ACTION

ACTION Robot01_PosPal_action:
Robot01.PosNo:=POS_FEED_PAL_WAIT + (PosIdx/TD.PartsInRoboGripper);
Robot01.PosOffset:=gRobotOffset;
Robot01.Override:=MP.ST00.Override;
Robot01.SetToolOn:=TRUE;
Robot01.SetToolOff:=FALSE;
Robot01.ExecuteMove:=TRUE;
END_ACTION

ACTION Robot01_PosPal_exit:
gRob01GripState:=PART_NO;
PosIdx:=PosIdx+TD.PartsInRoboGripper;
gPartsInserted:=gPartsInserted+TD.PartsInRoboGripper;
gPartsTest:=gPartsTest+TD.PartsInRoboGripper;
END_ACTION

ACTION Robot01_Park_Pos__action:
Robot01.PosNo:=POS_PARK;
Robot01.PosOffset:=gRobotOffset;
Robot01.Override:=MP.ST00.Override;
Robot01.SetToolOn:=FALSE;
Robot01.SetToolOff:=FALSE;
Robot01.ExecuteMove:=TRUE;
END_ACTION

ACTION Reset_Test1_action:
(*für das ausschleusen der Testteile mit einem Blister*)
IF LoopCounter >= MAX_NO_OF_DUMMYS THEN
	ST08_Palletizing.TestpartMoveOut:=TRUE;
END_IF
END_ACTION

ACTION ST08_Pallett_action:
IF 	ST08_Process.State=STATE_WAIT THEN
	ST08_Process.Start:=TRUE;
END_IF
END_ACTION

ACTION Count_Dummy_entry:
LoopCounter := LoopCounter +1;
END_ACTION

ACTION Check_Result__entry:
Dummy_ResOK:=TRUE;
END_ACTION

ACTION Check_Result__action:
(*Überprüfung, ob alle Dummys in der richtigen Reihenfolge waren*)
FOR i:=1 TO MAX_NO_OF_DUMMYS
DO
	IF Dummy_test_Result[i] = FALSE
	THEN
		Dummy_ResOK:=FALSE;
	END_IF
END_FOR
END_ACTION

ACTION Dummy_Test_Nok__entry:
MessageHandler.ClearMessageLines(sVisu:=Visu.Message);

NokMsgString:='';
END_ACTION

ACTION Dummy_Test_Nok__action:
MessageHandler.Msg.ID:='PM55';
MessageHandler.Msg.Name:='Dummyprüfung NOK';
MessageHandler.Msg.Text:='Dummyprüfung NOK';
MessageHandler.Msg.Color:=Color.red;
MessageHandler.Msg.Station:=2;


FOR i:= 1 TO MAX_NO_OF_DUMMYS BY 1 DO
	MessageHandler.MessageLine[i].MsgTypeEnum:=MsgDataTypeString;
	MessageHandler.MessageLine[i].Text:=CONCAT('Dummy_',DINT_TO_STRING(i));
	IF Dummy_test_Result[i] THEN
		MessageHandler.MessageLine[i].MsgString:='OK';
	ELSE
		MessageHandler.MessageLine[i].MsgString:='NOK';
	END_IF
END_FOR


MessageHandler(
	Prio:=2, 								(*1=highest, .. , 4=lowest*)
	Btn1Addr:=ADR(MsgOk),						(*Address of Button1 , if Zero then Button is unvisible*)
	Btn2Addr:=0,						(*Address of Button2 , if Zero then Button is unvisible*)
	sVisu:=Visu.Message);
END_ACTION

ACTION Dummy_Test_Nok__exit:
MsgOk := FALSE;
END_ACTION

ACTION Dummy_Test_ok__entry:
MessageHandler.ClearMessageLines(sVisu:=Visu.Message);
END_ACTION

ACTION Dummy_Test_ok__action:
MessageHandler.Msg.ID:='PM54';
MessageHandler.Msg.Name:='DummyTest';
MessageHandler.Msg.Text:=' Dummy Pruefung OK, Ergebnis aller Teile OK ';
MessageHandler.Msg.Color:=Color.green;
MessageHandler.Msg.Station:=1;


MessageHandler(
	Prio:=2, 								(*1=highest, .. , 4=lowest*)
	Btn1Addr:=ADR(MsgOk),						(*Address of Button1 , if Zero then Button is unvisible*)
	Btn2Addr:=0,						(*Address of Button2 , if Zero then Button is unvisible*)
	sVisu:=Visu.Message);
END_ACTION

ACTION Dummy_Test_ok__exit:
MessageHandler.ClearMessageLines(sVisu:=Visu.Message);
MsgOk:=FALSE;
END_ACTION

ACTION SeqEnd_action:
IF 	State=STATE_RUN THEN
	SFCTime:=TIME_TO_DINT(TIME()-SFCTimeStart);
	State:=STATE_OK;
END_IF


IF 	NOT Start THEN
	State:=STATE_WAIT;
END_IF

StartErlaubt93pol:=TRUE;
END_ACTION

TRANSITION 160pol:
gTypeCode=322
END_TRANSITION

TRANSITION Empty:
ST08_CallPRGs.PosIdxHelp = 0
END_TRANSITION

TRANSITION #StateOK:
Robot01.State=STATE_OK

AND gTipImp
END_TRANSITION

TRANSITION 93_102pol:
(gTypeCode=312 OR			(*93pol*)
gTypeCode=499)	(*102pol*)
END_TRANSITION

TRANSITION Kamera_betriebsbereit:
(NOT ST02_DT_95_A1.b_kamera_aktiv (*Kamera Farberkennung*)
OR
NOT ST02_DT_95_A1.sm_kamera_nicht_bb) 	 (*Kamera Farberkennung*)
AND
(NOT ST02_DT_95_A2.sm_kamera_nicht_bb
OR
NOT ST02_DT_95_A2.Activated)
END_TRANSITION

TRANSITION DrehtellerLeer:
gTableEmpty=TRUE
END_TRANSITION

TRANSITION End_Test:
ST02_Main.LoopCounter >= 6
END_TRANSITION

TRANSITION OK_:
Dummy_ResOK=TRUE
END_TRANSITION

TRANSITION Reset_Dummytest:
MP.ST02.DummyPruefung_93pol = FALSE
END_TRANSITION

TRANSITION Reset_Dummytest:
MP.ST02.DummyPruefung_93pol = FALSE
END_TRANSITION

TRANSITION CheckState:
ST03_160pol_Zufuehrung.State = STATE_RUN
END_TRANSITION

TRANSITION DummyReady:
ST03_160pol_Zufuehrung.State <> STATE_RUN
END_TRANSITION

TRANSITION #StateOK:
Robot01.State=STATE_OK

AND gTipImp
END_TRANSITION

TRANSITION StateOk:
ST08_Process.State=STATE_OK
END_TRANSITION

TRANSITION StateWait:
ST08_Process.State=STATE_Wait
END_TRANSITION

TRANSITION Pal_OK:
ST08_Process.Pal_Ready=TRUE
END_TRANSITION

TRANSITION #StateOK:
Robot01.State=STATE_OK

AND gTipImp
END_TRANSITION

TRANSITION StateOk:
ST08_Process.State=STATE_OK OR ST08_Process.State=STATE_Wait
END_TRANSITION

TRANSITION Pal_OK:
ST08_Process.Pal_Ready=TRUE
END_TRANSITION

TRANSITION StateOK:
Robot01.State=STATE_OK
END_TRANSITION

TRANSITION #StateOK:
Robot01.State=STATE_OK

AND gTipImp
END_TRANSITION

TRANSITION StateRun:
ST08_Process.State=STATE_Run
END_TRANSITION

TRANSITION completed:
LoopCounter >= MAX_NO_OF_DUMMYS
END_TRANSITION

TRANSITION Ok:
Dummy_ResOK=TRUE
END_TRANSITION
END_PROGRAM

